REGION Network 57: ABFV 204 CLOSE FB
   RUNG wire#powerrail
      { S7_Templates := "SrcType := Int" } EQ_Contact(in1 := "MODE SELECTION DB"."UF PLC_1 MODE BUFF", in2 := 1)
      { S7_Templates := "SrcType := Int" } EQ_Contact(in1 := "MODE SELECTION DB"."UF PLC_1 PROCESS BUFF", in2 := 255)
      Contact( "INPUT MAPPING DB"."ABFV 204 FEED BACK CLOSE" )
      Move(in := 260, out1 => "MODE SELECTION DB"."UF PLC_1 PROCESS BUFF")
   END_RUNG
   // the same network as SCL:
   IF ("MODE SELECTION DB"."UF PLC_1 MODE BUFF" = 1) AND ("MODE SELECTION DB"."UF PLC_1 PROCESS BUFF" = 255) AND "INPUT MAPPING DB"."ABFV 204 FEED BACK CLOSE" THEN
       "MODE SELECTION DB"."UF PLC_1 PROCESS BUFF" := 260;
   END_IF;
END_REGION

REGION Network 58: ABFV 202 CLOSE FB
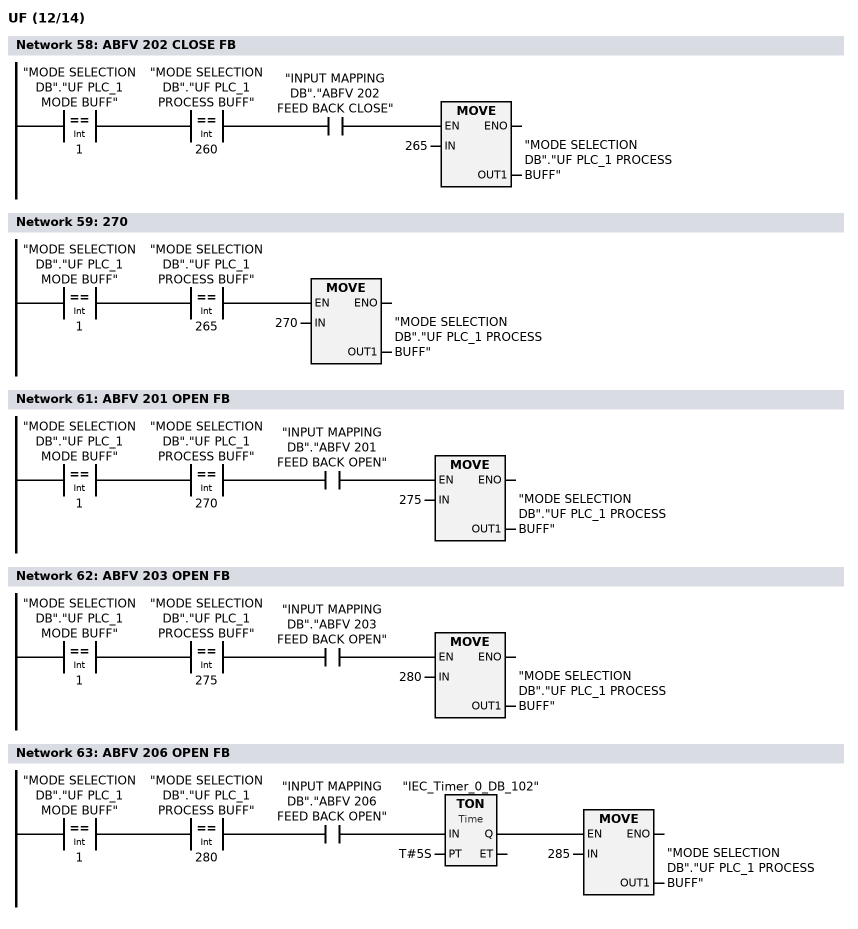
   RUNG wire#powerrail
      { S7_Templates := "SrcType := Int" } EQ_Contact(in1 := "MODE SELECTION DB"."UF PLC_1 MODE BUFF", in2 := 1)
      { S7_Templates := "SrcType := Int" } EQ_Contact(in1 := "MODE SELECTION DB"."UF PLC_1 PROCESS BUFF", in2 := 260)
      Contact( "INPUT MAPPING DB"."ABFV 202 FEED BACK CLOSE" )
      Move(in := 265, out1 => "MODE SELECTION DB"."UF PLC_1 PROCESS BUFF")
   END_RUNG
   // the same network as SCL:
   IF ("MODE SELECTION DB"."UF PLC_1 MODE BUFF" = 1) AND ("MODE SELECTION DB"."UF PLC_1 PROCESS BUFF" = 260) AND "INPUT MAPPING DB"."ABFV 202 FEED BACK CLOSE" THEN
       "MODE SELECTION DB"."UF PLC_1 PROCESS BUFF" := 265;
   END_IF;
END_REGION

REGION Network 59: 270
   RUNG wire#powerrail
      { S7_Templates := "SrcType := Int" } EQ_Contact(in1 := "MODE SELECTION DB"."UF PLC_1 MODE BUFF", in2 := 1)
      { S7_Templates := "SrcType := Int" } EQ_Contact(in1 := "MODE SELECTION DB"."UF PLC_1 PROCESS BUFF", in2 := 265)
      Move(in := 270, out1 => "MODE SELECTION DB"."UF PLC_1 PROCESS BUFF")
   END_RUNG
   // the same network as SCL:
   IF ("MODE SELECTION DB"."UF PLC_1 MODE BUFF" = 1) AND ("MODE SELECTION DB"."UF PLC_1 PROCESS BUFF" = 265) THEN
       "MODE SELECTION DB"."UF PLC_1 PROCESS BUFF" := 270;
   END_IF;
END_REGION

REGION Network 61: ABFV 201 OPEN FB
   RUNG wire#powerrail
      { S7_Templates := "SrcType := Int" } EQ_Contact(in1 := "MODE SELECTION DB"."UF PLC_1 MODE BUFF", in2 := 1)
      { S7_Templates := "SrcType := Int" } EQ_Contact(in1 := "MODE SELECTION DB"."UF PLC_1 PROCESS BUFF", in2 := 270)
      Contact( "INPUT MAPPING DB"."ABFV 201 FEED BACK OPEN" )
      Move(in := 275, out1 => "MODE SELECTION DB"."UF PLC_1 PROCESS BUFF")
   END_RUNG
   // the same network as SCL:
   IF ("MODE SELECTION DB"."UF PLC_1 MODE BUFF" = 1) AND ("MODE SELECTION DB"."UF PLC_1 PROCESS BUFF" = 270) AND "INPUT MAPPING DB"."ABFV 201 FEED BACK OPEN" THEN
       "MODE SELECTION DB"."UF PLC_1 PROCESS BUFF" := 275;
   END_IF;
END_REGION

REGION Network 62: ABFV 203 OPEN FB
   RUNG wire#powerrail
      { S7_Templates := "SrcType := Int" } EQ_Contact(in1 := "MODE SELECTION DB"."UF PLC_1 MODE BUFF", in2 := 1)
      { S7_Templates := "SrcType := Int" } EQ_Contact(in1 := "MODE SELECTION DB"."UF PLC_1 PROCESS BUFF", in2 := 275)
      Contact( "INPUT MAPPING DB"."ABFV 203 FEED BACK OPEN" )
      Move(in := 280, out1 => "MODE SELECTION DB"."UF PLC_1 PROCESS BUFF")
   END_RUNG
   // the same network as SCL:
   IF ("MODE SELECTION DB"."UF PLC_1 MODE BUFF" = 1) AND ("MODE SELECTION DB"."UF PLC_1 PROCESS BUFF" = 275) AND "INPUT MAPPING DB"."ABFV 203 FEED BACK OPEN" THEN
       "MODE SELECTION DB"."UF PLC_1 PROCESS BUFF" := 280;
   END_IF;
END_REGION

REGION Network 63: ABFV 206 OPEN FB
   RUNG wire#powerrail
      { S7_Templates := "SrcType := Int" } EQ_Contact(in1 := "MODE SELECTION DB"."UF PLC_1 MODE BUFF", in2 := 1)
      { S7_Templates := "SrcType := Int" } EQ_Contact(in1 := "MODE SELECTION DB"."UF PLC_1 PROCESS BUFF", in2 := 280)
      Contact( "INPUT MAPPING DB"."ABFV 206 FEED BACK OPEN" )
      { S7_Templates := "time_type := Time" } "IEC_Timer_0_DB_102".TON(pt := T#5S, et =>)
      Move(in := 285, out1 => "MODE SELECTION DB"."UF PLC_1 PROCESS BUFF")
   END_RUNG
   // the same network as SCL:
   "IEC_Timer_0_DB_102".TON(IN := ("MODE SELECTION DB"."UF PLC_1 MODE BUFF" = 1) AND ("MODE SELECTION DB"."UF PLC_1 PROCESS BUFF" = 280) AND "INPUT MAPPING DB"."ABFV 206 FEED BACK OPEN",
                           PT := T#5S);
   IF "IEC_Timer_0_DB_102".Q THEN "MODE SELECTION DB"."UF PLC_1 PROCESS BUFF" := 285; END_IF;
END_REGION

REGION Network 64: FORWARD FLUSH_2
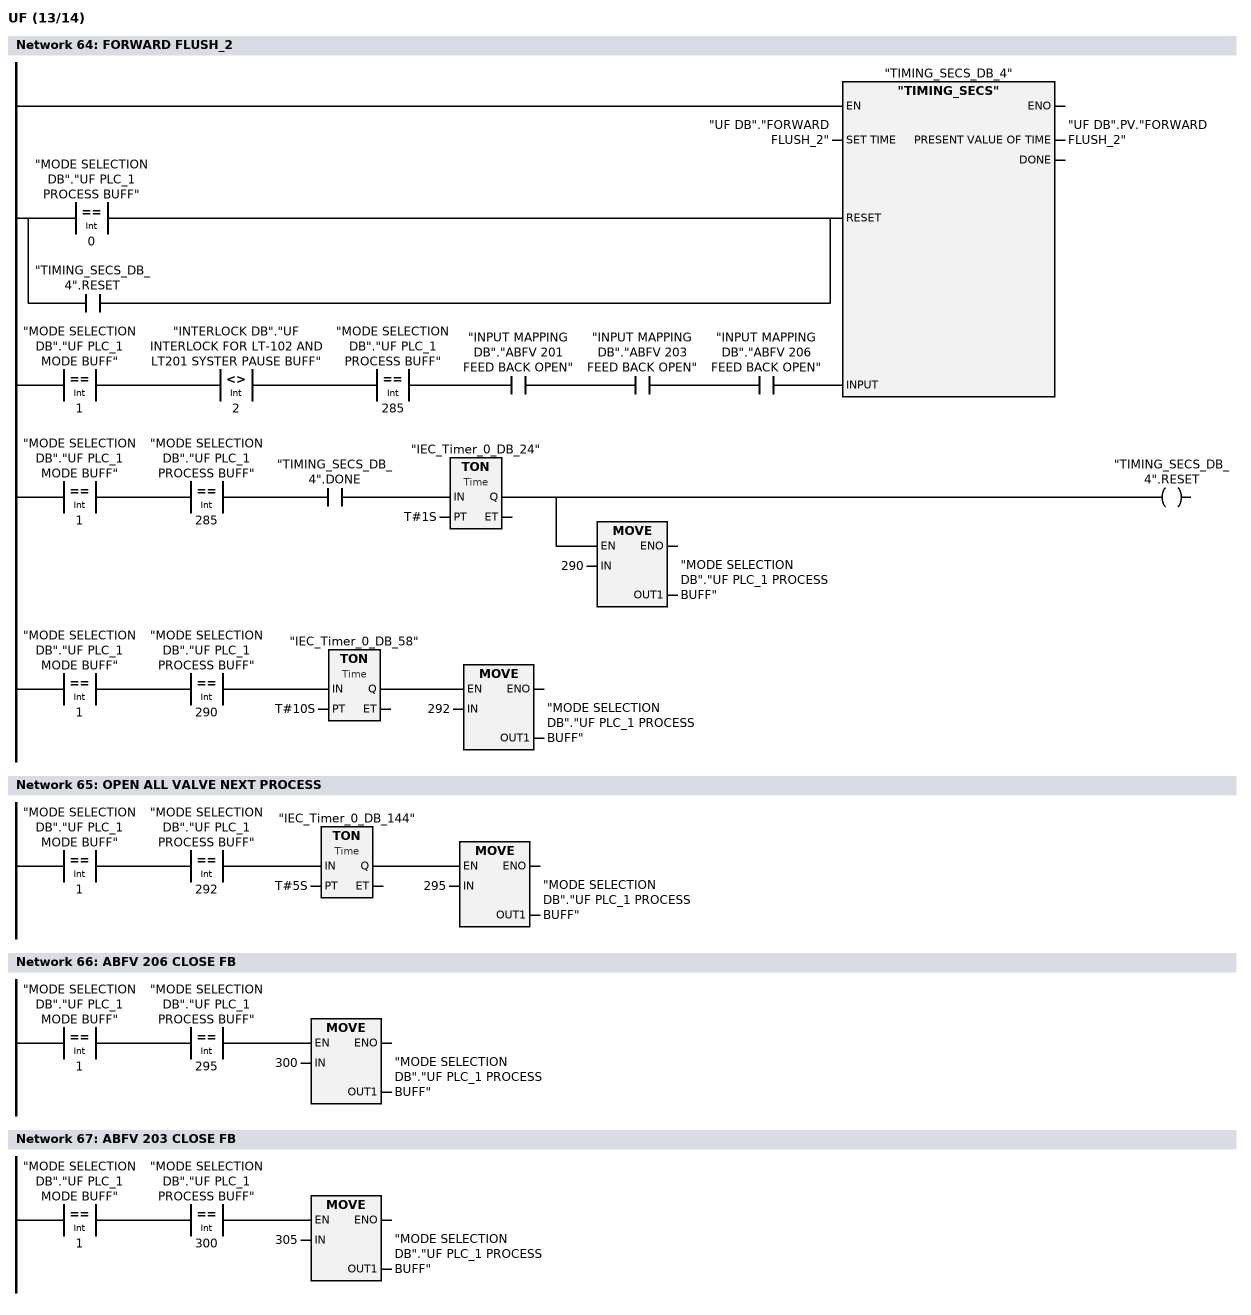
   RUNG wire#powerrail
      "TIMING_SECS_DB_4"(RESET := wire#w1, INPUT := wire#w2, "SET TIME" := "UF DB"."FORWARD FLUSH_2", "PRESENT VALUE OF TIME" => "UF DB".PV."FORWARD FLUSH_2", DONE =>)
   END_RUNG
   RUNG wire#powerrail
      { S7_Templates := "SrcType := Int" } EQ_Contact(in1 := "MODE SELECTION DB"."UF PLC_1 PROCESS BUFF", in2 := 0)
   END_RUNG wire#w1
   RUNG wire#powerrail
      Contact( "TIMING_SECS_DB_4".RESET )
   END_RUNG wire#w1
   RUNG wire#powerrail
      { S7_Templates := "SrcType := Int" } EQ_Contact(in1 := "MODE SELECTION DB"."UF PLC_1 MODE BUFF", in2 := 1)
      { S7_Templates := "SrcType := Int" } NE_Contact(in1 := "INTERLOCK DB"."UF INTERLOCK FOR LT-102 AND LT201 SYSTER PAUSE BUFF", in2 := 2)
      { S7_Templates := "SrcType := Int" } EQ_Contact(in1 := "MODE SELECTION DB"."UF PLC_1 PROCESS BUFF", in2 := 285)
      Contact( "INPUT MAPPING DB"."ABFV 201 FEED BACK OPEN" )
      Contact( "INPUT MAPPING DB"."ABFV 203 FEED BACK OPEN" )
      Contact( "INPUT MAPPING DB"."ABFV 206 FEED BACK OPEN" )
   END_RUNG wire#w2
   RUNG wire#powerrail
      { S7_Templates := "SrcType := Int" } EQ_Contact(in1 := "MODE SELECTION DB"."UF PLC_1 MODE BUFF", in2 := 1)
      { S7_Templates := "SrcType := Int" } EQ_Contact(in1 := "MODE SELECTION DB"."UF PLC_1 PROCESS BUFF", in2 := 285)
      Contact( "TIMING_SECS_DB_4".DONE )
      { S7_Templates := "time_type := Time" } "IEC_Timer_0_DB_24".TON(pt := T#1S, et =>)
      wire#w3
      Coil( "TIMING_SECS_DB_4".RESET )
   END_RUNG
   RUNG wire#w3
      Move(in := 290, out1 => "MODE SELECTION DB"."UF PLC_1 PROCESS BUFF")
   END_RUNG
   RUNG wire#powerrail
      { S7_Templates := "SrcType := Int" } EQ_Contact(in1 := "MODE SELECTION DB"."UF PLC_1 MODE BUFF", in2 := 1)
      { S7_Templates := "SrcType := Int" } EQ_Contact(in1 := "MODE SELECTION DB"."UF PLC_1 PROCESS BUFF", in2 := 290)
      { S7_Templates := "time_type := Time" } "IEC_Timer_0_DB_58".TON(pt := T#10S, et =>)
      Move(in := 292, out1 => "MODE SELECTION DB"."UF PLC_1 PROCESS BUFF")
   END_RUNG
   // the same network as SCL:
   "TIMING_SECS_DB_4"("SET TIME" := "UF DB"."FORWARD FLUSH_2",   // "TIMING_SECS"
                      RESET := ("MODE SELECTION DB"."UF PLC_1 PROCESS BUFF" = 0) OR "TIMING_SECS_DB_4".RESET,
                      INPUT := ("MODE SELECTION DB"."UF PLC_1 MODE BUFF" = 1) AND ("INTERLOCK DB"."UF INTERLOCK FOR LT-102 AND LT201 SYSTER PAUSE BUFF" <> 2) AND ("MODE SELECTION DB"."UF PLC_1 PROCESS BUFF" = 285) AND "INPUT MAPPING DB"."ABFV 201 FEED BACK OPEN" AND "INPUT MAPPING DB"."ABFV 203 FEED BACK OPEN" AND "INPUT MAPPING DB"."ABFV 206 FEED BACK OPEN",
                      "PRESENT VALUE OF TIME" => "UF DB".PV."FORWARD FLUSH_2");
   "IEC_Timer_0_DB_24".TON(IN := ("MODE SELECTION DB"."UF PLC_1 MODE BUFF" = 1) AND ("MODE SELECTION DB"."UF PLC_1 PROCESS BUFF" = 285) AND "TIMING_SECS_DB_4".DONE,
                           PT := T#1S);
   "TIMING_SECS_DB_4".RESET := "IEC_Timer_0_DB_24".Q;
   IF "IEC_Timer_0_DB_24".Q THEN "MODE SELECTION DB"."UF PLC_1 PROCESS BUFF" := 290; END_IF;
   "IEC_Timer_0_DB_58".TON(IN := ("MODE SELECTION DB"."UF PLC_1 MODE BUFF" = 1) AND ("MODE SELECTION DB"."UF PLC_1 PROCESS BUFF" = 290),
                           PT := T#10S);
   IF "IEC_Timer_0_DB_58".Q THEN "MODE SELECTION DB"."UF PLC_1 PROCESS BUFF" := 292; END_IF;
END_REGION

REGION Network 65: OPEN ALL VALVE NEXT PROCESS
   RUNG wire#powerrail
      { S7_Templates := "SrcType := Int" } EQ_Contact(in1 := "MODE SELECTION DB"."UF PLC_1 MODE BUFF", in2 := 1)
      { S7_Templates := "SrcType := Int" } EQ_Contact(in1 := "MODE SELECTION DB"."UF PLC_1 PROCESS BUFF", in2 := 292)
      { S7_Templates := "time_type := Time" } "IEC_Timer_0_DB_144".TON(pt := T#5S, et =>)
      Move(in := 295, out1 => "MODE SELECTION DB"."UF PLC_1 PROCESS BUFF")
   END_RUNG
   // the same network as SCL:
   "IEC_Timer_0_DB_144".TON(IN := ("MODE SELECTION DB"."UF PLC_1 MODE BUFF" = 1) AND ("MODE SELECTION DB"."UF PLC_1 PROCESS BUFF" = 292),
                           PT := T#5S);
   IF "IEC_Timer_0_DB_144".Q THEN "MODE SELECTION DB"."UF PLC_1 PROCESS BUFF" := 295; END_IF;
END_REGION

REGION Network 66: ABFV 206 CLOSE FB
   RUNG wire#powerrail
      { S7_Templates := "SrcType := Int" } EQ_Contact(in1 := "MODE SELECTION DB"."UF PLC_1 MODE BUFF", in2 := 1)
      { S7_Templates := "SrcType := Int" } EQ_Contact(in1 := "MODE SELECTION DB"."UF PLC_1 PROCESS BUFF", in2 := 295)
      Move(in := 300, out1 => "MODE SELECTION DB"."UF PLC_1 PROCESS BUFF")
   END_RUNG
   // the same network as SCL:
   IF ("MODE SELECTION DB"."UF PLC_1 MODE BUFF" = 1) AND ("MODE SELECTION DB"."UF PLC_1 PROCESS BUFF" = 295) THEN
       "MODE SELECTION DB"."UF PLC_1 PROCESS BUFF" := 300;
   END_IF;
END_REGION

REGION Network 67: ABFV 203 CLOSE FB
   RUNG wire#powerrail
      { S7_Templates := "SrcType := Int" } EQ_Contact(in1 := "MODE SELECTION DB"."UF PLC_1 MODE BUFF", in2 := 1)
      { S7_Templates := "SrcType := Int" } EQ_Contact(in1 := "MODE SELECTION DB"."UF PLC_1 PROCESS BUFF", in2 := 300)
      Move(in := 305, out1 => "MODE SELECTION DB"."UF PLC_1 PROCESS BUFF")
   END_RUNG
   // the same network as SCL:
   IF ("MODE SELECTION DB"."UF PLC_1 MODE BUFF" = 1) AND ("MODE SELECTION DB"."UF PLC_1 PROCESS BUFF" = 300) THEN
       "MODE SELECTION DB"."UF PLC_1 PROCESS BUFF" := 305;
   END_IF;
END_REGION

REGION Network 68: ABFV 201 CLOSE FB
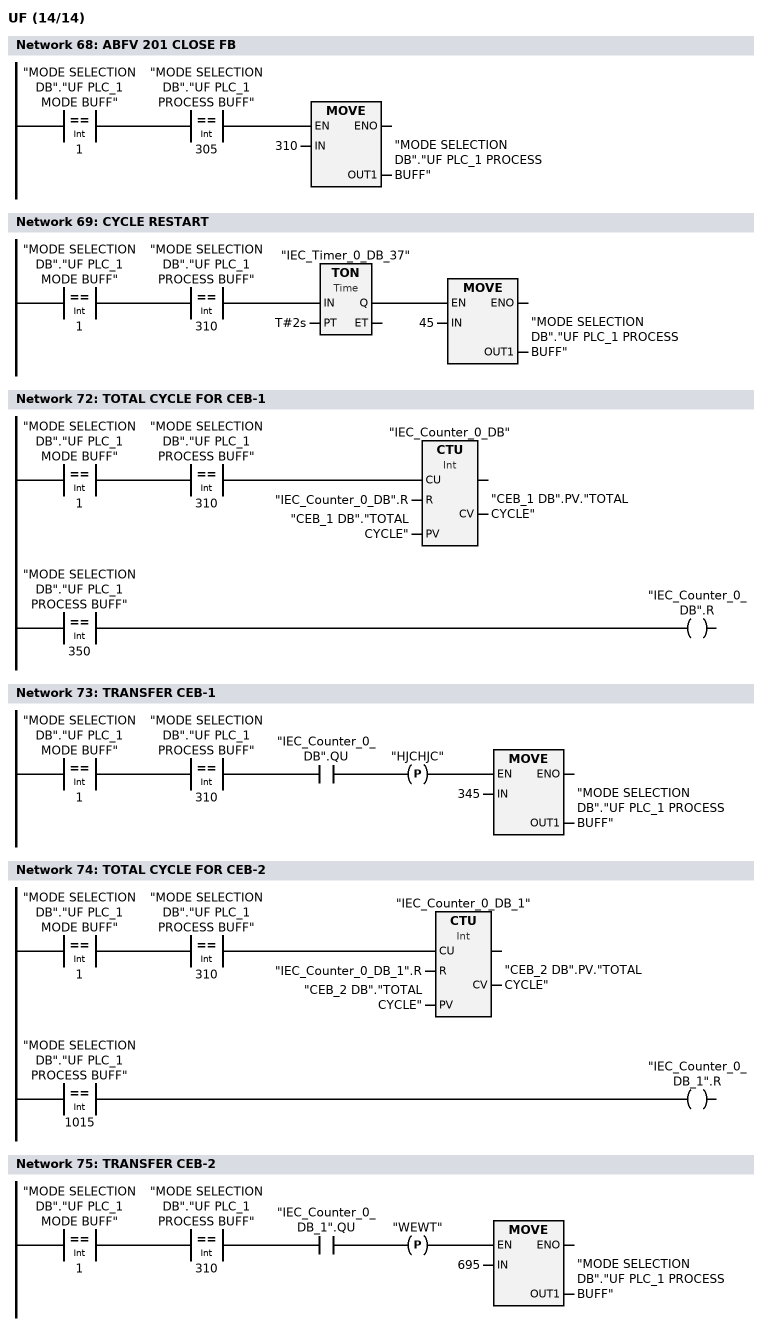
   RUNG wire#powerrail
      { S7_Templates := "SrcType := Int" } EQ_Contact(in1 := "MODE SELECTION DB"."UF PLC_1 MODE BUFF", in2 := 1)
      { S7_Templates := "SrcType := Int" } EQ_Contact(in1 := "MODE SELECTION DB"."UF PLC_1 PROCESS BUFF", in2 := 305)
      Move(in := 310, out1 => "MODE SELECTION DB"."UF PLC_1 PROCESS BUFF")
   END_RUNG
   // the same network as SCL:
   IF ("MODE SELECTION DB"."UF PLC_1 MODE BUFF" = 1) AND ("MODE SELECTION DB"."UF PLC_1 PROCESS BUFF" = 305) THEN
       "MODE SELECTION DB"."UF PLC_1 PROCESS BUFF" := 310;
   END_IF;
END_REGION

REGION Network 69: CYCLE RESTART
   RUNG wire#powerrail
      { S7_Templates := "SrcType := Int" } EQ_Contact(in1 := "MODE SELECTION DB"."UF PLC_1 MODE BUFF", in2 := 1)
      { S7_Templates := "SrcType := Int" } EQ_Contact(in1 := "MODE SELECTION DB"."UF PLC_1 PROCESS BUFF", in2 := 310)
      { S7_Templates := "time_type := Time" } "IEC_Timer_0_DB_37".TON(pt := T#2s, et =>)
      Move(in := 45, out1 => "MODE SELECTION DB"."UF PLC_1 PROCESS BUFF")
   END_RUNG
   // the same network as SCL:
   "IEC_Timer_0_DB_37".TON(IN := ("MODE SELECTION DB"."UF PLC_1 MODE BUFF" = 1) AND ("MODE SELECTION DB"."UF PLC_1 PROCESS BUFF" = 310),
                           PT := T#2s);
   IF "IEC_Timer_0_DB_37".Q THEN "MODE SELECTION DB"."UF PLC_1 PROCESS BUFF" := 45; END_IF;
END_REGION

REGION Network 72: TOTAL CYCLE FOR CEB-1
   RUNG wire#powerrail
      { S7_Templates := "SrcType := Int" } EQ_Contact(in1 := "MODE SELECTION DB"."UF PLC_1 MODE BUFF", in2 := 1)
      { S7_Templates := "SrcType := Int" } EQ_Contact(in1 := "MODE SELECTION DB"."UF PLC_1 PROCESS BUFF", in2 := 310)
      { S7_Templates := "value_type := Int" } "IEC_Counter_0_DB".CTU(r := "IEC_Counter_0_DB".R, pv := "CEB_1 DB"."TOTAL CYCLE", cv => "CEB_1 DB".PV."TOTAL CYCLE")
   END_RUNG
   RUNG wire#powerrail
      { S7_Templates := "SrcType := Int" } EQ_Contact(in1 := "MODE SELECTION DB"."UF PLC_1 PROCESS BUFF", in2 := 350)
      Coil( "IEC_Counter_0_DB".R )
   END_RUNG
   // the same network as SCL:
   "IEC_Counter_0_DB".CTU(CU := ("MODE SELECTION DB"."UF PLC_1 MODE BUFF" = 1) AND ("MODE SELECTION DB"."UF PLC_1 PROCESS BUFF" = 310),
                          R := "IEC_Counter_0_DB".R,
                          PV := "CEB_1 DB"."TOTAL CYCLE",
                          CV => "CEB_1 DB".PV."TOTAL CYCLE");
   "IEC_Counter_0_DB".R := "MODE SELECTION DB"."UF PLC_1 PROCESS BUFF" = 350;
END_REGION

REGION Network 73: TRANSFER CEB-1
   RUNG wire#powerrail
      { S7_Templates := "SrcType := Int" } EQ_Contact(in1 := "MODE SELECTION DB"."UF PLC_1 MODE BUFF", in2 := 1)
      { S7_Templates := "SrcType := Int" } EQ_Contact(in1 := "MODE SELECTION DB"."UF PLC_1 PROCESS BUFF", in2 := 310)
      Contact( "IEC_Counter_0_DB".QU )
      P_Trig( "HJCHJC" )
      Move(in := 345, out1 => "MODE SELECTION DB"."UF PLC_1 PROCESS BUFF")
   END_RUNG
   // the same network as SCL:
   #_w1 := ("MODE SELECTION DB"."UF PLC_1 MODE BUFF" = 1) AND ("MODE SELECTION DB"."UF PLC_1 PROCESS BUFF" = 310) AND "IEC_Counter_0_DB".QU;
   #_w2 := #_w1 AND NOT "HJCHJC";   // rising edge
   "HJCHJC" := #_w1;
   IF #_w2 THEN "MODE SELECTION DB"."UF PLC_1 PROCESS BUFF" := 345; END_IF;
END_REGION

REGION Network 74: TOTAL CYCLE FOR CEB-2
   RUNG wire#powerrail
      { S7_Templates := "SrcType := Int" } EQ_Contact(in1 := "MODE SELECTION DB"."UF PLC_1 MODE BUFF", in2 := 1)
      { S7_Templates := "SrcType := Int" } EQ_Contact(in1 := "MODE SELECTION DB"."UF PLC_1 PROCESS BUFF", in2 := 310)
      { S7_Templates := "value_type := Int" } "IEC_Counter_0_DB_1".CTU(r := "IEC_Counter_0_DB_1".R, pv := "CEB_2 DB"."TOTAL CYCLE", cv => "CEB_2 DB".PV."TOTAL CYCLE")
   END_RUNG
   RUNG wire#powerrail
      { S7_Templates := "SrcType := Int" } EQ_Contact(in1 := "MODE SELECTION DB"."UF PLC_1 PROCESS BUFF", in2 := 1015)
      Coil( "IEC_Counter_0_DB_1".R )
   END_RUNG
   // the same network as SCL:
   "IEC_Counter_0_DB_1".CTU(CU := ("MODE SELECTION DB"."UF PLC_1 MODE BUFF" = 1) AND ("MODE SELECTION DB"."UF PLC_1 PROCESS BUFF" = 310),
                           R := "IEC_Counter_0_DB_1".R,
                           PV := "CEB_2 DB"."TOTAL CYCLE",
                           CV => "CEB_2 DB".PV."TOTAL CYCLE");
   "IEC_Counter_0_DB_1".R := "MODE SELECTION DB"."UF PLC_1 PROCESS BUFF" = 1015;
END_REGION

REGION Network 75: TRANSFER CEB-2
   RUNG wire#powerrail
      { S7_Templates := "SrcType := Int" } EQ_Contact(in1 := "MODE SELECTION DB"."UF PLC_1 MODE BUFF", in2 := 1)
      { S7_Templates := "SrcType := Int" } EQ_Contact(in1 := "MODE SELECTION DB"."UF PLC_1 PROCESS BUFF", in2 := 310)
      Contact( "IEC_Counter_0_DB_1".QU )
      P_Trig( "WEWT" )
      Move(in := 695, out1 => "MODE SELECTION DB"."UF PLC_1 PROCESS BUFF")
   END_RUNG
   // the same network as SCL:
   #_w1 := ("MODE SELECTION DB"."UF PLC_1 MODE BUFF" = 1) AND ("MODE SELECTION DB"."UF PLC_1 PROCESS BUFF" = 310) AND "IEC_Counter_0_DB_1".QU;
   #_w2 := #_w1 AND NOT "WEWT";   // rising edge
   "WEWT" := #_w1;
   IF #_w2 THEN "MODE SELECTION DB"."UF PLC_1 PROCESS BUFF" := 695; END_IF;
END_REGION
END_FUNCTION

FUNCTION_BLOCK "TIMING_SECS"   // FB3, LAD
{ S7_Optimized_Access := 'TRUE' }
// stored: MemoryReserve 100, SetENOAutomatically false
   VAR_INPUT
      "SET TIME" : Int;
      RESET : Bool;
      INPUT : Bool;
   END_VAR
   VAR_OUTPUT
      "PRESENT VALUE OF TIME" : Int;
      DONE : Bool;
   END_VAR
   VAR
      "TIMER 1" { S7_SetPoint := 'True'} : IEC_TIMER;
   END_VAR
   VAR RETAIN
      "COUNTER1 1" { S7_SetPoint := 'True'} : IEC_COUNTER;
   END_VAR
   VAR_TEMP   // added for the SCL form of the ladder/FBD networks
      _w1 : Bool;
      _w2 : Bool;
   END_VAR
BEGIN

REGION Network 1
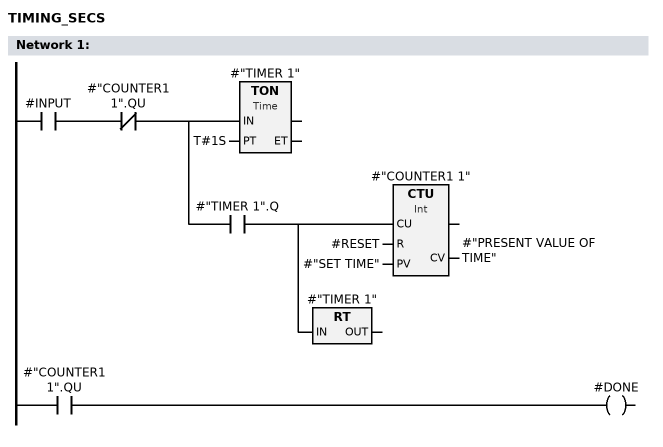
   RUNG wire#powerrail
      Contact( #INPUT )
      I_Contact( #"COUNTER1 1".QU )
      wire#w1
      { S7_Templates := "time_type := Time" } #"TIMER 1".TON(pt := T#1S, et =>)
   END_RUNG
   RUNG wire#w1
      Contact( #"TIMER 1".Q )
      wire#w2
      { S7_Templates := "value_type := Int" } #"COUNTER1 1".CTU(r := #RESET, pv := #"SET TIME", cv => #"PRESENT VALUE OF TIME")
   END_RUNG
   RUNG wire#w2
      RT_Coil( #"TIMER 1" )
   END_RUNG
   RUNG wire#powerrail
      Contact( #"COUNTER1 1".QU )
      Coil( #DONE )
   END_RUNG
   // the same network as SCL:
   #_w1 := #INPUT AND NOT #"COUNTER1 1".QU;
   #"TIMER 1".TON(IN := #_w1, PT := T#1S);
   #_w2 := #_w1 AND #"TIMER 1".Q;
   #"COUNTER1 1".CTU(CU := #_w2, R := #RESET, PV := #"SET TIME", CV => #"PRESENT VALUE OF TIME");
   IF #_w2 THEN RESET_TIMER(#"TIMER 1"); END_IF;
   #DONE := #"COUNTER1 1".QU;
END_REGION
END_FUNCTION_BLOCK

FUNCTION "CEB_1" : Void   // FC14, LAD
{ S7_Optimized_Access := 'TRUE' }
// stored: SetENOAutomatically false
BEGIN

REGION Network 1: CEB_1 START
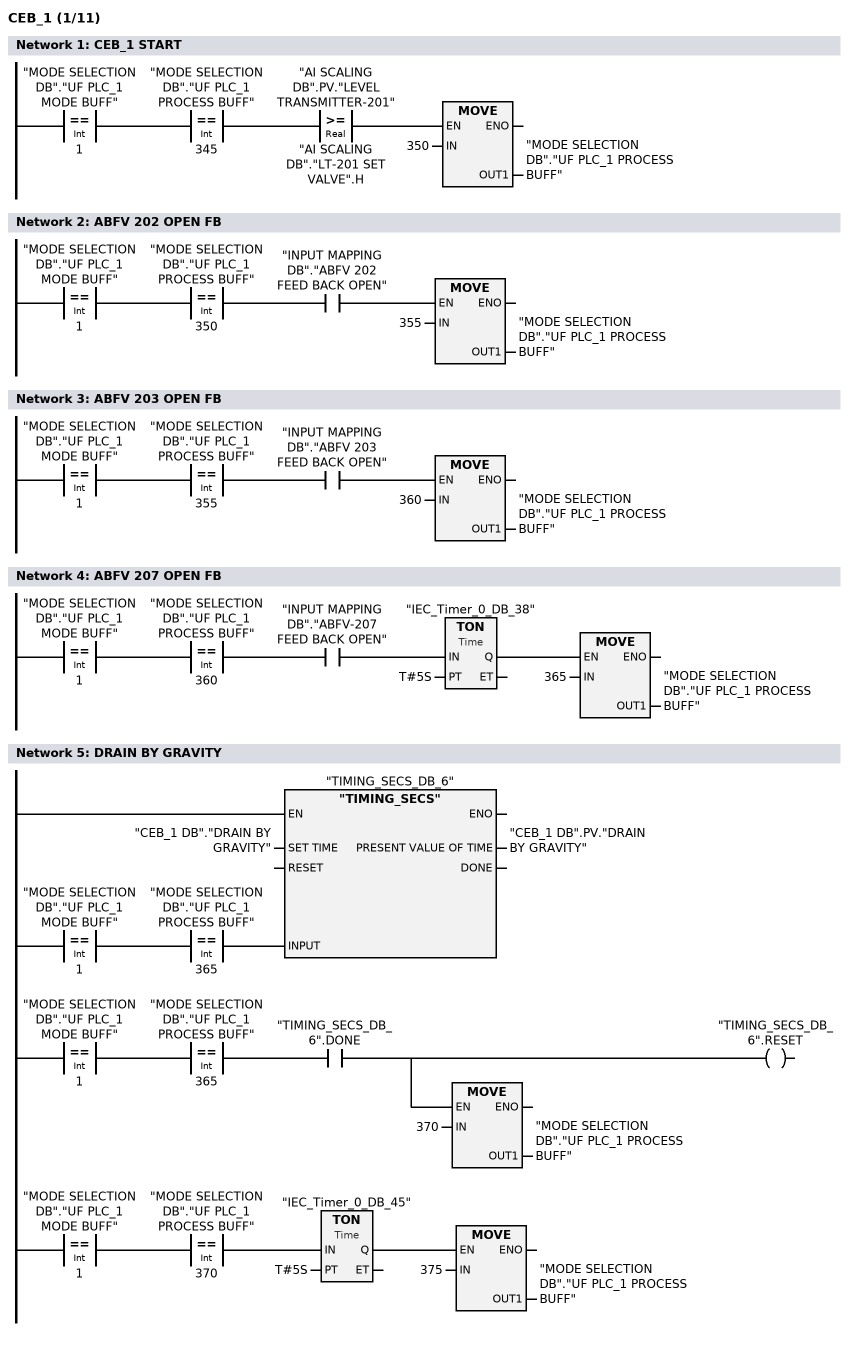
   RUNG wire#powerrail
      { S7_Templates := "SrcType := Int" } EQ_Contact(in1 := "MODE SELECTION DB"."UF PLC_1 MODE BUFF", in2 := 1)
      { S7_Templates := "SrcType := Int" } EQ_Contact(in1 := "MODE SELECTION DB"."UF PLC_1 PROCESS BUFF", in2 := 345)
      { S7_Templates := "SrcType := Real" } GE_Contact(in1 := "AI SCALING DB".PV."LEVEL TRANSMITTER-201", in2 := "AI SCALING DB"."LT-201 SET VALVE".H)
      Move(in := 350, out1 => "MODE SELECTION DB"."UF PLC_1 PROCESS BUFF")
   END_RUNG
   // the same network as SCL:
   IF ("MODE SELECTION DB"."UF PLC_1 MODE BUFF" = 1) AND ("MODE SELECTION DB"."UF PLC_1 PROCESS BUFF" = 345) AND ("AI SCALING DB".PV."LEVEL TRANSMITTER-201" >= "AI SCALING DB"."LT-201 SET VALVE".H) THEN
       "MODE SELECTION DB"."UF PLC_1 PROCESS BUFF" := 350;
   END_IF;
END_REGION

REGION Network 2: ABFV 202 OPEN FB
   RUNG wire#powerrail
      { S7_Templates := "SrcType := Int" } EQ_Contact(in1 := "MODE SELECTION DB"."UF PLC_1 MODE BUFF", in2 := 1)
      { S7_Templates := "SrcType := Int" } EQ_Contact(in1 := "MODE SELECTION DB"."UF PLC_1 PROCESS BUFF", in2 := 350)
      Contact( "INPUT MAPPING DB"."ABFV 202 FEED BACK OPEN" )
      Move(in := 355, out1 => "MODE SELECTION DB"."UF PLC_1 PROCESS BUFF")
   END_RUNG
   // the same network as SCL:
   IF ("MODE SELECTION DB"."UF PLC_1 MODE BUFF" = 1) AND ("MODE SELECTION DB"."UF PLC_1 PROCESS BUFF" = 350) AND "INPUT MAPPING DB"."ABFV 202 FEED BACK OPEN" THEN
       "MODE SELECTION DB"."UF PLC_1 PROCESS BUFF" := 355;
   END_IF;
END_REGION

REGION Network 3: ABFV 203 OPEN FB
   RUNG wire#powerrail
      { S7_Templates := "SrcType := Int" } EQ_Contact(in1 := "MODE SELECTION DB"."UF PLC_1 MODE BUFF", in2 := 1)
      { S7_Templates := "SrcType := Int" } EQ_Contact(in1 := "MODE SELECTION DB"."UF PLC_1 PROCESS BUFF", in2 := 355)
      Contact( "INPUT MAPPING DB"."ABFV 203 FEED BACK OPEN" )
      Move(in := 360, out1 => "MODE SELECTION DB"."UF PLC_1 PROCESS BUFF")
   END_RUNG
   // the same network as SCL:
   IF ("MODE SELECTION DB"."UF PLC_1 MODE BUFF" = 1) AND ("MODE SELECTION DB"."UF PLC_1 PROCESS BUFF" = 355) AND "INPUT MAPPING DB"."ABFV 203 FEED BACK OPEN" THEN
       "MODE SELECTION DB"."UF PLC_1 PROCESS BUFF" := 360;
   END_IF;
END_REGION

REGION Network 4: ABFV 207 OPEN FB
   RUNG wire#powerrail
      { S7_Templates := "SrcType := Int" } EQ_Contact(in1 := "MODE SELECTION DB"."UF PLC_1 MODE BUFF", in2 := 1)
      { S7_Templates := "SrcType := Int" } EQ_Contact(in1 := "MODE SELECTION DB"."UF PLC_1 PROCESS BUFF", in2 := 360)
      Contact( "INPUT MAPPING DB"."ABFV-207 FEED BACK OPEN" )
      { S7_Templates := "time_type := Time" } "IEC_Timer_0_DB_38".TON(pt := T#5S, et =>)
      Move(in := 365, out1 => "MODE SELECTION DB"."UF PLC_1 PROCESS BUFF")
   END_RUNG
   // the same network as SCL:
   "IEC_Timer_0_DB_38".TON(IN := ("MODE SELECTION DB"."UF PLC_1 MODE BUFF" = 1) AND ("MODE SELECTION DB"."UF PLC_1 PROCESS BUFF" = 360) AND "INPUT MAPPING DB"."ABFV-207 FEED BACK OPEN",
                           PT := T#5S);
   IF "IEC_Timer_0_DB_38".Q THEN "MODE SELECTION DB"."UF PLC_1 PROCESS BUFF" := 365; END_IF;
END_REGION

REGION Network 5: DRAIN BY GRAVITY
   RUNG wire#powerrail
      "TIMING_SECS_DB_6"(INPUT := wire#w1, "SET TIME" := "CEB_1 DB"."DRAIN BY GRAVITY", RESET :=, "PRESENT VALUE OF TIME" => "CEB_1 DB".PV."DRAIN BY GRAVITY", DONE =>)
   END_RUNG
   RUNG wire#powerrail
      { S7_Templates := "SrcType := Int" } EQ_Contact(in1 := "MODE SELECTION DB"."UF PLC_1 MODE BUFF", in2 := 1)
      { S7_Templates := "SrcType := Int" } EQ_Contact(in1 := "MODE SELECTION DB"."UF PLC_1 PROCESS BUFF", in2 := 365)
   END_RUNG wire#w1
   RUNG wire#powerrail
      { S7_Templates := "SrcType := Int" } EQ_Contact(in1 := "MODE SELECTION DB"."UF PLC_1 MODE BUFF", in2 := 1)
      { S7_Templates := "SrcType := Int" } EQ_Contact(in1 := "MODE SELECTION DB"."UF PLC_1 PROCESS BUFF", in2 := 365)
      Contact( "TIMING_SECS_DB_6".DONE )
      wire#w2
      Coil( "TIMING_SECS_DB_6".RESET )
   END_RUNG
   RUNG wire#w2
      Move(in := 370, out1 => "MODE SELECTION DB"."UF PLC_1 PROCESS BUFF")
   END_RUNG
   RUNG wire#powerrail
      { S7_Templates := "SrcType := Int" } EQ_Contact(in1 := "MODE SELECTION DB"."UF PLC_1 MODE BUFF", in2 := 1)
      { S7_Templates := "SrcType := Int" } EQ_Contact(in1 := "MODE SELECTION DB"."UF PLC_1 PROCESS BUFF", in2 := 370)
      { S7_Templates := "time_type := Time" } "IEC_Timer_0_DB_45".TON(pt := T#5S, et =>)
      Move(in := 375, out1 => "MODE SELECTION DB"."UF PLC_1 PROCESS BUFF")
   END_RUNG
   // the same network as SCL:
   "TIMING_SECS_DB_6"("SET TIME" := "CEB_1 DB"."DRAIN BY GRAVITY",   // "TIMING_SECS"
                      INPUT := ("MODE SELECTION DB"."UF PLC_1 MODE BUFF" = 1) AND ("MODE SELECTION DB"."UF PLC_1 PROCESS BUFF" = 365),
                      "PRESENT VALUE OF TIME" => "CEB_1 DB".PV."DRAIN BY GRAVITY");
   "TIMING_SECS_DB_6".RESET := ("MODE SELECTION DB"."UF PLC_1 MODE BUFF" = 1) AND ("MODE SELECTION DB"."UF PLC_1 PROCESS BUFF" = 365) AND "TIMING_SECS_DB_6".DONE;
   IF "TIMING_SECS_DB_6".RESET THEN "MODE SELECTION DB"."UF PLC_1 PROCESS BUFF" := 370; END_IF;
   "IEC_Timer_0_DB_45".TON(IN := ("MODE SELECTION DB"."UF PLC_1 MODE BUFF" = 1) AND ("MODE SELECTION DB"."UF PLC_1 PROCESS BUFF" = 370),
                           PT := T#5S);
   IF "IEC_Timer_0_DB_45".Q THEN "MODE SELECTION DB"."UF PLC_1 PROCESS BUFF" := 375; END_IF;
END_REGION

REGION Network 6: ABFV 207 CLOSE FB
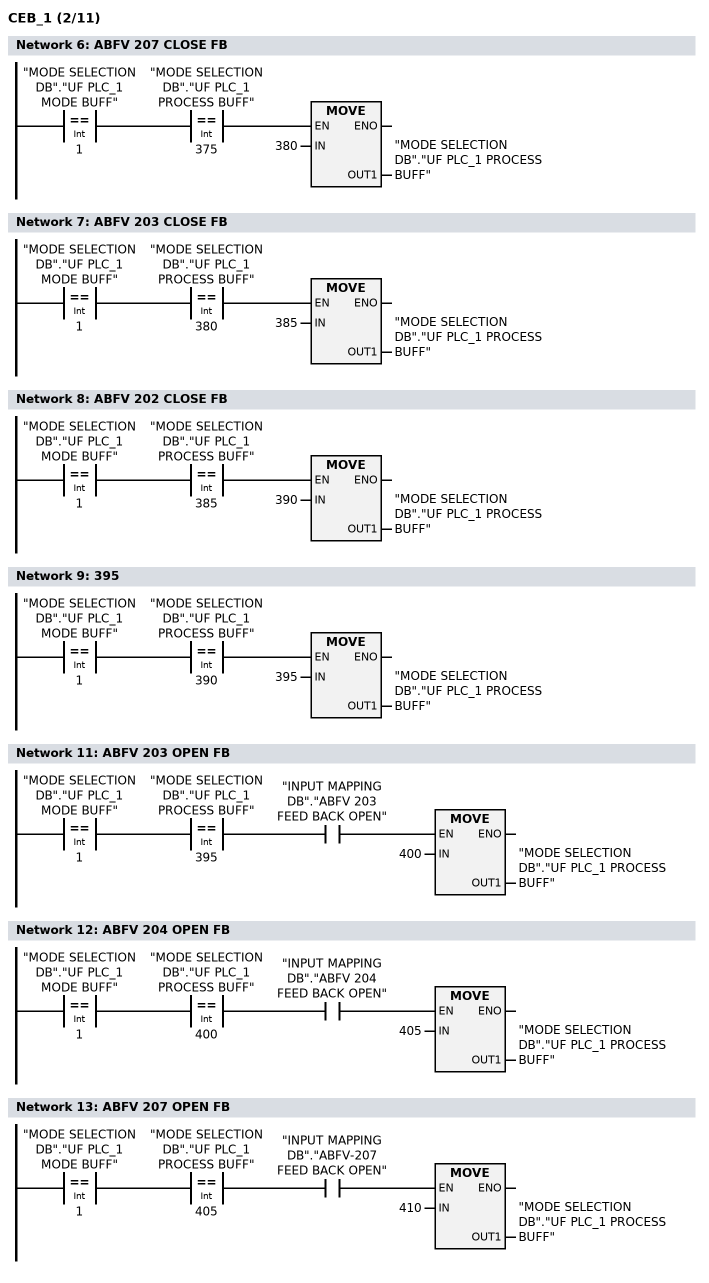
   RUNG wire#powerrail
      { S7_Templates := "SrcType := Int" } EQ_Contact(in1 := "MODE SELECTION DB"."UF PLC_1 MODE BUFF", in2 := 1)
      { S7_Templates := "SrcType := Int" } EQ_Contact(in1 := "MODE SELECTION DB"."UF PLC_1 PROCESS BUFF", in2 := 375)
      Move(in := 380, out1 => "MODE SELECTION DB"."UF PLC_1 PROCESS BUFF")
   END_RUNG
   // the same network as SCL:
   IF ("MODE SELECTION DB"."UF PLC_1 MODE BUFF" = 1) AND ("MODE SELECTION DB"."UF PLC_1 PROCESS BUFF" = 375) THEN
       "MODE SELECTION DB"."UF PLC_1 PROCESS BUFF" := 380;
   END_IF;
END_REGION

REGION Network 7: ABFV 203 CLOSE FB
   RUNG wire#powerrail
      { S7_Templates := "SrcType := Int" } EQ_Contact(in1 := "MODE SELECTION DB"."UF PLC_1 MODE BUFF", in2 := 1)
      { S7_Templates := "SrcType := Int" } EQ_Contact(in1 := "MODE SELECTION DB"."UF PLC_1 PROCESS BUFF", in2 := 380)
      Move(in := 385, out1 => "MODE SELECTION DB"."UF PLC_1 PROCESS BUFF")
   END_RUNG
   // the same network as SCL:
   IF ("MODE SELECTION DB"."UF PLC_1 MODE BUFF" = 1) AND ("MODE SELECTION DB"."UF PLC_1 PROCESS BUFF" = 380) THEN
       "MODE SELECTION DB"."UF PLC_1 PROCESS BUFF" := 385;
   END_IF;
END_REGION

REGION Network 8: ABFV 202 CLOSE FB
   RUNG wire#powerrail
      { S7_Templates := "SrcType := Int" } EQ_Contact(in1 := "MODE SELECTION DB"."UF PLC_1 MODE BUFF", in2 := 1)
      { S7_Templates := "SrcType := Int" } EQ_Contact(in1 := "MODE SELECTION DB"."UF PLC_1 PROCESS BUFF", in2 := 385)
      Move(in := 390, out1 => "MODE SELECTION DB"."UF PLC_1 PROCESS BUFF")
   END_RUNG
   // the same network as SCL:
   IF ("MODE SELECTION DB"."UF PLC_1 MODE BUFF" = 1) AND ("MODE SELECTION DB"."UF PLC_1 PROCESS BUFF" = 385) THEN
       "MODE SELECTION DB"."UF PLC_1 PROCESS BUFF" := 390;
   END_IF;
END_REGION

REGION Network 9: 395
   RUNG wire#powerrail
      { S7_Templates := "SrcType := Int" } EQ_Contact(in1 := "MODE SELECTION DB"."UF PLC_1 MODE BUFF", in2 := 1)
      { S7_Templates := "SrcType := Int" } EQ_Contact(in1 := "MODE SELECTION DB"."UF PLC_1 PROCESS BUFF", in2 := 390)
      Move(in := 395, out1 => "MODE SELECTION DB"."UF PLC_1 PROCESS BUFF")
   END_RUNG
   // the same network as SCL:
   IF ("MODE SELECTION DB"."UF PLC_1 MODE BUFF" = 1) AND ("MODE SELECTION DB"."UF PLC_1 PROCESS BUFF" = 390) THEN
       "MODE SELECTION DB"."UF PLC_1 PROCESS BUFF" := 395;
   END_IF;
END_REGION

REGION Network 11: ABFV 203 OPEN FB
   RUNG wire#powerrail
      { S7_Templates := "SrcType := Int" } EQ_Contact(in1 := "MODE SELECTION DB"."UF PLC_1 MODE BUFF", in2 := 1)
      { S7_Templates := "SrcType := Int" } EQ_Contact(in1 := "MODE SELECTION DB"."UF PLC_1 PROCESS BUFF", in2 := 395)
      Contact( "INPUT MAPPING DB"."ABFV 203 FEED BACK OPEN" )
      Move(in := 400, out1 => "MODE SELECTION DB"."UF PLC_1 PROCESS BUFF")
   END_RUNG
   // the same network as SCL:
   IF ("MODE SELECTION DB"."UF PLC_1 MODE BUFF" = 1) AND ("MODE SELECTION DB"."UF PLC_1 PROCESS BUFF" = 395) AND "INPUT MAPPING DB"."ABFV 203 FEED BACK OPEN" THEN
       "MODE SELECTION DB"."UF PLC_1 PROCESS BUFF" := 400;
   END_IF;
END_REGION

REGION Network 12: ABFV 204 OPEN FB
   RUNG wire#powerrail
      { S7_Templates := "SrcType := Int" } EQ_Contact(in1 := "MODE SELECTION DB"."UF PLC_1 MODE BUFF", in2 := 1)
      { S7_Templates := "SrcType := Int" } EQ_Contact(in1 := "MODE SELECTION DB"."UF PLC_1 PROCESS BUFF", in2 := 400)
      Contact( "INPUT MAPPING DB"."ABFV 204 FEED BACK OPEN" )
      Move(in := 405, out1 => "MODE SELECTION DB"."UF PLC_1 PROCESS BUFF")
   END_RUNG
   // the same network as SCL:
   IF ("MODE SELECTION DB"."UF PLC_1 MODE BUFF" = 1) AND ("MODE SELECTION DB"."UF PLC_1 PROCESS BUFF" = 400) AND "INPUT MAPPING DB"."ABFV 204 FEED BACK OPEN" THEN
       "MODE SELECTION DB"."UF PLC_1 PROCESS BUFF" := 405;
   END_IF;
END_REGION

REGION Network 13: ABFV 207 OPEN FB
   RUNG wire#powerrail
      { S7_Templates := "SrcType := Int" } EQ_Contact(in1 := "MODE SELECTION DB"."UF PLC_1 MODE BUFF", in2 := 1)
      { S7_Templates := "SrcType := Int" } EQ_Contact(in1 := "MODE SELECTION DB"."UF PLC_1 PROCESS BUFF", in2 := 405)
      Contact( "INPUT MAPPING DB"."ABFV-207 FEED BACK OPEN" )
      Move(in := 410, out1 => "MODE SELECTION DB"."UF PLC_1 PROCESS BUFF")
   END_RUNG
   // the same network as SCL:
   IF ("MODE SELECTION DB"."UF PLC_1 MODE BUFF" = 1) AND ("MODE SELECTION DB"."UF PLC_1 PROCESS BUFF" = 405) AND "INPUT MAPPING DB"."ABFV-207 FEED BACK OPEN" THEN
       "MODE SELECTION DB"."UF PLC_1 PROCESS BUFF" := 410;
   END_IF;
END_REGION

REGION Network 14: ABFV 208 OPEN FB
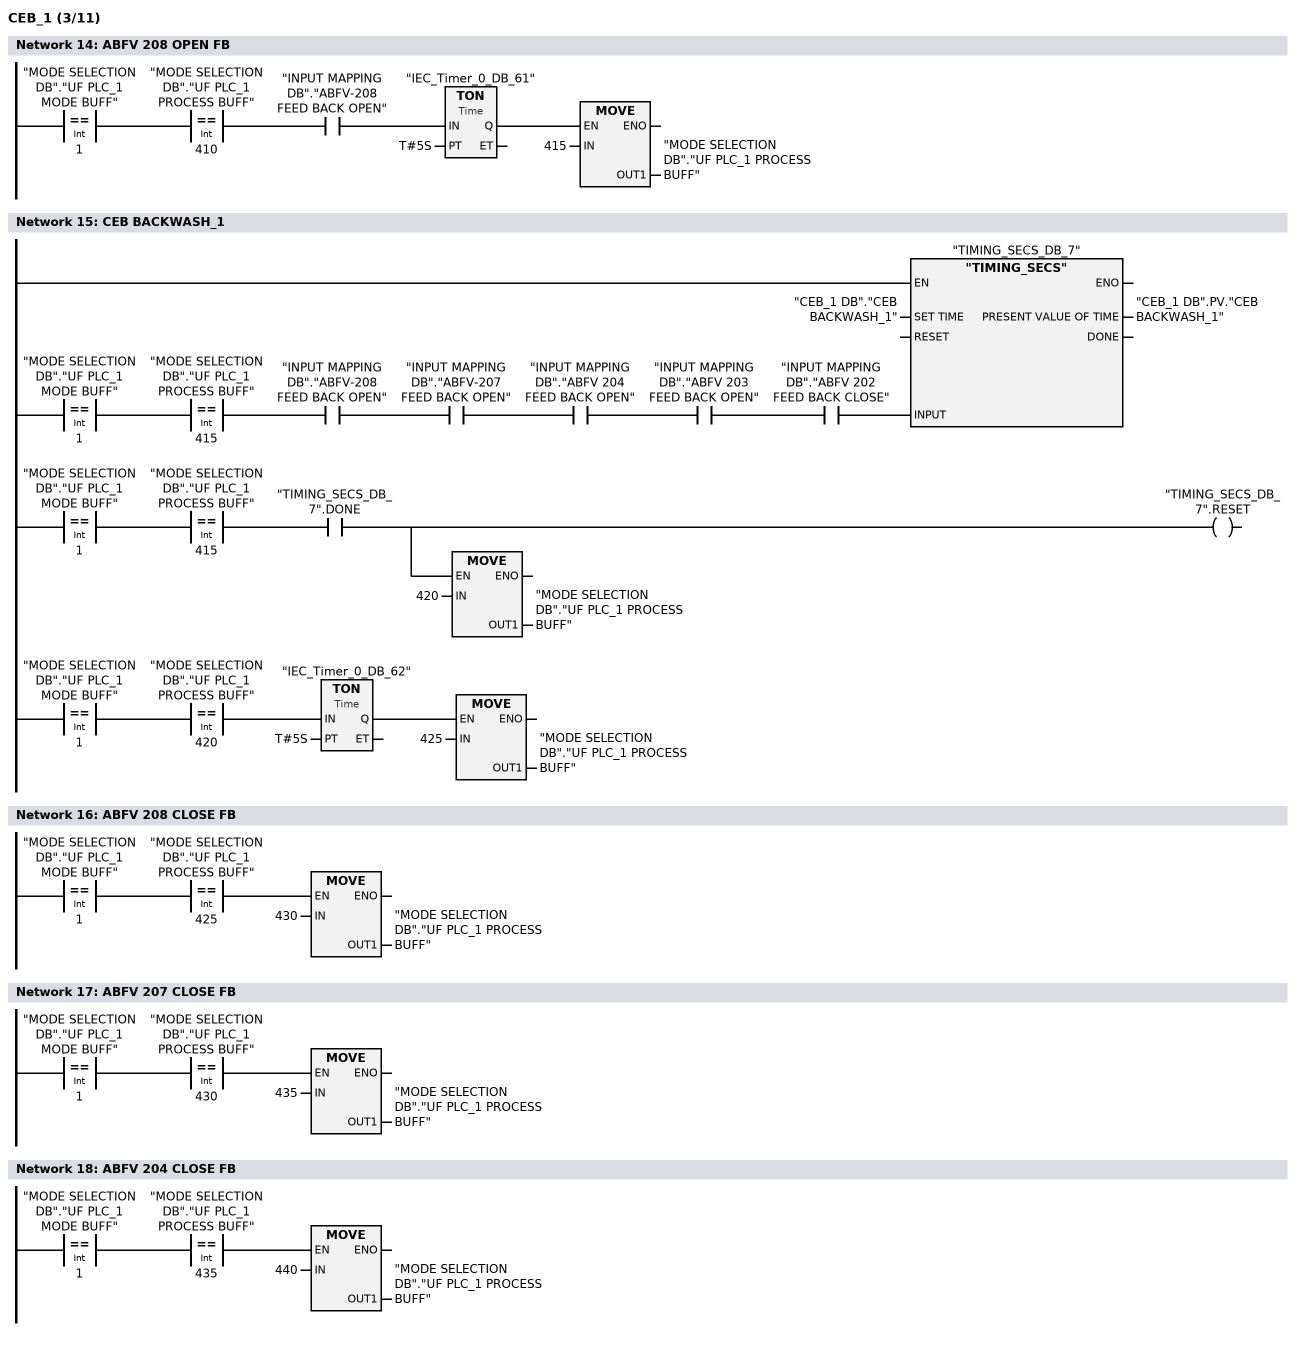
   RUNG wire#powerrail
      { S7_Templates := "SrcType := Int" } EQ_Contact(in1 := "MODE SELECTION DB"."UF PLC_1 MODE BUFF", in2 := 1)
      { S7_Templates := "SrcType := Int" } EQ_Contact(in1 := "MODE SELECTION DB"."UF PLC_1 PROCESS BUFF", in2 := 410)
      Contact( "INPUT MAPPING DB"."ABFV-208 FEED BACK OPEN" )
      { S7_Templates := "time_type := Time" } "IEC_Timer_0_DB_61".TON(pt := T#5S, et =>)
      Move(in := 415, out1 => "MODE SELECTION DB"."UF PLC_1 PROCESS BUFF")
   END_RUNG
   // the same network as SCL:
   "IEC_Timer_0_DB_61".TON(IN := ("MODE SELECTION DB"."UF PLC_1 MODE BUFF" = 1) AND ("MODE SELECTION DB"."UF PLC_1 PROCESS BUFF" = 410) AND "INPUT MAPPING DB"."ABFV-208 FEED BACK OPEN",
                           PT := T#5S);
   IF "IEC_Timer_0_DB_61".Q THEN "MODE SELECTION DB"."UF PLC_1 PROCESS BUFF" := 415; END_IF;
END_REGION

REGION Network 15: CEB BACKWASH_1
   RUNG wire#powerrail
      "TIMING_SECS_DB_7"(INPUT := wire#w1, "SET TIME" := "CEB_1 DB"."CEB BACKWASH_1", RESET :=, "PRESENT VALUE OF TIME" => "CEB_1 DB".PV."CEB BACKWASH_1", DONE =>)
   END_RUNG
   RUNG wire#powerrail
      { S7_Templates := "SrcType := Int" } EQ_Contact(in1 := "MODE SELECTION DB"."UF PLC_1 MODE BUFF", in2 := 1)
      { S7_Templates := "SrcType := Int" } EQ_Contact(in1 := "MODE SELECTION DB"."UF PLC_1 PROCESS BUFF", in2 := 415)
      Contact( "INPUT MAPPING DB"."ABFV-208 FEED BACK OPEN" )
      Contact( "INPUT MAPPING DB"."ABFV-207 FEED BACK OPEN" )
      Contact( "INPUT MAPPING DB"."ABFV 204 FEED BACK OPEN" )
      Contact( "INPUT MAPPING DB"."ABFV 203 FEED BACK OPEN" )
      Contact( "INPUT MAPPING DB"."ABFV 202 FEED BACK CLOSE" )
   END_RUNG wire#w1
   RUNG wire#powerrail
      { S7_Templates := "SrcType := Int" } EQ_Contact(in1 := "MODE SELECTION DB"."UF PLC_1 MODE BUFF", in2 := 1)
      { S7_Templates := "SrcType := Int" } EQ_Contact(in1 := "MODE SELECTION DB"."UF PLC_1 PROCESS BUFF", in2 := 415)
      Contact( "TIMING_SECS_DB_7".DONE )
      wire#w2
      Coil( "TIMING_SECS_DB_7".RESET )
   END_RUNG
   RUNG wire#w2
      Move(in := 420, out1 => "MODE SELECTION DB"."UF PLC_1 PROCESS BUFF")
   END_RUNG
   RUNG wire#powerrail
      { S7_Templates := "SrcType := Int" } EQ_Contact(in1 := "MODE SELECTION DB"."UF PLC_1 MODE BUFF", in2 := 1)
      { S7_Templates := "SrcType := Int" } EQ_Contact(in1 := "MODE SELECTION DB"."UF PLC_1 PROCESS BUFF", in2 := 420)
      { S7_Templates := "time_type := Time" } "IEC_Timer_0_DB_62".TON(pt := T#5S, et =>)
      Move(in := 425, out1 => "MODE SELECTION DB"."UF PLC_1 PROCESS BUFF")
   END_RUNG
   // the same network as SCL:
   "TIMING_SECS_DB_7"("SET TIME" := "CEB_1 DB"."CEB BACKWASH_1",   // "TIMING_SECS"
                      INPUT := ("MODE SELECTION DB"."UF PLC_1 MODE BUFF" = 1) AND ("MODE SELECTION DB"."UF PLC_1 PROCESS BUFF" = 415) AND "INPUT MAPPING DB"."ABFV-208 FEED BACK OPEN" AND "INPUT MAPPING DB"."ABFV-207 FEED BACK OPEN" AND "INPUT MAPPING DB"."ABFV 204 FEED BACK OPEN" AND "INPUT MAPPING DB"."ABFV 203 FEED BACK OPEN" AND "INPUT MAPPING DB"."ABFV 202 FEED BACK CLOSE",
                      "PRESENT VALUE OF TIME" => "CEB_1 DB".PV."CEB BACKWASH_1");
   "TIMING_SECS_DB_7".RESET := ("MODE SELECTION DB"."UF PLC_1 MODE BUFF" = 1) AND ("MODE SELECTION DB"."UF PLC_1 PROCESS BUFF" = 415) AND "TIMING_SECS_DB_7".DONE;
   IF "TIMING_SECS_DB_7".RESET THEN "MODE SELECTION DB"."UF PLC_1 PROCESS BUFF" := 420; END_IF;
   "IEC_Timer_0_DB_62".TON(IN := ("MODE SELECTION DB"."UF PLC_1 MODE BUFF" = 1) AND ("MODE SELECTION DB"."UF PLC_1 PROCESS BUFF" = 420),
                           PT := T#5S);
   IF "IEC_Timer_0_DB_62".Q THEN "MODE SELECTION DB"."UF PLC_1 PROCESS BUFF" := 425; END_IF;
END_REGION

REGION Network 16: ABFV 208 CLOSE FB
   RUNG wire#powerrail
      { S7_Templates := "SrcType := Int" } EQ_Contact(in1 := "MODE SELECTION DB"."UF PLC_1 MODE BUFF", in2 := 1)
      { S7_Templates := "SrcType := Int" } EQ_Contact(in1 := "MODE SELECTION DB"."UF PLC_1 PROCESS BUFF", in2 := 425)
      Move(in := 430, out1 => "MODE SELECTION DB"."UF PLC_1 PROCESS BUFF")
   END_RUNG
   // the same network as SCL:
   IF ("MODE SELECTION DB"."UF PLC_1 MODE BUFF" = 1) AND ("MODE SELECTION DB"."UF PLC_1 PROCESS BUFF" = 425) THEN
       "MODE SELECTION DB"."UF PLC_1 PROCESS BUFF" := 430;
   END_IF;
END_REGION

REGION Network 17: ABFV 207 CLOSE FB
   RUNG wire#powerrail
      { S7_Templates := "SrcType := Int" } EQ_Contact(in1 := "MODE SELECTION DB"."UF PLC_1 MODE BUFF", in2 := 1)
      { S7_Templates := "SrcType := Int" } EQ_Contact(in1 := "MODE SELECTION DB"."UF PLC_1 PROCESS BUFF", in2 := 430)
      Move(in := 435, out1 => "MODE SELECTION DB"."UF PLC_1 PROCESS BUFF")
   END_RUNG
   // the same network as SCL:
   IF ("MODE SELECTION DB"."UF PLC_1 MODE BUFF" = 1) AND ("MODE SELECTION DB"."UF PLC_1 PROCESS BUFF" = 430) THEN
       "MODE SELECTION DB"."UF PLC_1 PROCESS BUFF" := 435;
   END_IF;
END_REGION

REGION Network 18: ABFV 204 CLOSE FB
   RUNG wire#powerrail
      { S7_Templates := "SrcType := Int" } EQ_Contact(in1 := "MODE SELECTION DB"."UF PLC_1 MODE BUFF", in2 := 1)
      { S7_Templates := "SrcType := Int" } EQ_Contact(in1 := "MODE SELECTION DB"."UF PLC_1 PROCESS BUFF", in2 := 435)
      Move(in := 440, out1 => "MODE SELECTION DB"."UF PLC_1 PROCESS BUFF")
   END_RUNG
   // the same network as SCL:
   IF ("MODE SELECTION DB"."UF PLC_1 MODE BUFF" = 1) AND ("MODE SELECTION DB"."UF PLC_1 PROCESS BUFF" = 435) THEN
       "MODE SELECTION DB"."UF PLC_1 PROCESS BUFF" := 440;
   END_IF;
END_REGION

REGION Network 19: ABFV 203 CLOSE FB
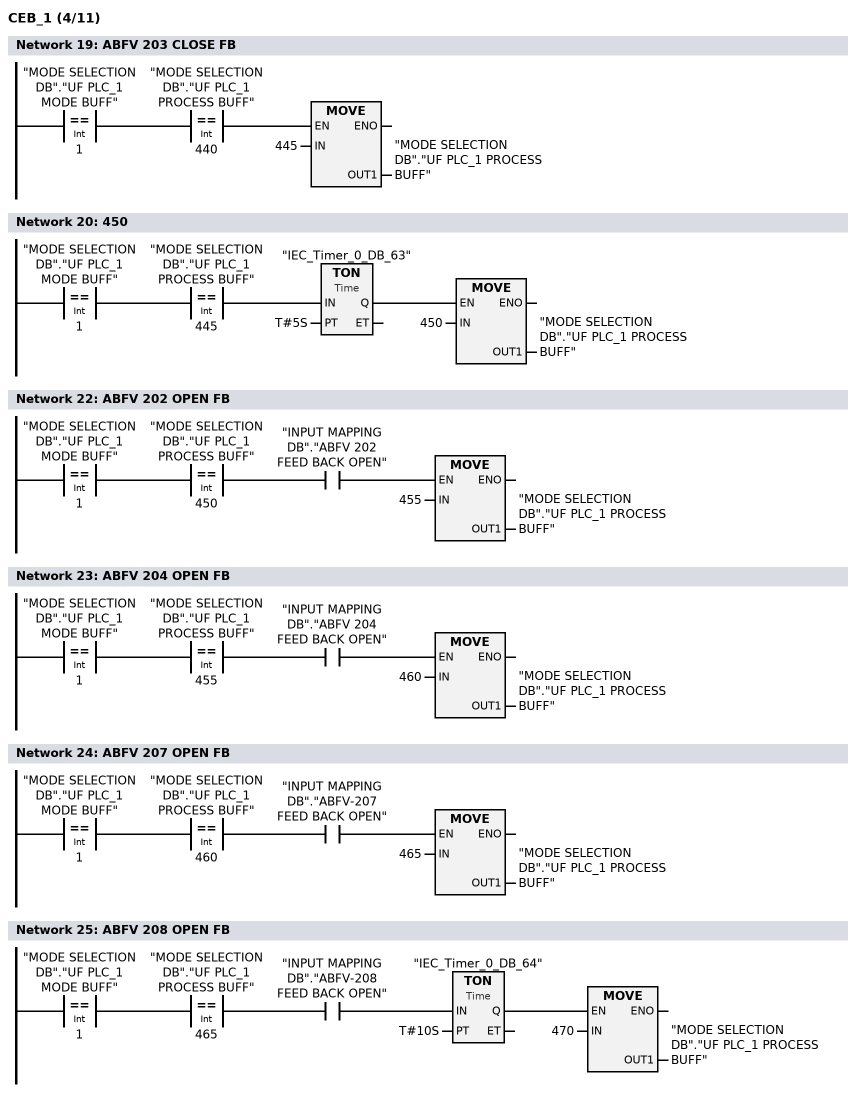
   RUNG wire#powerrail
      { S7_Templates := "SrcType := Int" } EQ_Contact(in1 := "MODE SELECTION DB"."UF PLC_1 MODE BUFF", in2 := 1)
      { S7_Templates := "SrcType := Int" } EQ_Contact(in1 := "MODE SELECTION DB"."UF PLC_1 PROCESS BUFF", in2 := 440)
      Move(in := 445, out1 => "MODE SELECTION DB"."UF PLC_1 PROCESS BUFF")
   END_RUNG
   // the same network as SCL:
   IF ("MODE SELECTION DB"."UF PLC_1 MODE BUFF" = 1) AND ("MODE SELECTION DB"."UF PLC_1 PROCESS BUFF" = 440) THEN
       "MODE SELECTION DB"."UF PLC_1 PROCESS BUFF" := 445;
   END_IF;
END_REGION

REGION Network 20: 450
   RUNG wire#powerrail
      { S7_Templates := "SrcType := Int" } EQ_Contact(in1 := "MODE SELECTION DB"."UF PLC_1 MODE BUFF", in2 := 1)
      { S7_Templates := "SrcType := Int" } EQ_Contact(in1 := "MODE SELECTION DB"."UF PLC_1 PROCESS BUFF", in2 := 445)
      { S7_Templates := "time_type := Time" } "IEC_Timer_0_DB_63".TON(pt := T#5S, et =>)
      Move(in := 450, out1 => "MODE SELECTION DB"."UF PLC_1 PROCESS BUFF")
   END_RUNG
   // the same network as SCL:
   "IEC_Timer_0_DB_63".TON(IN := ("MODE SELECTION DB"."UF PLC_1 MODE BUFF" = 1) AND ("MODE SELECTION DB"."UF PLC_1 PROCESS BUFF" = 445),
                           PT := T#5S);
   IF "IEC_Timer_0_DB_63".Q THEN "MODE SELECTION DB"."UF PLC_1 PROCESS BUFF" := 450; END_IF;
END_REGION

REGION Network 22: ABFV 202 OPEN FB
   RUNG wire#powerrail
      { S7_Templates := "SrcType := Int" } EQ_Contact(in1 := "MODE SELECTION DB"."UF PLC_1 MODE BUFF", in2 := 1)
      { S7_Templates := "SrcType := Int" } EQ_Contact(in1 := "MODE SELECTION DB"."UF PLC_1 PROCESS BUFF", in2 := 450)
      Contact( "INPUT MAPPING DB"."ABFV 202 FEED BACK OPEN" )
      Move(in := 455, out1 => "MODE SELECTION DB"."UF PLC_1 PROCESS BUFF")
   END_RUNG
   // the same network as SCL:
   IF ("MODE SELECTION DB"."UF PLC_1 MODE BUFF" = 1) AND ("MODE SELECTION DB"."UF PLC_1 PROCESS BUFF" = 450) AND "INPUT MAPPING DB"."ABFV 202 FEED BACK OPEN" THEN
       "MODE SELECTION DB"."UF PLC_1 PROCESS BUFF" := 455;
   END_IF;
END_REGION

REGION Network 23: ABFV 204 OPEN FB
   RUNG wire#powerrail
      { S7_Templates := "SrcType := Int" } EQ_Contact(in1 := "MODE SELECTION DB"."UF PLC_1 MODE BUFF", in2 := 1)
      { S7_Templates := "SrcType := Int" } EQ_Contact(in1 := "MODE SELECTION DB"."UF PLC_1 PROCESS BUFF", in2 := 455)
      Contact( "INPUT MAPPING DB"."ABFV 204 FEED BACK OPEN" )
      Move(in := 460, out1 => "MODE SELECTION DB"."UF PLC_1 PROCESS BUFF")
   END_RUNG
   // the same network as SCL:
   IF ("MODE SELECTION DB"."UF PLC_1 MODE BUFF" = 1) AND ("MODE SELECTION DB"."UF PLC_1 PROCESS BUFF" = 455) AND "INPUT MAPPING DB"."ABFV 204 FEED BACK OPEN" THEN
       "MODE SELECTION DB"."UF PLC_1 PROCESS BUFF" := 460;
   END_IF;
END_REGION

REGION Network 24: ABFV 207 OPEN FB
   RUNG wire#powerrail
      { S7_Templates := "SrcType := Int" } EQ_Contact(in1 := "MODE SELECTION DB"."UF PLC_1 MODE BUFF", in2 := 1)
      { S7_Templates := "SrcType := Int" } EQ_Contact(in1 := "MODE SELECTION DB"."UF PLC_1 PROCESS BUFF", in2 := 460)
      Contact( "INPUT MAPPING DB"."ABFV-207 FEED BACK OPEN" )
      Move(in := 465, out1 => "MODE SELECTION DB"."UF PLC_1 PROCESS BUFF")
   END_RUNG
   // the same network as SCL:
   IF ("MODE SELECTION DB"."UF PLC_1 MODE BUFF" = 1) AND ("MODE SELECTION DB"."UF PLC_1 PROCESS BUFF" = 460) AND "INPUT MAPPING DB"."ABFV-207 FEED BACK OPEN" THEN
       "MODE SELECTION DB"."UF PLC_1 PROCESS BUFF" := 465;
   END_IF;
END_REGION

REGION Network 25: ABFV 208 OPEN FB
   RUNG wire#powerrail
      { S7_Templates := "SrcType := Int" } EQ_Contact(in1 := "MODE SELECTION DB"."UF PLC_1 MODE BUFF", in2 := 1)
      { S7_Templates := "SrcType := Int" } EQ_Contact(in1 := "MODE SELECTION DB"."UF PLC_1 PROCESS BUFF", in2 := 465)
      Contact( "INPUT MAPPING DB"."ABFV-208 FEED BACK OPEN" )
      { S7_Templates := "time_type := Time" } "IEC_Timer_0_DB_64".TON(pt := T#10S, et =>)
      Move(in := 470, out1 => "MODE SELECTION DB"."UF PLC_1 PROCESS BUFF")
   END_RUNG
   // the same network as SCL:
   "IEC_Timer_0_DB_64".TON(IN := ("MODE SELECTION DB"."UF PLC_1 MODE BUFF" = 1) AND ("MODE SELECTION DB"."UF PLC_1 PROCESS BUFF" = 465) AND "INPUT MAPPING DB"."ABFV-208 FEED BACK OPEN",
                           PT := T#10S);
   IF "IEC_Timer_0_DB_64".Q THEN "MODE SELECTION DB"."UF PLC_1 PROCESS BUFF" := 470; END_IF;
END_REGION

REGION Network 26: CEB BACKWASH_2
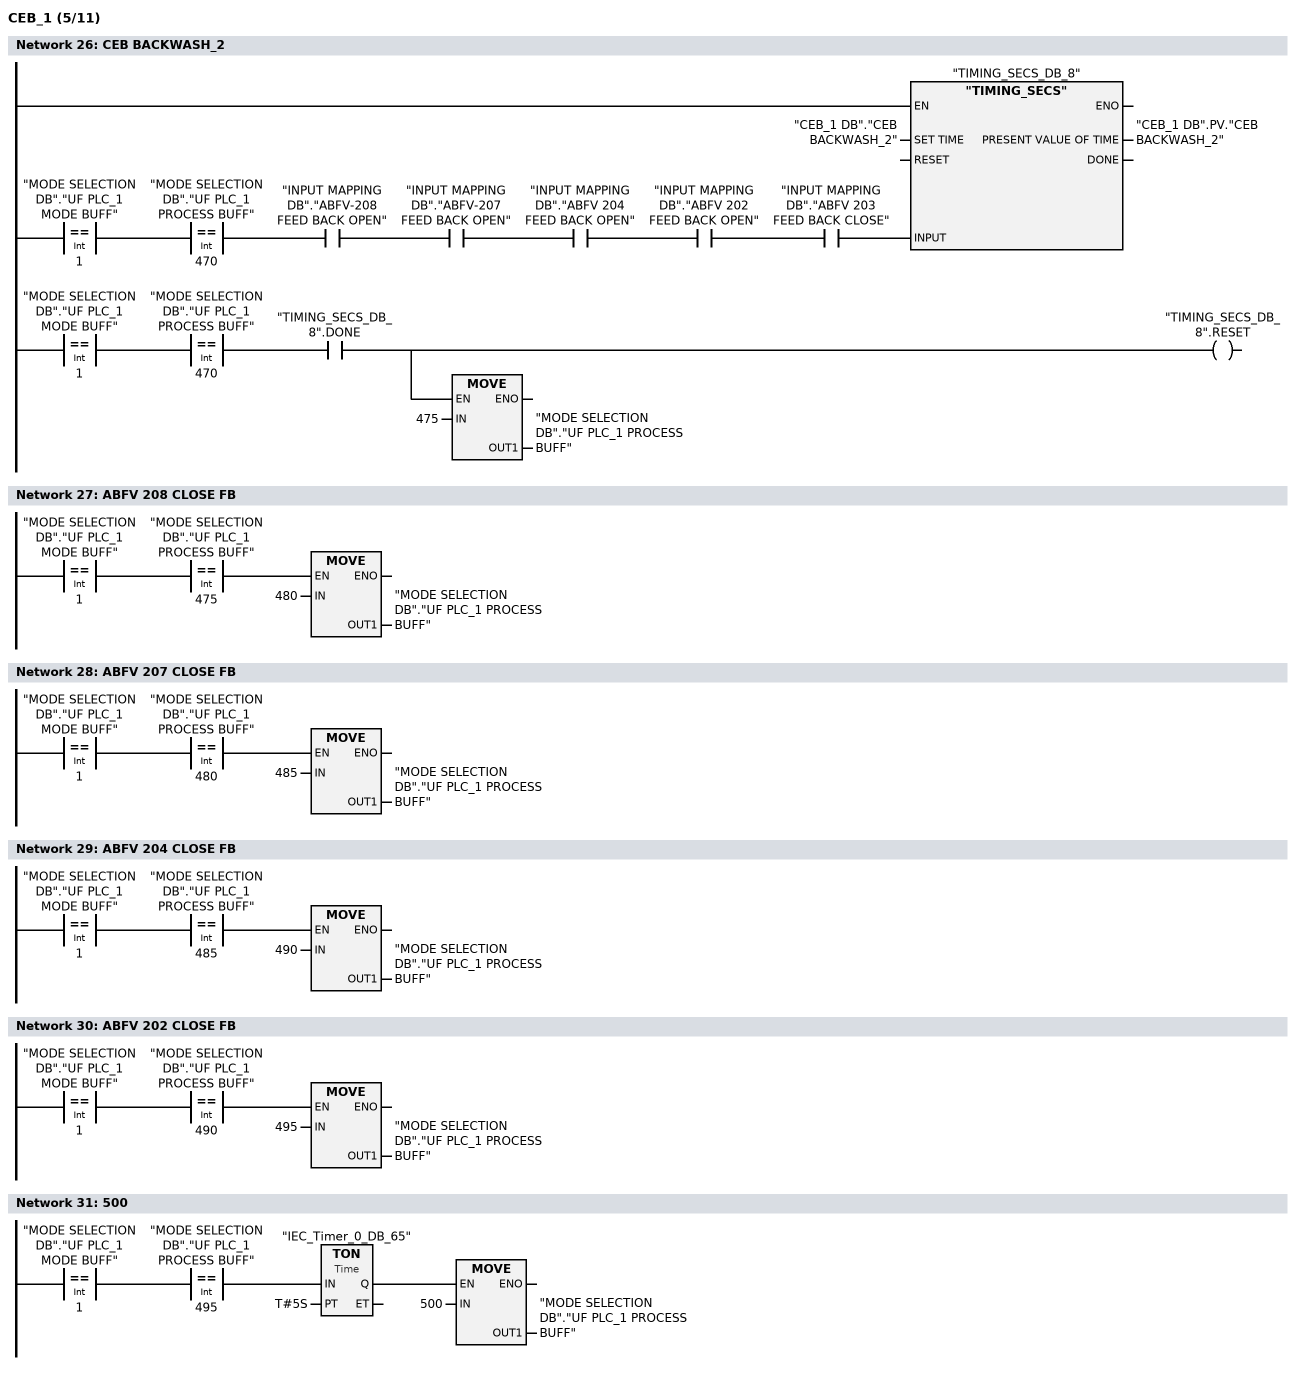
   RUNG wire#powerrail
      "TIMING_SECS_DB_8"(INPUT := wire#w1, "SET TIME" := "CEB_1 DB"."CEB BACKWASH_2", RESET :=, "PRESENT VALUE OF TIME" => "CEB_1 DB".PV."CEB BACKWASH_2", DONE =>)
   END_RUNG
   RUNG wire#powerrail
      { S7_Templates := "SrcType := Int" } EQ_Contact(in1 := "MODE SELECTION DB"."UF PLC_1 MODE BUFF", in2 := 1)
      { S7_Templates := "SrcType := Int" } EQ_Contact(in1 := "MODE SELECTION DB"."UF PLC_1 PROCESS BUFF", in2 := 470)
      Contact( "INPUT MAPPING DB"."ABFV-208 FEED BACK OPEN" )
      Contact( "INPUT MAPPING DB"."ABFV-207 FEED BACK OPEN" )
      Contact( "INPUT MAPPING DB"."ABFV 204 FEED BACK OPEN" )
      Contact( "INPUT MAPPING DB"."ABFV 202 FEED BACK OPEN" )
      Contact( "INPUT MAPPING DB"."ABFV 203 FEED BACK CLOSE" )
   END_RUNG wire#w1
   RUNG wire#powerrail
      { S7_Templates := "SrcType := Int" } EQ_Contact(in1 := "MODE SELECTION DB"."UF PLC_1 MODE BUFF", in2 := 1)
      { S7_Templates := "SrcType := Int" } EQ_Contact(in1 := "MODE SELECTION DB"."UF PLC_1 PROCESS BUFF", in2 := 470)
      Contact( "TIMING_SECS_DB_8".DONE )
      wire#w2
      Coil( "TIMING_SECS_DB_8".RESET )
   END_RUNG
   RUNG wire#w2
      Move(in := 475, out1 => "MODE SELECTION DB"."UF PLC_1 PROCESS BUFF")
   END_RUNG
   // the same network as SCL:
   "TIMING_SECS_DB_8"("SET TIME" := "CEB_1 DB"."CEB BACKWASH_2",   // "TIMING_SECS"
                      INPUT := ("MODE SELECTION DB"."UF PLC_1 MODE BUFF" = 1) AND ("MODE SELECTION DB"."UF PLC_1 PROCESS BUFF" = 470) AND "INPUT MAPPING DB"."ABFV-208 FEED BACK OPEN" AND "INPUT MAPPING DB"."ABFV-207 FEED BACK OPEN" AND "INPUT MAPPING DB"."ABFV 204 FEED BACK OPEN" AND "INPUT MAPPING DB"."ABFV 202 FEED BACK OPEN" AND "INPUT MAPPING DB"."ABFV 203 FEED BACK CLOSE",
                      "PRESENT VALUE OF TIME" => "CEB_1 DB".PV."CEB BACKWASH_2");
   "TIMING_SECS_DB_8".RESET := ("MODE SELECTION DB"."UF PLC_1 MODE BUFF" = 1) AND ("MODE SELECTION DB"."UF PLC_1 PROCESS BUFF" = 470) AND "TIMING_SECS_DB_8".DONE;
   IF "TIMING_SECS_DB_8".RESET THEN "MODE SELECTION DB"."UF PLC_1 PROCESS BUFF" := 475; END_IF;
END_REGION

REGION Network 27: ABFV 208 CLOSE FB
   RUNG wire#powerrail
      { S7_Templates := "SrcType := Int" } EQ_Contact(in1 := "MODE SELECTION DB"."UF PLC_1 MODE BUFF", in2 := 1)
      { S7_Templates := "SrcType := Int" } EQ_Contact(in1 := "MODE SELECTION DB"."UF PLC_1 PROCESS BUFF", in2 := 475)
      Move(in := 480, out1 => "MODE SELECTION DB"."UF PLC_1 PROCESS BUFF")
   END_RUNG
   // the same network as SCL:
   IF ("MODE SELECTION DB"."UF PLC_1 MODE BUFF" = 1) AND ("MODE SELECTION DB"."UF PLC_1 PROCESS BUFF" = 475) THEN
       "MODE SELECTION DB"."UF PLC_1 PROCESS BUFF" := 480;
   END_IF;
END_REGION

REGION Network 28: ABFV 207 CLOSE FB
   RUNG wire#powerrail
      { S7_Templates := "SrcType := Int" } EQ_Contact(in1 := "MODE SELECTION DB"."UF PLC_1 MODE BUFF", in2 := 1)
      { S7_Templates := "SrcType := Int" } EQ_Contact(in1 := "MODE SELECTION DB"."UF PLC_1 PROCESS BUFF", in2 := 480)
      Move(in := 485, out1 => "MODE SELECTION DB"."UF PLC_1 PROCESS BUFF")
   END_RUNG
   // the same network as SCL:
   IF ("MODE SELECTION DB"."UF PLC_1 MODE BUFF" = 1) AND ("MODE SELECTION DB"."UF PLC_1 PROCESS BUFF" = 480) THEN
       "MODE SELECTION DB"."UF PLC_1 PROCESS BUFF" := 485;
   END_IF;
END_REGION

REGION Network 29: ABFV 204 CLOSE FB
   RUNG wire#powerrail
      { S7_Templates := "SrcType := Int" } EQ_Contact(in1 := "MODE SELECTION DB"."UF PLC_1 MODE BUFF", in2 := 1)
      { S7_Templates := "SrcType := Int" } EQ_Contact(in1 := "MODE SELECTION DB"."UF PLC_1 PROCESS BUFF", in2 := 485)
      Move(in := 490, out1 => "MODE SELECTION DB"."UF PLC_1 PROCESS BUFF")
   END_RUNG
   // the same network as SCL:
   IF ("MODE SELECTION DB"."UF PLC_1 MODE BUFF" = 1) AND ("MODE SELECTION DB"."UF PLC_1 PROCESS BUFF" = 485) THEN
       "MODE SELECTION DB"."UF PLC_1 PROCESS BUFF" := 490;
   END_IF;
END_REGION

REGION Network 30: ABFV 202 CLOSE FB
   RUNG wire#powerrail
      { S7_Templates := "SrcType := Int" } EQ_Contact(in1 := "MODE SELECTION DB"."UF PLC_1 MODE BUFF", in2 := 1)
      { S7_Templates := "SrcType := Int" } EQ_Contact(in1 := "MODE SELECTION DB"."UF PLC_1 PROCESS BUFF", in2 := 490)
      Move(in := 495, out1 => "MODE SELECTION DB"."UF PLC_1 PROCESS BUFF")
   END_RUNG
   // the same network as SCL:
   IF ("MODE SELECTION DB"."UF PLC_1 MODE BUFF" = 1) AND ("MODE SELECTION DB"."UF PLC_1 PROCESS BUFF" = 490) THEN
       "MODE SELECTION DB"."UF PLC_1 PROCESS BUFF" := 495;
   END_IF;
END_REGION

REGION Network 31: 500
   RUNG wire#powerrail
      { S7_Templates := "SrcType := Int" } EQ_Contact(in1 := "MODE SELECTION DB"."UF PLC_1 MODE BUFF", in2 := 1)
      { S7_Templates := "SrcType := Int" } EQ_Contact(in1 := "MODE SELECTION DB"."UF PLC_1 PROCESS BUFF", in2 := 495)
      { S7_Templates := "time_type := Time" } "IEC_Timer_0_DB_65".TON(pt := T#5S, et =>)
      Move(in := 500, out1 => "MODE SELECTION DB"."UF PLC_1 PROCESS BUFF")
   END_RUNG
   // the same network as SCL:
   "IEC_Timer_0_DB_65".TON(IN := ("MODE SELECTION DB"."UF PLC_1 MODE BUFF" = 1) AND ("MODE SELECTION DB"."UF PLC_1 PROCESS BUFF" = 495),
                           PT := T#5S);
   IF "IEC_Timer_0_DB_65".Q THEN "MODE SELECTION DB"."UF PLC_1 PROCESS BUFF" := 500; END_IF;
END_REGION

REGION Network 33: SOAK
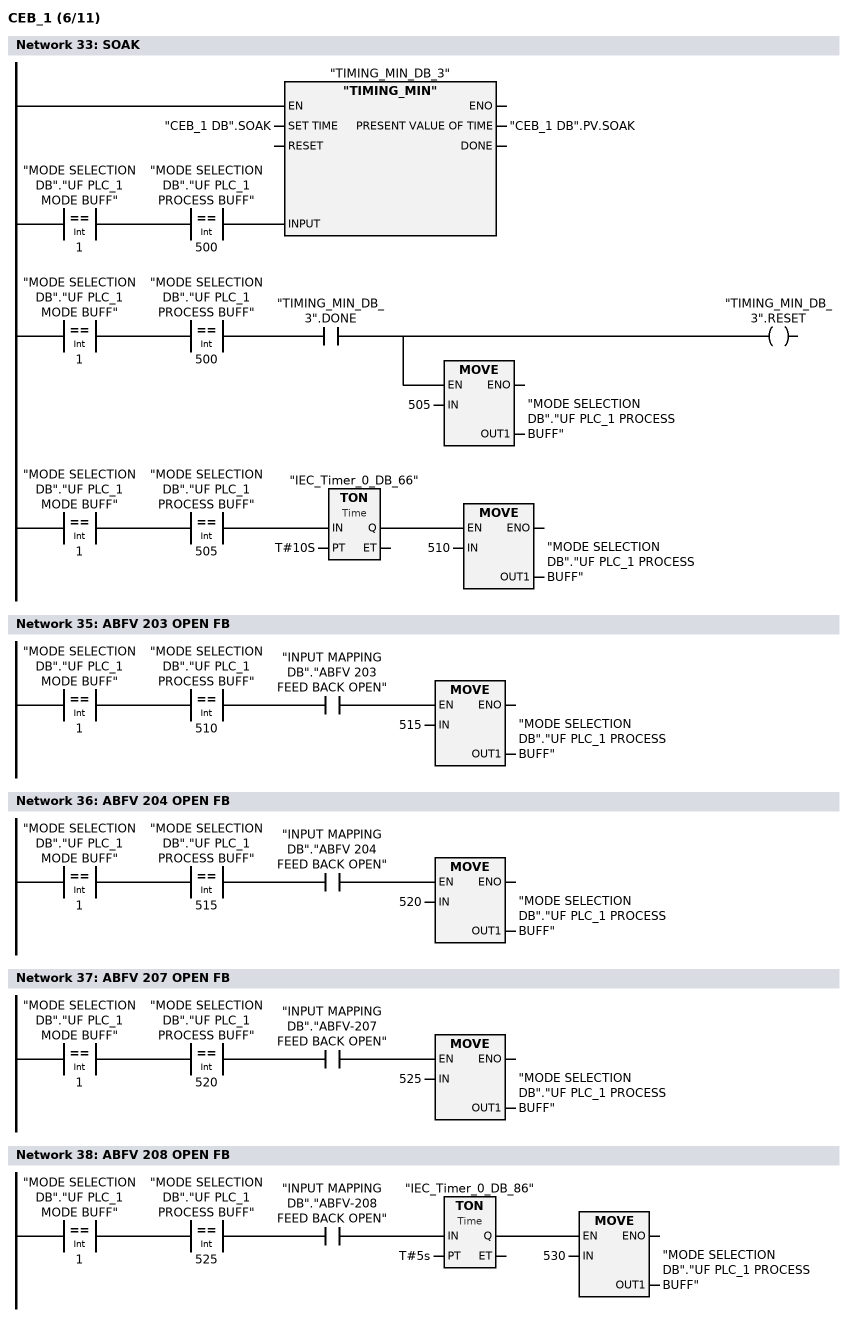
   RUNG wire#powerrail
      "TIMING_MIN_DB_3"(INPUT := wire#w1, "SET TIME" := "CEB_1 DB".SOAK, RESET :=, "PRESENT VALUE OF TIME" => "CEB_1 DB".PV.SOAK, DONE =>)
   END_RUNG
   RUNG wire#powerrail
      { S7_Templates := "SrcType := Int" } EQ_Contact(in1 := "MODE SELECTION DB"."UF PLC_1 MODE BUFF", in2 := 1)
      { S7_Templates := "SrcType := Int" } EQ_Contact(in1 := "MODE SELECTION DB"."UF PLC_1 PROCESS BUFF", in2 := 500)
   END_RUNG wire#w1
   RUNG wire#powerrail
      { S7_Templates := "SrcType := Int" } EQ_Contact(in1 := "MODE SELECTION DB"."UF PLC_1 MODE BUFF", in2 := 1)
      { S7_Templates := "SrcType := Int" } EQ_Contact(in1 := "MODE SELECTION DB"."UF PLC_1 PROCESS BUFF", in2 := 500)
      Contact( "TIMING_MIN_DB_3".DONE )
      wire#w2
      Coil( "TIMING_MIN_DB_3".RESET )
   END_RUNG
   RUNG wire#w2
      Move(in := 505, out1 => "MODE SELECTION DB"."UF PLC_1 PROCESS BUFF")
   END_RUNG
   RUNG wire#powerrail
      { S7_Templates := "SrcType := Int" } EQ_Contact(in1 := "MODE SELECTION DB"."UF PLC_1 MODE BUFF", in2 := 1)
      { S7_Templates := "SrcType := Int" } EQ_Contact(in1 := "MODE SELECTION DB"."UF PLC_1 PROCESS BUFF", in2 := 505)
      { S7_Templates := "time_type := Time" } "IEC_Timer_0_DB_66".TON(pt := T#10S, et =>)
      Move(in := 510, out1 => "MODE SELECTION DB"."UF PLC_1 PROCESS BUFF")
   END_RUNG
   // the same network as SCL:
   "TIMING_MIN_DB_3"("SET TIME" := "CEB_1 DB".SOAK,   // "TIMING_MIN"
                     INPUT := ("MODE SELECTION DB"."UF PLC_1 MODE BUFF" = 1) AND ("MODE SELECTION DB"."UF PLC_1 PROCESS BUFF" = 500),
                     "PRESENT VALUE OF TIME" => "CEB_1 DB".PV.SOAK);
   "TIMING_MIN_DB_3".RESET := ("MODE SELECTION DB"."UF PLC_1 MODE BUFF" = 1) AND ("MODE SELECTION DB"."UF PLC_1 PROCESS BUFF" = 500) AND "TIMING_MIN_DB_3".DONE;
   IF "TIMING_MIN_DB_3".RESET THEN "MODE SELECTION DB"."UF PLC_1 PROCESS BUFF" := 505; END_IF;
   "IEC_Timer_0_DB_66".TON(IN := ("MODE SELECTION DB"."UF PLC_1 MODE BUFF" = 1) AND ("MODE SELECTION DB"."UF PLC_1 PROCESS BUFF" = 505),
                           PT := T#10S);
   IF "IEC_Timer_0_DB_66".Q THEN "MODE SELECTION DB"."UF PLC_1 PROCESS BUFF" := 510; END_IF;
END_REGION

REGION Network 35: ABFV 203 OPEN FB
   RUNG wire#powerrail
      { S7_Templates := "SrcType := Int" } EQ_Contact(in1 := "MODE SELECTION DB"."UF PLC_1 MODE BUFF", in2 := 1)
      { S7_Templates := "SrcType := Int" } EQ_Contact(in1 := "MODE SELECTION DB"."UF PLC_1 PROCESS BUFF", in2 := 510)
      Contact( "INPUT MAPPING DB"."ABFV 203 FEED BACK OPEN" )
      Move(in := 515, out1 => "MODE SELECTION DB"."UF PLC_1 PROCESS BUFF")
   END_RUNG
   // the same network as SCL:
   IF ("MODE SELECTION DB"."UF PLC_1 MODE BUFF" = 1) AND ("MODE SELECTION DB"."UF PLC_1 PROCESS BUFF" = 510) AND "INPUT MAPPING DB"."ABFV 203 FEED BACK OPEN" THEN
       "MODE SELECTION DB"."UF PLC_1 PROCESS BUFF" := 515;
   END_IF;
END_REGION

REGION Network 36: ABFV 204 OPEN FB
   RUNG wire#powerrail
      { S7_Templates := "SrcType := Int" } EQ_Contact(in1 := "MODE SELECTION DB"."UF PLC_1 MODE BUFF", in2 := 1)
      { S7_Templates := "SrcType := Int" } EQ_Contact(in1 := "MODE SELECTION DB"."UF PLC_1 PROCESS BUFF", in2 := 515)
      Contact( "INPUT MAPPING DB"."ABFV 204 FEED BACK OPEN" )
      Move(in := 520, out1 => "MODE SELECTION DB"."UF PLC_1 PROCESS BUFF")
   END_RUNG
   // the same network as SCL:
   IF ("MODE SELECTION DB"."UF PLC_1 MODE BUFF" = 1) AND ("MODE SELECTION DB"."UF PLC_1 PROCESS BUFF" = 515) AND "INPUT MAPPING DB"."ABFV 204 FEED BACK OPEN" THEN
       "MODE SELECTION DB"."UF PLC_1 PROCESS BUFF" := 520;
   END_IF;
END_REGION

REGION Network 37: ABFV 207 OPEN FB
   RUNG wire#powerrail
      { S7_Templates := "SrcType := Int" } EQ_Contact(in1 := "MODE SELECTION DB"."UF PLC_1 MODE BUFF", in2 := 1)
      { S7_Templates := "SrcType := Int" } EQ_Contact(in1 := "MODE SELECTION DB"."UF PLC_1 PROCESS BUFF", in2 := 520)
      Contact( "INPUT MAPPING DB"."ABFV-207 FEED BACK OPEN" )
      Move(in := 525, out1 => "MODE SELECTION DB"."UF PLC_1 PROCESS BUFF")
   END_RUNG
   // the same network as SCL:
   IF ("MODE SELECTION DB"."UF PLC_1 MODE BUFF" = 1) AND ("MODE SELECTION DB"."UF PLC_1 PROCESS BUFF" = 520) AND "INPUT MAPPING DB"."ABFV-207 FEED BACK OPEN" THEN
       "MODE SELECTION DB"."UF PLC_1 PROCESS BUFF" := 525;
   END_IF;
END_REGION

REGION Network 38: ABFV 208 OPEN FB
   RUNG wire#powerrail
      { S7_Templates := "SrcType := Int" } EQ_Contact(in1 := "MODE SELECTION DB"."UF PLC_1 MODE BUFF", in2 := 1)
      { S7_Templates := "SrcType := Int" } EQ_Contact(in1 := "MODE SELECTION DB"."UF PLC_1 PROCESS BUFF", in2 := 525)
      Contact( "INPUT MAPPING DB"."ABFV-208 FEED BACK OPEN" )
      { S7_Templates := "time_type := Time" } "IEC_Timer_0_DB_86".TON(pt := T#5s, et =>)
      Move(in := 530, out1 => "MODE SELECTION DB"."UF PLC_1 PROCESS BUFF")
   END_RUNG
   // the same network as SCL:
   "IEC_Timer_0_DB_86".TON(IN := ("MODE SELECTION DB"."UF PLC_1 MODE BUFF" = 1) AND ("MODE SELECTION DB"."UF PLC_1 PROCESS BUFF" = 525) AND "INPUT MAPPING DB"."ABFV-208 FEED BACK OPEN",
                           PT := T#5s);
   IF "IEC_Timer_0_DB_86".Q THEN "MODE SELECTION DB"."UF PLC_1 PROCESS BUFF" := 530; END_IF;
END_REGION

REGION Network 39: BACKWASH_1
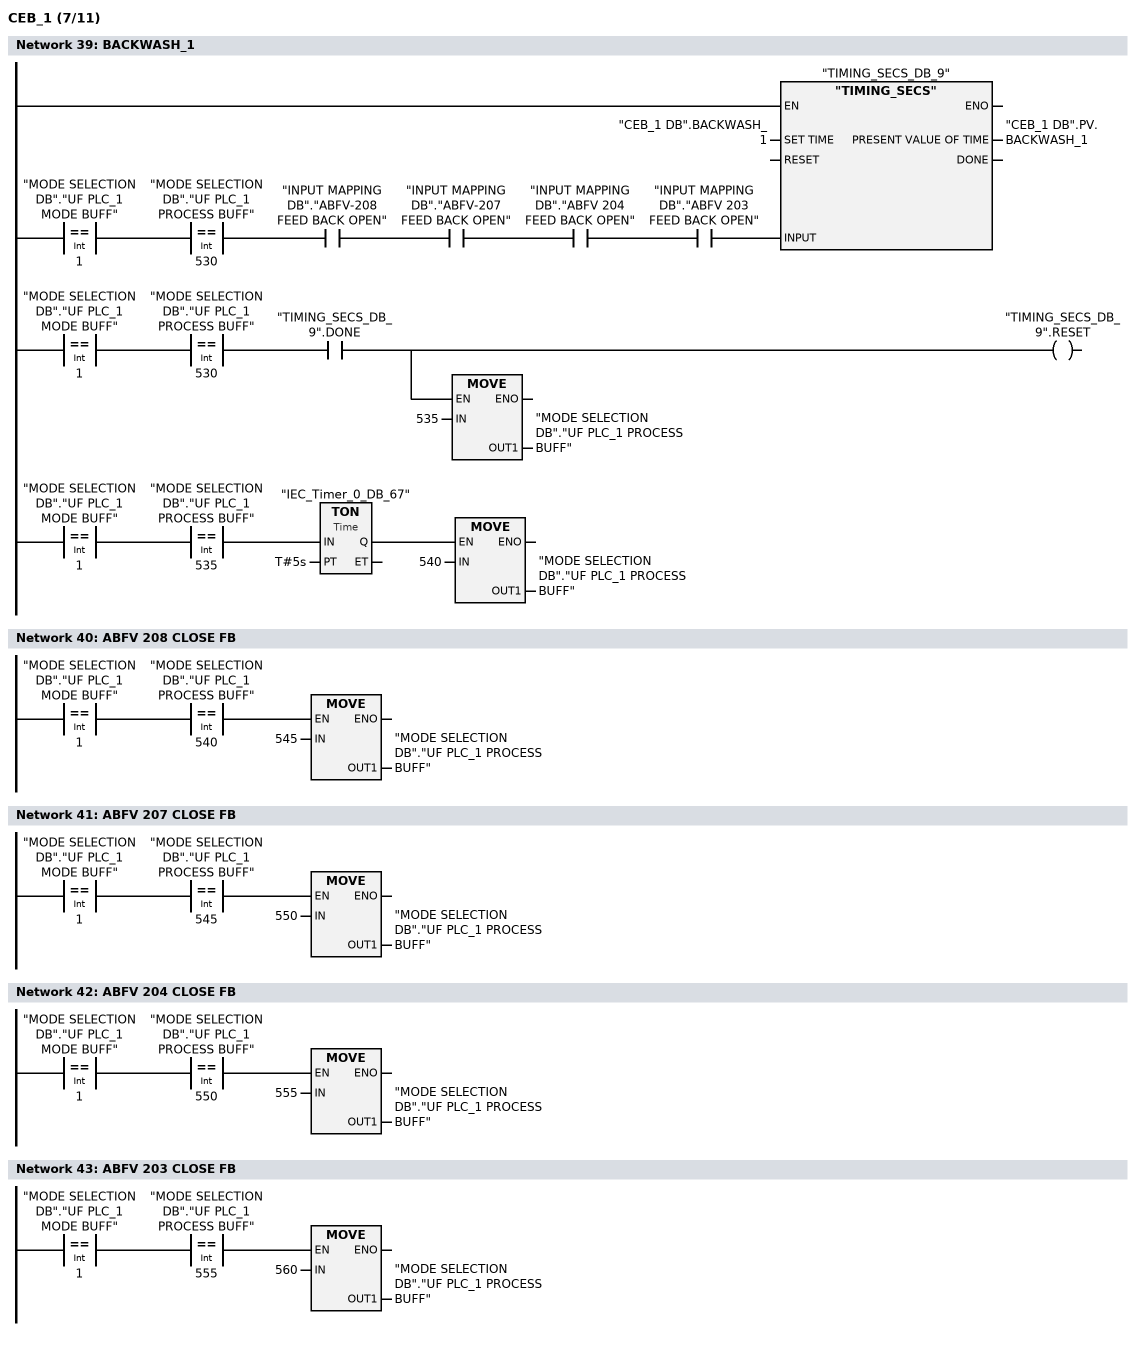
   RUNG wire#powerrail
      "TIMING_SECS_DB_9"(INPUT := wire#w1, "SET TIME" := "CEB_1 DB".BACKWASH_1, RESET :=, "PRESENT VALUE OF TIME" => "CEB_1 DB".PV.BACKWASH_1, DONE =>)
   END_RUNG
   RUNG wire#powerrail
      { S7_Templates := "SrcType := Int" } EQ_Contact(in1 := "MODE SELECTION DB"."UF PLC_1 MODE BUFF", in2 := 1)
      { S7_Templates := "SrcType := Int" } EQ_Contact(in1 := "MODE SELECTION DB"."UF PLC_1 PROCESS BUFF", in2 := 530)
      Contact( "INPUT MAPPING DB"."ABFV-208 FEED BACK OPEN" )
      Contact( "INPUT MAPPING DB"."ABFV-207 FEED BACK OPEN" )
      Contact( "INPUT MAPPING DB"."ABFV 204 FEED BACK OPEN" )
      Contact( "INPUT MAPPING DB"."ABFV 203 FEED BACK OPEN" )
   END_RUNG wire#w1
   RUNG wire#powerrail
      { S7_Templates := "SrcType := Int" } EQ_Contact(in1 := "MODE SELECTION DB"."UF PLC_1 MODE BUFF", in2 := 1)
      { S7_Templates := "SrcType := Int" } EQ_Contact(in1 := "MODE SELECTION DB"."UF PLC_1 PROCESS BUFF", in2 := 530)
      Contact( "TIMING_SECS_DB_9".DONE )
      wire#w2
      Coil( "TIMING_SECS_DB_9".RESET )
   END_RUNG
   RUNG wire#w2
      Move(in := 535, out1 => "MODE SELECTION DB"."UF PLC_1 PROCESS BUFF")
   END_RUNG
   RUNG wire#powerrail
      { S7_Templates := "SrcType := Int" } EQ_Contact(in1 := "MODE SELECTION DB"."UF PLC_1 MODE BUFF", in2 := 1)
      { S7_Templates := "SrcType := Int" } EQ_Contact(in1 := "MODE SELECTION DB"."UF PLC_1 PROCESS BUFF", in2 := 535)
      { S7_Templates := "time_type := Time" } "IEC_Timer_0_DB_67".TON(pt := T#5s, et =>)
      Move(in := 540, out1 => "MODE SELECTION DB"."UF PLC_1 PROCESS BUFF")
   END_RUNG
   // the same network as SCL:
   "TIMING_SECS_DB_9"("SET TIME" := "CEB_1 DB".BACKWASH_1,   // "TIMING_SECS"
                      INPUT := ("MODE SELECTION DB"."UF PLC_1 MODE BUFF" = 1) AND ("MODE SELECTION DB"."UF PLC_1 PROCESS BUFF" = 530) AND "INPUT MAPPING DB"."ABFV-208 FEED BACK OPEN" AND "INPUT MAPPING DB"."ABFV-207 FEED BACK OPEN" AND "INPUT MAPPING DB"."ABFV 204 FEED BACK OPEN" AND "INPUT MAPPING DB"."ABFV 203 FEED BACK OPEN",
                      "PRESENT VALUE OF TIME" => "CEB_1 DB".PV.BACKWASH_1);
   "TIMING_SECS_DB_9".RESET := ("MODE SELECTION DB"."UF PLC_1 MODE BUFF" = 1) AND ("MODE SELECTION DB"."UF PLC_1 PROCESS BUFF" = 530) AND "TIMING_SECS_DB_9".DONE;
   IF "TIMING_SECS_DB_9".RESET THEN "MODE SELECTION DB"."UF PLC_1 PROCESS BUFF" := 535; END_IF;
   "IEC_Timer_0_DB_67".TON(IN := ("MODE SELECTION DB"."UF PLC_1 MODE BUFF" = 1) AND ("MODE SELECTION DB"."UF PLC_1 PROCESS BUFF" = 535),
                           PT := T#5s);
   IF "IEC_Timer_0_DB_67".Q THEN "MODE SELECTION DB"."UF PLC_1 PROCESS BUFF" := 540; END_IF;
END_REGION

REGION Network 40: ABFV 208 CLOSE FB
   RUNG wire#powerrail
      { S7_Templates := "SrcType := Int" } EQ_Contact(in1 := "MODE SELECTION DB"."UF PLC_1 MODE BUFF", in2 := 1)
      { S7_Templates := "SrcType := Int" } EQ_Contact(in1 := "MODE SELECTION DB"."UF PLC_1 PROCESS BUFF", in2 := 540)
      Move(in := 545, out1 => "MODE SELECTION DB"."UF PLC_1 PROCESS BUFF")
   END_RUNG
   // the same network as SCL:
   IF ("MODE SELECTION DB"."UF PLC_1 MODE BUFF" = 1) AND ("MODE SELECTION DB"."UF PLC_1 PROCESS BUFF" = 540) THEN
       "MODE SELECTION DB"."UF PLC_1 PROCESS BUFF" := 545;
   END_IF;
END_REGION

REGION Network 41: ABFV 207 CLOSE FB
   RUNG wire#powerrail
      { S7_Templates := "SrcType := Int" } EQ_Contact(in1 := "MODE SELECTION DB"."UF PLC_1 MODE BUFF", in2 := 1)
      { S7_Templates := "SrcType := Int" } EQ_Contact(in1 := "MODE SELECTION DB"."UF PLC_1 PROCESS BUFF", in2 := 545)
      Move(in := 550, out1 => "MODE SELECTION DB"."UF PLC_1 PROCESS BUFF")
   END_RUNG
   // the same network as SCL:
   IF ("MODE SELECTION DB"."UF PLC_1 MODE BUFF" = 1) AND ("MODE SELECTION DB"."UF PLC_1 PROCESS BUFF" = 545) THEN
       "MODE SELECTION DB"."UF PLC_1 PROCESS BUFF" := 550;
   END_IF;
END_REGION

REGION Network 42: ABFV 204 CLOSE FB
   RUNG wire#powerrail
      { S7_Templates := "SrcType := Int" } EQ_Contact(in1 := "MODE SELECTION DB"."UF PLC_1 MODE BUFF", in2 := 1)
      { S7_Templates := "SrcType := Int" } EQ_Contact(in1 := "MODE SELECTION DB"."UF PLC_1 PROCESS BUFF", in2 := 550)
      Move(in := 555, out1 => "MODE SELECTION DB"."UF PLC_1 PROCESS BUFF")
   END_RUNG
   // the same network as SCL:
   IF ("MODE SELECTION DB"."UF PLC_1 MODE BUFF" = 1) AND ("MODE SELECTION DB"."UF PLC_1 PROCESS BUFF" = 550) THEN
       "MODE SELECTION DB"."UF PLC_1 PROCESS BUFF" := 555;
   END_IF;
END_REGION

REGION Network 43: ABFV 203 CLOSE FB
   RUNG wire#powerrail
      { S7_Templates := "SrcType := Int" } EQ_Contact(in1 := "MODE SELECTION DB"."UF PLC_1 MODE BUFF", in2 := 1)
      { S7_Templates := "SrcType := Int" } EQ_Contact(in1 := "MODE SELECTION DB"."UF PLC_1 PROCESS BUFF", in2 := 555)
      Move(in := 560, out1 => "MODE SELECTION DB"."UF PLC_1 PROCESS BUFF")
   END_RUNG
   // the same network as SCL:
   IF ("MODE SELECTION DB"."UF PLC_1 MODE BUFF" = 1) AND ("MODE SELECTION DB"."UF PLC_1 PROCESS BUFF" = 555) THEN
       "MODE SELECTION DB"."UF PLC_1 PROCESS BUFF" := 560;
   END_IF;
END_REGION

REGION Network 44: 565
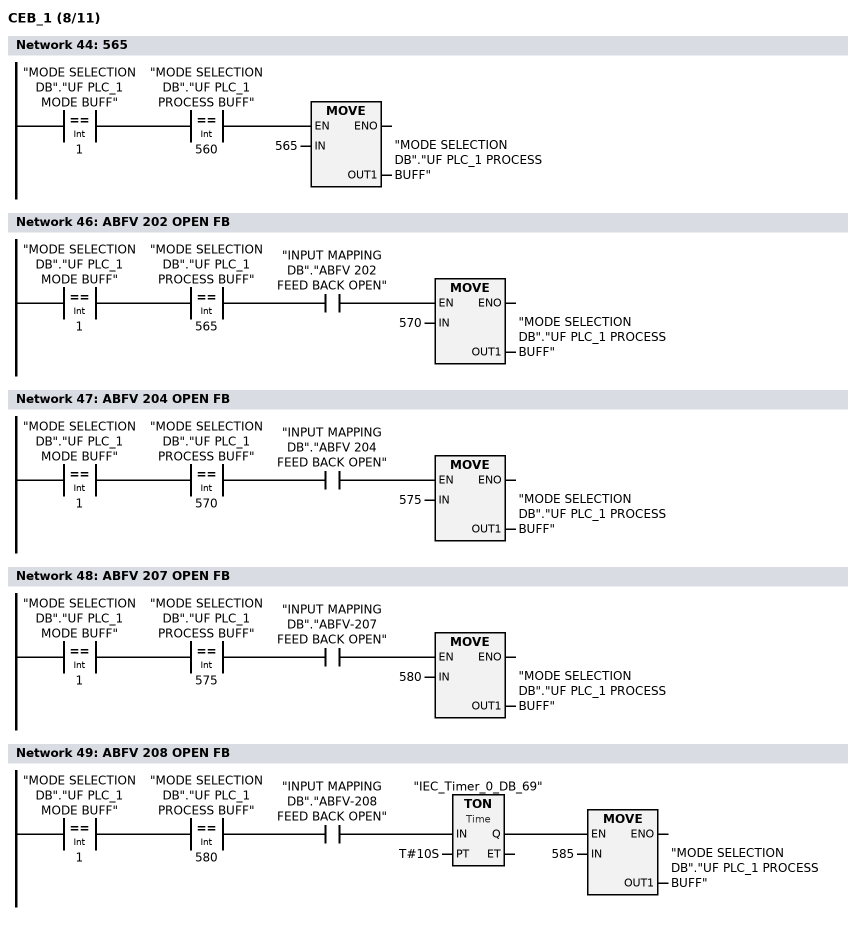
   RUNG wire#powerrail
      { S7_Templates := "SrcType := Int" } EQ_Contact(in1 := "MODE SELECTION DB"."UF PLC_1 MODE BUFF", in2 := 1)
      { S7_Templates := "SrcType := Int" } EQ_Contact(in1 := "MODE SELECTION DB"."UF PLC_1 PROCESS BUFF", in2 := 560)
      Move(in := 565, out1 => "MODE SELECTION DB"."UF PLC_1 PROCESS BUFF")
   END_RUNG
   // the same network as SCL:
   IF ("MODE SELECTION DB"."UF PLC_1 MODE BUFF" = 1) AND ("MODE SELECTION DB"."UF PLC_1 PROCESS BUFF" = 560) THEN
       "MODE SELECTION DB"."UF PLC_1 PROCESS BUFF" := 565;
   END_IF;
END_REGION

REGION Network 46: ABFV 202 OPEN FB
   RUNG wire#powerrail
      { S7_Templates := "SrcType := Int" } EQ_Contact(in1 := "MODE SELECTION DB"."UF PLC_1 MODE BUFF", in2 := 1)
      { S7_Templates := "SrcType := Int" } EQ_Contact(in1 := "MODE SELECTION DB"."UF PLC_1 PROCESS BUFF", in2 := 565)
      Contact( "INPUT MAPPING DB"."ABFV 202 FEED BACK OPEN" )
      Move(in := 570, out1 => "MODE SELECTION DB"."UF PLC_1 PROCESS BUFF")
   END_RUNG
   // the same network as SCL:
   IF ("MODE SELECTION DB"."UF PLC_1 MODE BUFF" = 1) AND ("MODE SELECTION DB"."UF PLC_1 PROCESS BUFF" = 565) AND "INPUT MAPPING DB"."ABFV 202 FEED BACK OPEN" THEN
       "MODE SELECTION DB"."UF PLC_1 PROCESS BUFF" := 570;
   END_IF;
END_REGION

REGION Network 47: ABFV 204 OPEN FB
   RUNG wire#powerrail
      { S7_Templates := "SrcType := Int" } EQ_Contact(in1 := "MODE SELECTION DB"."UF PLC_1 MODE BUFF", in2 := 1)
      { S7_Templates := "SrcType := Int" } EQ_Contact(in1 := "MODE SELECTION DB"."UF PLC_1 PROCESS BUFF", in2 := 570)
      Contact( "INPUT MAPPING DB"."ABFV 204 FEED BACK OPEN" )
      Move(in := 575, out1 => "MODE SELECTION DB"."UF PLC_1 PROCESS BUFF")
   END_RUNG
   // the same network as SCL:
   IF ("MODE SELECTION DB"."UF PLC_1 MODE BUFF" = 1) AND ("MODE SELECTION DB"."UF PLC_1 PROCESS BUFF" = 570) AND "INPUT MAPPING DB"."ABFV 204 FEED BACK OPEN" THEN
       "MODE SELECTION DB"."UF PLC_1 PROCESS BUFF" := 575;
   END_IF;
END_REGION

REGION Network 48: ABFV 207 OPEN FB
   RUNG wire#powerrail
      { S7_Templates := "SrcType := Int" } EQ_Contact(in1 := "MODE SELECTION DB"."UF PLC_1 MODE BUFF", in2 := 1)
      { S7_Templates := "SrcType := Int" } EQ_Contact(in1 := "MODE SELECTION DB"."UF PLC_1 PROCESS BUFF", in2 := 575)
      Contact( "INPUT MAPPING DB"."ABFV-207 FEED BACK OPEN" )
      Move(in := 580, out1 => "MODE SELECTION DB"."UF PLC_1 PROCESS BUFF")
   END_RUNG
   // the same network as SCL:
   IF ("MODE SELECTION DB"."UF PLC_1 MODE BUFF" = 1) AND ("MODE SELECTION DB"."UF PLC_1 PROCESS BUFF" = 575) AND "INPUT MAPPING DB"."ABFV-207 FEED BACK OPEN" THEN
       "MODE SELECTION DB"."UF PLC_1 PROCESS BUFF" := 580;
   END_IF;
END_REGION

REGION Network 49: ABFV 208 OPEN FB
   RUNG wire#powerrail
      { S7_Templates := "SrcType := Int" } EQ_Contact(in1 := "MODE SELECTION DB"."UF PLC_1 MODE BUFF", in2 := 1)
      { S7_Templates := "SrcType := Int" } EQ_Contact(in1 := "MODE SELECTION DB"."UF PLC_1 PROCESS BUFF", in2 := 580)
      Contact( "INPUT MAPPING DB"."ABFV-208 FEED BACK OPEN" )
      { S7_Templates := "time_type := Time" } "IEC_Timer_0_DB_69".TON(pt := T#10S, et =>)
      Move(in := 585, out1 => "MODE SELECTION DB"."UF PLC_1 PROCESS BUFF")
   END_RUNG
   // the same network as SCL:
   "IEC_Timer_0_DB_69".TON(IN := ("MODE SELECTION DB"."UF PLC_1 MODE BUFF" = 1) AND ("MODE SELECTION DB"."UF PLC_1 PROCESS BUFF" = 580) AND "INPUT MAPPING DB"."ABFV-208 FEED BACK OPEN",
                           PT := T#10S);
   IF "IEC_Timer_0_DB_69".Q THEN "MODE SELECTION DB"."UF PLC_1 PROCESS BUFF" := 585; END_IF;
END_REGION

REGION Network 50: BACKWASH_2
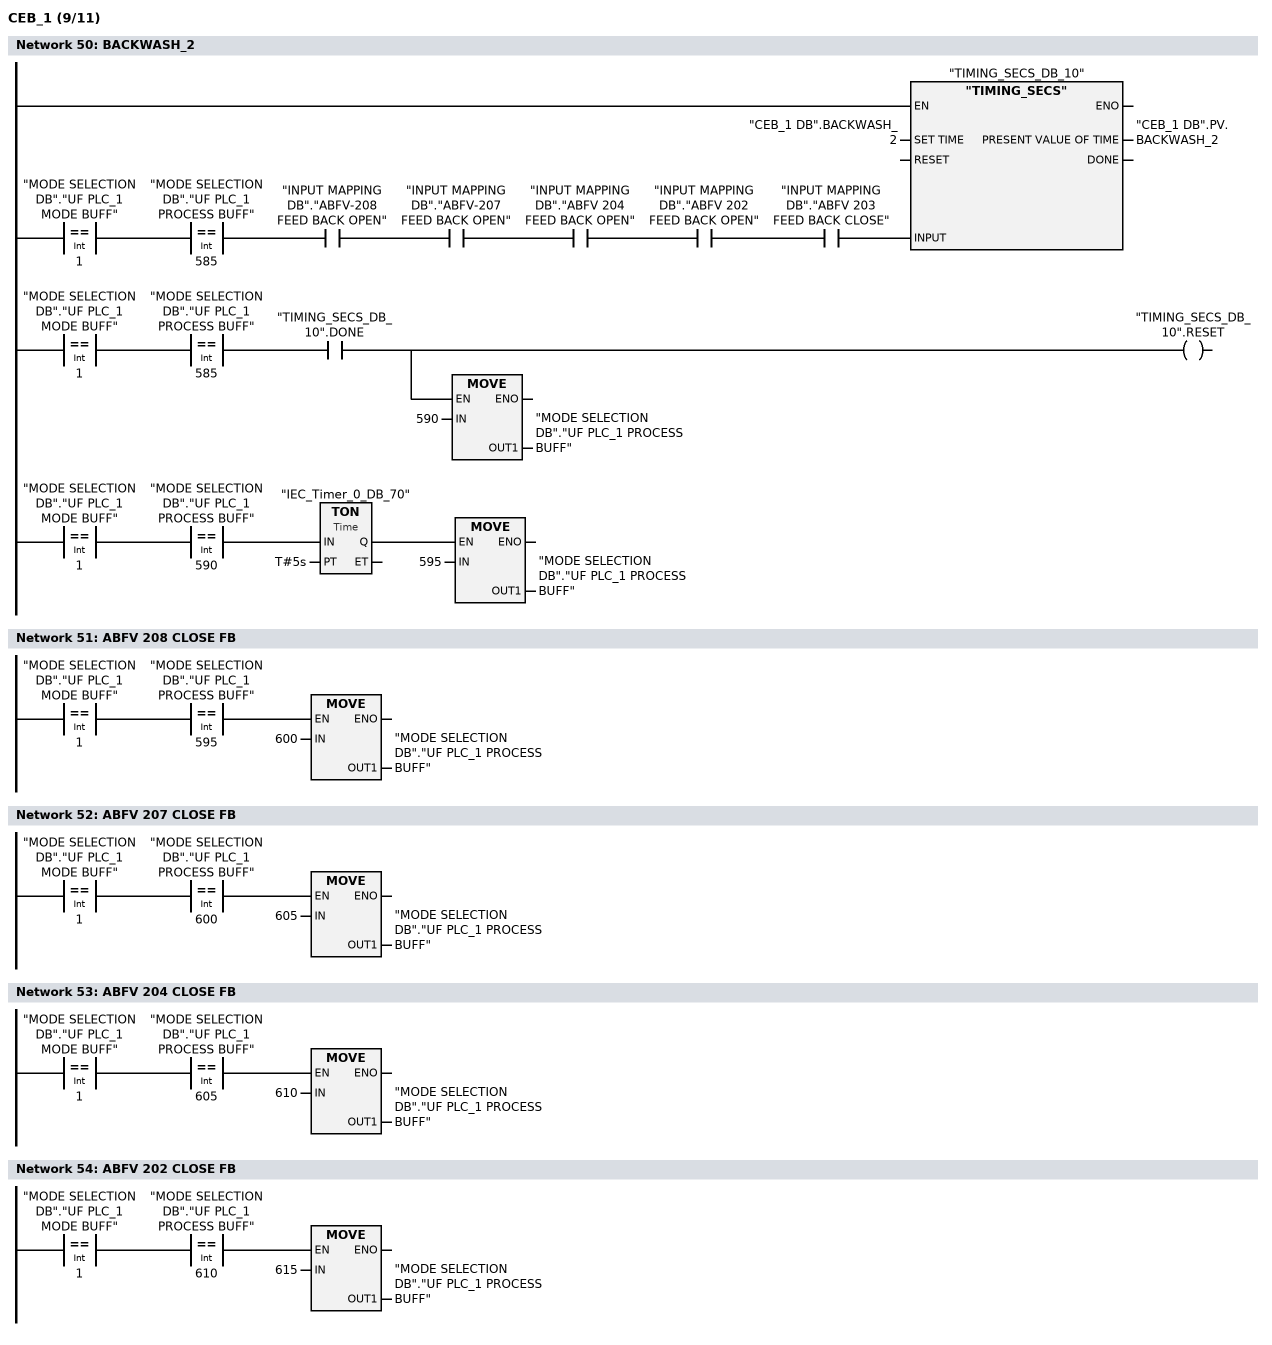
   RUNG wire#powerrail
      "TIMING_SECS_DB_10"(INPUT := wire#w1, "SET TIME" := "CEB_1 DB".BACKWASH_2, RESET :=, "PRESENT VALUE OF TIME" => "CEB_1 DB".PV.BACKWASH_2, DONE =>)
   END_RUNG
   RUNG wire#powerrail
      { S7_Templates := "SrcType := Int" } EQ_Contact(in1 := "MODE SELECTION DB"."UF PLC_1 MODE BUFF", in2 := 1)
      { S7_Templates := "SrcType := Int" } EQ_Contact(in1 := "MODE SELECTION DB"."UF PLC_1 PROCESS BUFF", in2 := 585)
      Contact( "INPUT MAPPING DB"."ABFV-208 FEED BACK OPEN" )
      Contact( "INPUT MAPPING DB"."ABFV-207 FEED BACK OPEN" )
      Contact( "INPUT MAPPING DB"."ABFV 204 FEED BACK OPEN" )
      Contact( "INPUT MAPPING DB"."ABFV 202 FEED BACK OPEN" )
      Contact( "INPUT MAPPING DB"."ABFV 203 FEED BACK CLOSE" )
   END_RUNG wire#w1
   RUNG wire#powerrail
      { S7_Templates := "SrcType := Int" } EQ_Contact(in1 := "MODE SELECTION DB"."UF PLC_1 MODE BUFF", in2 := 1)
      { S7_Templates := "SrcType := Int" } EQ_Contact(in1 := "MODE SELECTION DB"."UF PLC_1 PROCESS BUFF", in2 := 585)
      Contact( "TIMING_SECS_DB_10".DONE )
      wire#w2
      Coil( "TIMING_SECS_DB_10".RESET )
   END_RUNG
   RUNG wire#w2
      Move(in := 590, out1 => "MODE SELECTION DB"."UF PLC_1 PROCESS BUFF")
   END_RUNG
   RUNG wire#powerrail
      { S7_Templates := "SrcType := Int" } EQ_Contact(in1 := "MODE SELECTION DB"."UF PLC_1 MODE BUFF", in2 := 1)
      { S7_Templates := "SrcType := Int" } EQ_Contact(in1 := "MODE SELECTION DB"."UF PLC_1 PROCESS BUFF", in2 := 590)
      { S7_Templates := "time_type := Time" } "IEC_Timer_0_DB_70".TON(pt := T#5s, et =>)
      Move(in := 595, out1 => "MODE SELECTION DB"."UF PLC_1 PROCESS BUFF")
   END_RUNG
   // the same network as SCL:
   "TIMING_SECS_DB_10"("SET TIME" := "CEB_1 DB".BACKWASH_2,   // "TIMING_SECS"
                       INPUT := ("MODE SELECTION DB"."UF PLC_1 MODE BUFF" = 1) AND ("MODE SELECTION DB"."UF PLC_1 PROCESS BUFF" = 585) AND "INPUT MAPPING DB"."ABFV-208 FEED BACK OPEN" AND "INPUT MAPPING DB"."ABFV-207 FEED BACK OPEN" AND "INPUT MAPPING DB"."ABFV 204 FEED BACK OPEN" AND "INPUT MAPPING DB"."ABFV 202 FEED BACK OPEN" AND "INPUT MAPPING DB"."ABFV 203 FEED BACK CLOSE",
                       "PRESENT VALUE OF TIME" => "CEB_1 DB".PV.BACKWASH_2);
   "TIMING_SECS_DB_10".RESET := ("MODE SELECTION DB"."UF PLC_1 MODE BUFF" = 1) AND ("MODE SELECTION DB"."UF PLC_1 PROCESS BUFF" = 585) AND "TIMING_SECS_DB_10".DONE;
   IF "TIMING_SECS_DB_10".RESET THEN "MODE SELECTION DB"."UF PLC_1 PROCESS BUFF" := 590; END_IF;
   "IEC_Timer_0_DB_70".TON(IN := ("MODE SELECTION DB"."UF PLC_1 MODE BUFF" = 1) AND ("MODE SELECTION DB"."UF PLC_1 PROCESS BUFF" = 590),
                           PT := T#5s);
   IF "IEC_Timer_0_DB_70".Q THEN "MODE SELECTION DB"."UF PLC_1 PROCESS BUFF" := 595; END_IF;
END_REGION

REGION Network 51: ABFV 208 CLOSE FB
   RUNG wire#powerrail
      { S7_Templates := "SrcType := Int" } EQ_Contact(in1 := "MODE SELECTION DB"."UF PLC_1 MODE BUFF", in2 := 1)
      { S7_Templates := "SrcType := Int" } EQ_Contact(in1 := "MODE SELECTION DB"."UF PLC_1 PROCESS BUFF", in2 := 595)
      Move(in := 600, out1 => "MODE SELECTION DB"."UF PLC_1 PROCESS BUFF")
   END_RUNG
   // the same network as SCL:
   IF ("MODE SELECTION DB"."UF PLC_1 MODE BUFF" = 1) AND ("MODE SELECTION DB"."UF PLC_1 PROCESS BUFF" = 595) THEN
       "MODE SELECTION DB"."UF PLC_1 PROCESS BUFF" := 600;
   END_IF;
END_REGION

REGION Network 52: ABFV 207 CLOSE FB
   RUNG wire#powerrail
      { S7_Templates := "SrcType := Int" } EQ_Contact(in1 := "MODE SELECTION DB"."UF PLC_1 MODE BUFF", in2 := 1)
      { S7_Templates := "SrcType := Int" } EQ_Contact(in1 := "MODE SELECTION DB"."UF PLC_1 PROCESS BUFF", in2 := 600)
      Move(in := 605, out1 => "MODE SELECTION DB"."UF PLC_1 PROCESS BUFF")
   END_RUNG
   // the same network as SCL:
   IF ("MODE SELECTION DB"."UF PLC_1 MODE BUFF" = 1) AND ("MODE SELECTION DB"."UF PLC_1 PROCESS BUFF" = 600) THEN
       "MODE SELECTION DB"."UF PLC_1 PROCESS BUFF" := 605;
   END_IF;
END_REGION

REGION Network 53: ABFV 204 CLOSE FB
   RUNG wire#powerrail
      { S7_Templates := "SrcType := Int" } EQ_Contact(in1 := "MODE SELECTION DB"."UF PLC_1 MODE BUFF", in2 := 1)
      { S7_Templates := "SrcType := Int" } EQ_Contact(in1 := "MODE SELECTION DB"."UF PLC_1 PROCESS BUFF", in2 := 605)
      Move(in := 610, out1 => "MODE SELECTION DB"."UF PLC_1 PROCESS BUFF")
   END_RUNG
   // the same network as SCL:
   IF ("MODE SELECTION DB"."UF PLC_1 MODE BUFF" = 1) AND ("MODE SELECTION DB"."UF PLC_1 PROCESS BUFF" = 605) THEN
       "MODE SELECTION DB"."UF PLC_1 PROCESS BUFF" := 610;
   END_IF;
END_REGION

REGION Network 54: ABFV 202 CLOSE FB
   RUNG wire#powerrail
      { S7_Templates := "SrcType := Int" } EQ_Contact(in1 := "MODE SELECTION DB"."UF PLC_1 MODE BUFF", in2 := 1)
      { S7_Templates := "SrcType := Int" } EQ_Contact(in1 := "MODE SELECTION DB"."UF PLC_1 PROCESS BUFF", in2 := 610)
      Move(in := 615, out1 => "MODE SELECTION DB"."UF PLC_1 PROCESS BUFF")
   END_RUNG
   // the same network as SCL:
   IF ("MODE SELECTION DB"."UF PLC_1 MODE BUFF" = 1) AND ("MODE SELECTION DB"."UF PLC_1 PROCESS BUFF" = 610) THEN
       "MODE SELECTION DB"."UF PLC_1 PROCESS BUFF" := 615;
   END_IF;
END_REGION

REGION Network 55: 620
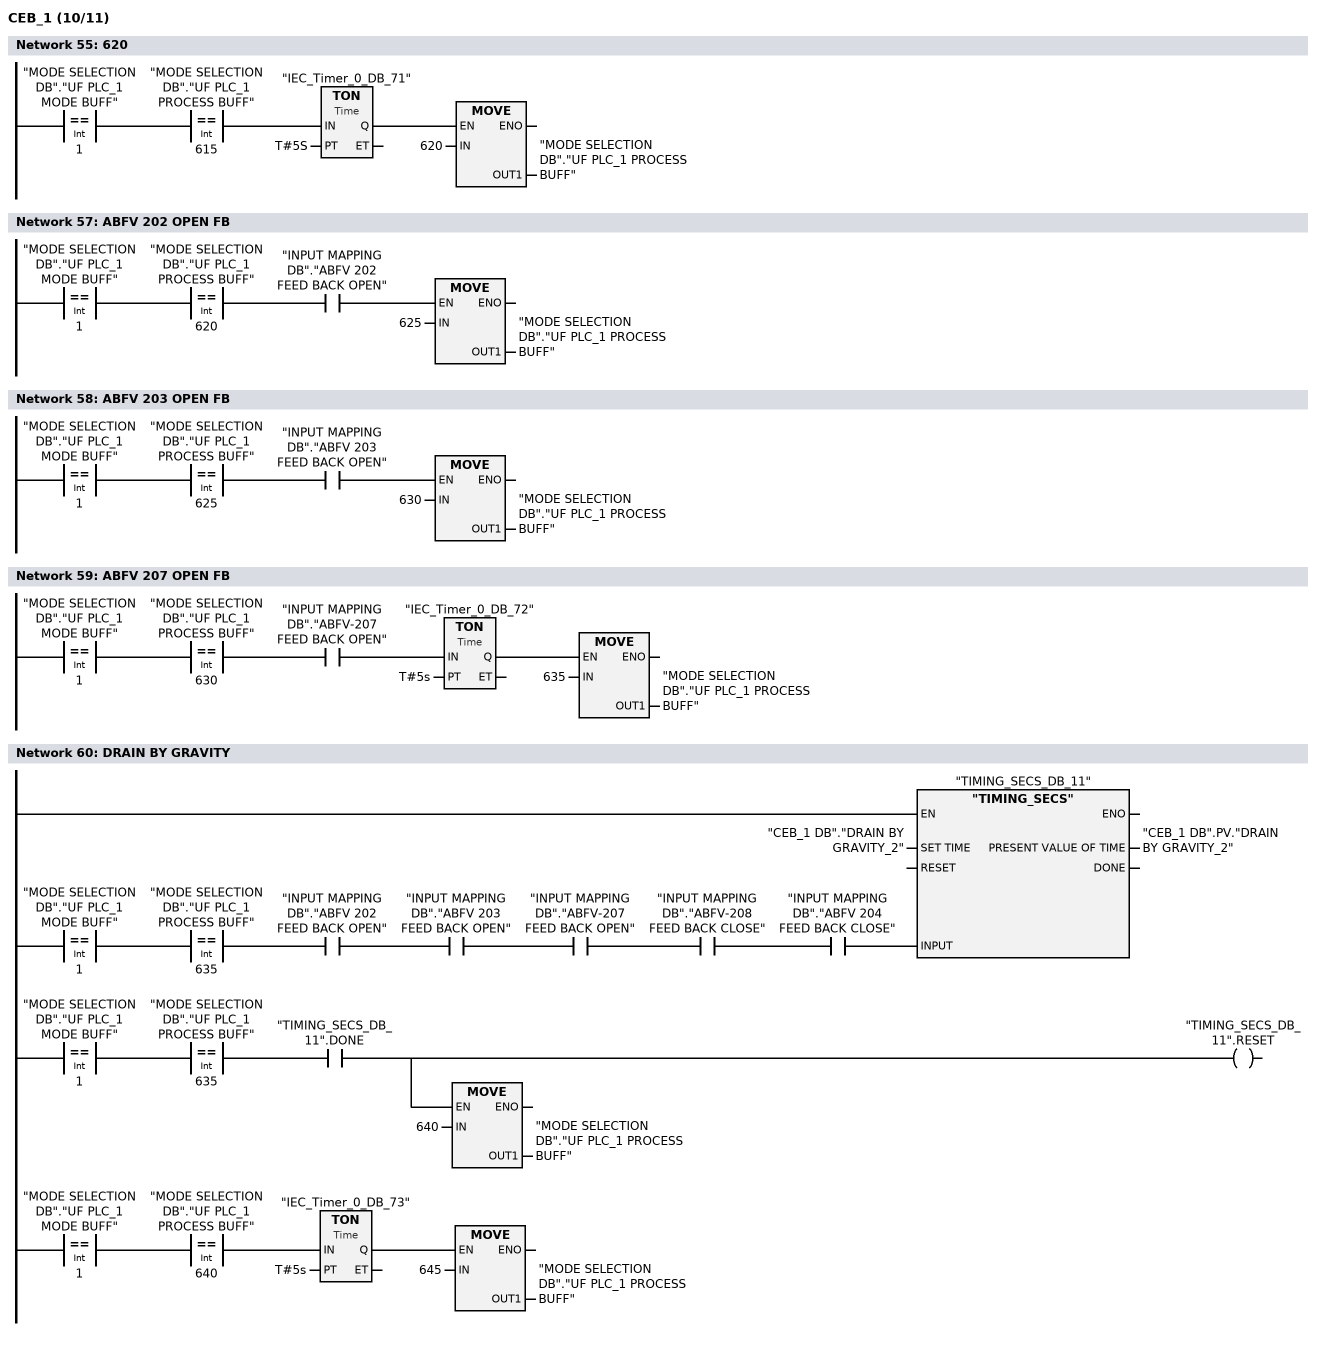
   RUNG wire#powerrail
      { S7_Templates := "SrcType := Int" } EQ_Contact(in1 := "MODE SELECTION DB"."UF PLC_1 MODE BUFF", in2 := 1)
      { S7_Templates := "SrcType := Int" } EQ_Contact(in1 := "MODE SELECTION DB"."UF PLC_1 PROCESS BUFF", in2 := 615)
      { S7_Templates := "time_type := Time" } "IEC_Timer_0_DB_71".TON(pt := T#5S, et =>)
      Move(in := 620, out1 => "MODE SELECTION DB"."UF PLC_1 PROCESS BUFF")
   END_RUNG
   // the same network as SCL:
   "IEC_Timer_0_DB_71".TON(IN := ("MODE SELECTION DB"."UF PLC_1 MODE BUFF" = 1) AND ("MODE SELECTION DB"."UF PLC_1 PROCESS BUFF" = 615),
                           PT := T#5S);
   IF "IEC_Timer_0_DB_71".Q THEN "MODE SELECTION DB"."UF PLC_1 PROCESS BUFF" := 620; END_IF;
END_REGION

REGION Network 57: ABFV 202 OPEN FB
   RUNG wire#powerrail
      { S7_Templates := "SrcType := Int" } EQ_Contact(in1 := "MODE SELECTION DB"."UF PLC_1 MODE BUFF", in2 := 1)
      { S7_Templates := "SrcType := Int" } EQ_Contact(in1 := "MODE SELECTION DB"."UF PLC_1 PROCESS BUFF", in2 := 620)
      Contact( "INPUT MAPPING DB"."ABFV 202 FEED BACK OPEN" )
      Move(in := 625, out1 => "MODE SELECTION DB"."UF PLC_1 PROCESS BUFF")
   END_RUNG
   // the same network as SCL:
   IF ("MODE SELECTION DB"."UF PLC_1 MODE BUFF" = 1) AND ("MODE SELECTION DB"."UF PLC_1 PROCESS BUFF" = 620) AND "INPUT MAPPING DB"."ABFV 202 FEED BACK OPEN" THEN
       "MODE SELECTION DB"."UF PLC_1 PROCESS BUFF" := 625;
   END_IF;
END_REGION

REGION Network 58: ABFV 203 OPEN FB
   RUNG wire#powerrail
      { S7_Templates := "SrcType := Int" } EQ_Contact(in1 := "MODE SELECTION DB"."UF PLC_1 MODE BUFF", in2 := 1)
      { S7_Templates := "SrcType := Int" } EQ_Contact(in1 := "MODE SELECTION DB"."UF PLC_1 PROCESS BUFF", in2 := 625)
      Contact( "INPUT MAPPING DB"."ABFV 203 FEED BACK OPEN" )
      Move(in := 630, out1 => "MODE SELECTION DB"."UF PLC_1 PROCESS BUFF")
   END_RUNG
   // the same network as SCL:
   IF ("MODE SELECTION DB"."UF PLC_1 MODE BUFF" = 1) AND ("MODE SELECTION DB"."UF PLC_1 PROCESS BUFF" = 625) AND "INPUT MAPPING DB"."ABFV 203 FEED BACK OPEN" THEN
       "MODE SELECTION DB"."UF PLC_1 PROCESS BUFF" := 630;
   END_IF;
END_REGION

REGION Network 59: ABFV 207 OPEN FB
   RUNG wire#powerrail
      { S7_Templates := "SrcType := Int" } EQ_Contact(in1 := "MODE SELECTION DB"."UF PLC_1 MODE BUFF", in2 := 1)
      { S7_Templates := "SrcType := Int" } EQ_Contact(in1 := "MODE SELECTION DB"."UF PLC_1 PROCESS BUFF", in2 := 630)
      Contact( "INPUT MAPPING DB"."ABFV-207 FEED BACK OPEN" )
      { S7_Templates := "time_type := Time" } "IEC_Timer_0_DB_72".TON(pt := T#5s, et =>)
      Move(in := 635, out1 => "MODE SELECTION DB"."UF PLC_1 PROCESS BUFF")
   END_RUNG
   // the same network as SCL:
   "IEC_Timer_0_DB_72".TON(IN := ("MODE SELECTION DB"."UF PLC_1 MODE BUFF" = 1) AND ("MODE SELECTION DB"."UF PLC_1 PROCESS BUFF" = 630) AND "INPUT MAPPING DB"."ABFV-207 FEED BACK OPEN",
                           PT := T#5s);
   IF "IEC_Timer_0_DB_72".Q THEN "MODE SELECTION DB"."UF PLC_1 PROCESS BUFF" := 635; END_IF;
END_REGION

REGION Network 60: DRAIN BY GRAVITY
   RUNG wire#powerrail
      "TIMING_SECS_DB_11"(INPUT := wire#w1, "SET TIME" := "CEB_1 DB"."DRAIN BY GRAVITY_2", RESET :=, "PRESENT VALUE OF TIME" => "CEB_1 DB".PV."DRAIN BY GRAVITY_2", DONE =>)
   END_RUNG
   RUNG wire#powerrail
      { S7_Templates := "SrcType := Int" } EQ_Contact(in1 := "MODE SELECTION DB"."UF PLC_1 MODE BUFF", in2 := 1)
      { S7_Templates := "SrcType := Int" } EQ_Contact(in1 := "MODE SELECTION DB"."UF PLC_1 PROCESS BUFF", in2 := 635)
      Contact( "INPUT MAPPING DB"."ABFV 202 FEED BACK OPEN" )
      Contact( "INPUT MAPPING DB"."ABFV 203 FEED BACK OPEN" )
      Contact( "INPUT MAPPING DB"."ABFV-207 FEED BACK OPEN" )
      Contact( "INPUT MAPPING DB"."ABFV-208 FEED BACK CLOSE" )
      Contact( "INPUT MAPPING DB"."ABFV 204 FEED BACK CLOSE" )
   END_RUNG wire#w1
   RUNG wire#powerrail
      { S7_Templates := "SrcType := Int" } EQ_Contact(in1 := "MODE SELECTION DB"."UF PLC_1 MODE BUFF", in2 := 1)
      { S7_Templates := "SrcType := Int" } EQ_Contact(in1 := "MODE SELECTION DB"."UF PLC_1 PROCESS BUFF", in2 := 635)
      Contact( "TIMING_SECS_DB_11".DONE )
      wire#w2
      Coil( "TIMING_SECS_DB_11".RESET )
   END_RUNG
   RUNG wire#w2
      Move(in := 640, out1 => "MODE SELECTION DB"."UF PLC_1 PROCESS BUFF")
   END_RUNG
   RUNG wire#powerrail
      { S7_Templates := "SrcType := Int" } EQ_Contact(in1 := "MODE SELECTION DB"."UF PLC_1 MODE BUFF", in2 := 1)
      { S7_Templates := "SrcType := Int" } EQ_Contact(in1 := "MODE SELECTION DB"."UF PLC_1 PROCESS BUFF", in2 := 640)
      { S7_Templates := "time_type := Time" } "IEC_Timer_0_DB_73".TON(pt := T#5s, et =>)
      Move(in := 645, out1 => "MODE SELECTION DB"."UF PLC_1 PROCESS BUFF")
   END_RUNG
   // the same network as SCL:
   "TIMING_SECS_DB_11"("SET TIME" := "CEB_1 DB"."DRAIN BY GRAVITY_2",   // "TIMING_SECS"
                       INPUT := ("MODE SELECTION DB"."UF PLC_1 MODE BUFF" = 1) AND ("MODE SELECTION DB"."UF PLC_1 PROCESS BUFF" = 635) AND "INPUT MAPPING DB"."ABFV 202 FEED BACK OPEN" AND "INPUT MAPPING DB"."ABFV 203 FEED BACK OPEN" AND "INPUT MAPPING DB"."ABFV-207 FEED BACK OPEN" AND "INPUT MAPPING DB"."ABFV-208 FEED BACK CLOSE" AND "INPUT MAPPING DB"."ABFV 204 FEED BACK CLOSE",
                       "PRESENT VALUE OF TIME" => "CEB_1 DB".PV."DRAIN BY GRAVITY_2");
   "TIMING_SECS_DB_11".RESET := ("MODE SELECTION DB"."UF PLC_1 MODE BUFF" = 1) AND ("MODE SELECTION DB"."UF PLC_1 PROCESS BUFF" = 635) AND "TIMING_SECS_DB_11".DONE;
   IF "TIMING_SECS_DB_11".RESET THEN "MODE SELECTION DB"."UF PLC_1 PROCESS BUFF" := 640; END_IF;
   "IEC_Timer_0_DB_73".TON(IN := ("MODE SELECTION DB"."UF PLC_1 MODE BUFF" = 1) AND ("MODE SELECTION DB"."UF PLC_1 PROCESS BUFF" = 640),
                           PT := T#5s);
   IF "IEC_Timer_0_DB_73".Q THEN "MODE SELECTION DB"."UF PLC_1 PROCESS BUFF" := 645; END_IF;
END_REGION

REGION Network 61: ABFV 207 CLOSE FB
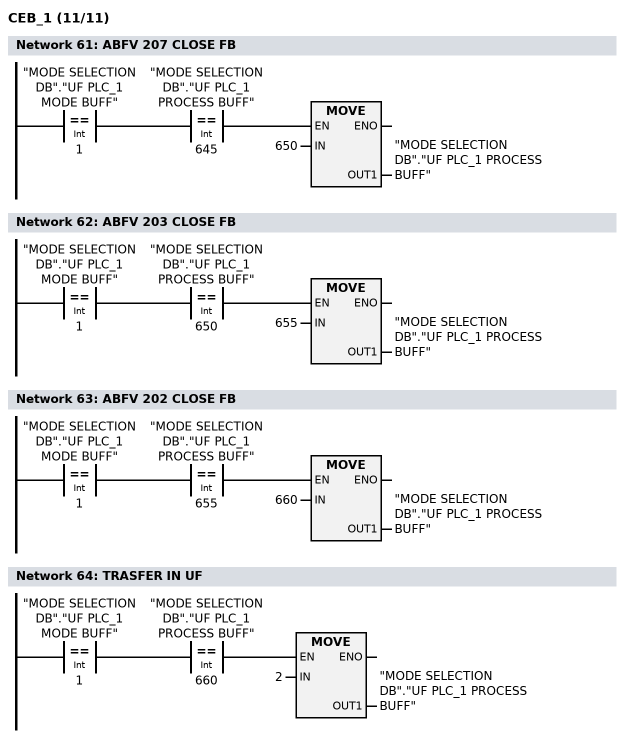
   RUNG wire#powerrail
      { S7_Templates := "SrcType := Int" } EQ_Contact(in1 := "MODE SELECTION DB"."UF PLC_1 MODE BUFF", in2 := 1)
      { S7_Templates := "SrcType := Int" } EQ_Contact(in1 := "MODE SELECTION DB"."UF PLC_1 PROCESS BUFF", in2 := 645)
      Move(in := 650, out1 => "MODE SELECTION DB"."UF PLC_1 PROCESS BUFF")
   END_RUNG
   // the same network as SCL:
   IF ("MODE SELECTION DB"."UF PLC_1 MODE BUFF" = 1) AND ("MODE SELECTION DB"."UF PLC_1 PROCESS BUFF" = 645) THEN
       "MODE SELECTION DB"."UF PLC_1 PROCESS BUFF" := 650;
   END_IF;
END_REGION

REGION Network 62: ABFV 203 CLOSE FB
   RUNG wire#powerrail
      { S7_Templates := "SrcType := Int" } EQ_Contact(in1 := "MODE SELECTION DB"."UF PLC_1 MODE BUFF", in2 := 1)
      { S7_Templates := "SrcType := Int" } EQ_Contact(in1 := "MODE SELECTION DB"."UF PLC_1 PROCESS BUFF", in2 := 650)
      Move(in := 655, out1 => "MODE SELECTION DB"."UF PLC_1 PROCESS BUFF")
   END_RUNG
   // the same network as SCL:
   IF ("MODE SELECTION DB"."UF PLC_1 MODE BUFF" = 1) AND ("MODE SELECTION DB"."UF PLC_1 PROCESS BUFF" = 650) THEN
       "MODE SELECTION DB"."UF PLC_1 PROCESS BUFF" := 655;
   END_IF;
END_REGION

REGION Network 63: ABFV 202 CLOSE FB
   RUNG wire#powerrail
      { S7_Templates := "SrcType := Int" } EQ_Contact(in1 := "MODE SELECTION DB"."UF PLC_1 MODE BUFF", in2 := 1)
      { S7_Templates := "SrcType := Int" } EQ_Contact(in1 := "MODE SELECTION DB"."UF PLC_1 PROCESS BUFF", in2 := 655)
      Move(in := 660, out1 => "MODE SELECTION DB"."UF PLC_1 PROCESS BUFF")
   END_RUNG
   // the same network as SCL:
   IF ("MODE SELECTION DB"."UF PLC_1 MODE BUFF" = 1) AND ("MODE SELECTION DB"."UF PLC_1 PROCESS BUFF" = 655) THEN
       "MODE SELECTION DB"."UF PLC_1 PROCESS BUFF" := 660;
   END_IF;
END_REGION

REGION Network 64: TRASFER IN UF
   RUNG wire#powerrail
      { S7_Templates := "SrcType := Int" } EQ_Contact(in1 := "MODE SELECTION DB"."UF PLC_1 MODE BUFF", in2 := 1)
      { S7_Templates := "SrcType := Int" } EQ_Contact(in1 := "MODE SELECTION DB"."UF PLC_1 PROCESS BUFF", in2 := 660)
      Move(in := 2, out1 => "MODE SELECTION DB"."UF PLC_1 PROCESS BUFF")
   END_RUNG
   // the same network as SCL:
   IF ("MODE SELECTION DB"."UF PLC_1 MODE BUFF" = 1) AND ("MODE SELECTION DB"."UF PLC_1 PROCESS BUFF" = 660) THEN
       "MODE SELECTION DB"."UF PLC_1 PROCESS BUFF" := 2;
   END_IF;
END_REGION
END_FUNCTION

FUNCTION "CEB_2" : Void   // FC15, LAD
{ S7_Optimized_Access := 'TRUE' }
// stored: SetENOAutomatically false
BEGIN

REGION Network 2: CEB_2 START
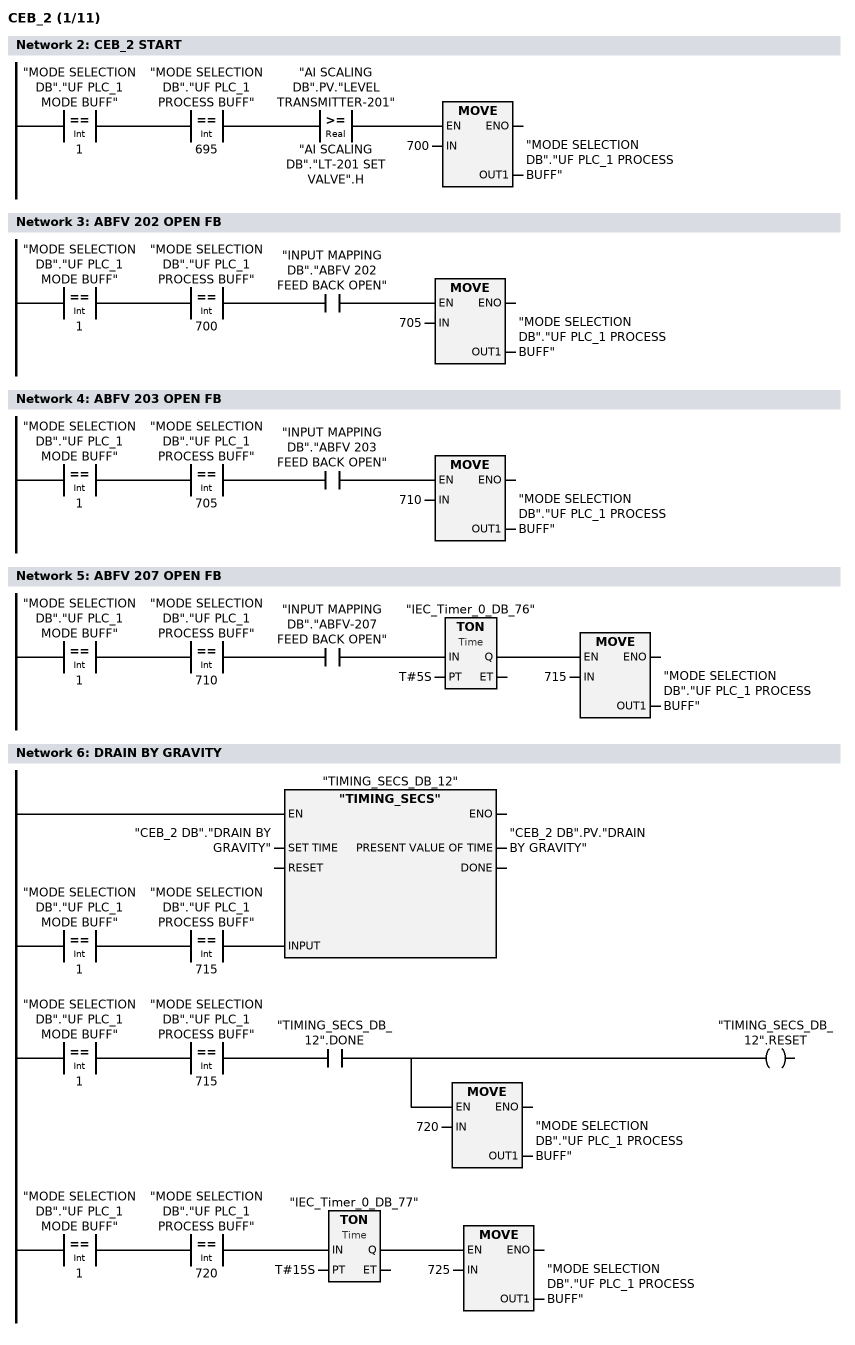
   RUNG wire#powerrail
      { S7_Templates := "SrcType := Int" } EQ_Contact(in1 := "MODE SELECTION DB"."UF PLC_1 MODE BUFF", in2 := 1)
      { S7_Templates := "SrcType := Int" } EQ_Contact(in1 := "MODE SELECTION DB"."UF PLC_1 PROCESS BUFF", in2 := 695)
      { S7_Templates := "SrcType := Real" } GE_Contact(in1 := "AI SCALING DB".PV."LEVEL TRANSMITTER-201", in2 := "AI SCALING DB"."LT-201 SET VALVE".H)
      Move(in := 700, out1 => "MODE SELECTION DB"."UF PLC_1 PROCESS BUFF")
   END_RUNG
   // the same network as SCL:
   IF ("MODE SELECTION DB"."UF PLC_1 MODE BUFF" = 1) AND ("MODE SELECTION DB"."UF PLC_1 PROCESS BUFF" = 695) AND ("AI SCALING DB".PV."LEVEL TRANSMITTER-201" >= "AI SCALING DB"."LT-201 SET VALVE".H) THEN
       "MODE SELECTION DB"."UF PLC_1 PROCESS BUFF" := 700;
   END_IF;
END_REGION

REGION Network 3: ABFV 202 OPEN FB
   RUNG wire#powerrail
      { S7_Templates := "SrcType := Int" } EQ_Contact(in1 := "MODE SELECTION DB"."UF PLC_1 MODE BUFF", in2 := 1)
      { S7_Templates := "SrcType := Int" } EQ_Contact(in1 := "MODE SELECTION DB"."UF PLC_1 PROCESS BUFF", in2 := 700)
      Contact( "INPUT MAPPING DB"."ABFV 202 FEED BACK OPEN" )
      Move(in := 705, out1 => "MODE SELECTION DB"."UF PLC_1 PROCESS BUFF")
   END_RUNG
   // the same network as SCL:
   IF ("MODE SELECTION DB"."UF PLC_1 MODE BUFF" = 1) AND ("MODE SELECTION DB"."UF PLC_1 PROCESS BUFF" = 700) AND "INPUT MAPPING DB"."ABFV 202 FEED BACK OPEN" THEN
       "MODE SELECTION DB"."UF PLC_1 PROCESS BUFF" := 705;
   END_IF;
END_REGION

REGION Network 4: ABFV 203 OPEN FB
   RUNG wire#powerrail
      { S7_Templates := "SrcType := Int" } EQ_Contact(in1 := "MODE SELECTION DB"."UF PLC_1 MODE BUFF", in2 := 1)
      { S7_Templates := "SrcType := Int" } EQ_Contact(in1 := "MODE SELECTION DB"."UF PLC_1 PROCESS BUFF", in2 := 705)
      Contact( "INPUT MAPPING DB"."ABFV 203 FEED BACK OPEN" )
      Move(in := 710, out1 => "MODE SELECTION DB"."UF PLC_1 PROCESS BUFF")
   END_RUNG
   // the same network as SCL:
   IF ("MODE SELECTION DB"."UF PLC_1 MODE BUFF" = 1) AND ("MODE SELECTION DB"."UF PLC_1 PROCESS BUFF" = 705) AND "INPUT MAPPING DB"."ABFV 203 FEED BACK OPEN" THEN
       "MODE SELECTION DB"."UF PLC_1 PROCESS BUFF" := 710;
   END_IF;
END_REGION

REGION Network 5: ABFV 207 OPEN FB
   RUNG wire#powerrail
      { S7_Templates := "SrcType := Int" } EQ_Contact(in1 := "MODE SELECTION DB"."UF PLC_1 MODE BUFF", in2 := 1)
      { S7_Templates := "SrcType := Int" } EQ_Contact(in1 := "MODE SELECTION DB"."UF PLC_1 PROCESS BUFF", in2 := 710)
      Contact( "INPUT MAPPING DB"."ABFV-207 FEED BACK OPEN" )
      { S7_Templates := "time_type := Time" } "IEC_Timer_0_DB_76".TON(pt := T#5S, et =>)
      Move(in := 715, out1 => "MODE SELECTION DB"."UF PLC_1 PROCESS BUFF")
   END_RUNG
   // the same network as SCL:
   "IEC_Timer_0_DB_76".TON(IN := ("MODE SELECTION DB"."UF PLC_1 MODE BUFF" = 1) AND ("MODE SELECTION DB"."UF PLC_1 PROCESS BUFF" = 710) AND "INPUT MAPPING DB"."ABFV-207 FEED BACK OPEN",
                           PT := T#5S);
   IF "IEC_Timer_0_DB_76".Q THEN "MODE SELECTION DB"."UF PLC_1 PROCESS BUFF" := 715; END_IF;
END_REGION

REGION Network 6: DRAIN BY GRAVITY
   RUNG wire#powerrail
      "TIMING_SECS_DB_12"(INPUT := wire#w1, "SET TIME" := "CEB_2 DB"."DRAIN BY GRAVITY", RESET :=, "PRESENT VALUE OF TIME" => "CEB_2 DB".PV."DRAIN BY GRAVITY", DONE =>)
   END_RUNG
   RUNG wire#powerrail
      { S7_Templates := "SrcType := Int" } EQ_Contact(in1 := "MODE SELECTION DB"."UF PLC_1 MODE BUFF", in2 := 1)
      { S7_Templates := "SrcType := Int" } EQ_Contact(in1 := "MODE SELECTION DB"."UF PLC_1 PROCESS BUFF", in2 := 715)
   END_RUNG wire#w1
   RUNG wire#powerrail
      { S7_Templates := "SrcType := Int" } EQ_Contact(in1 := "MODE SELECTION DB"."UF PLC_1 MODE BUFF", in2 := 1)
      { S7_Templates := "SrcType := Int" } EQ_Contact(in1 := "MODE SELECTION DB"."UF PLC_1 PROCESS BUFF", in2 := 715)
      Contact( "TIMING_SECS_DB_12".DONE )
      wire#w2
      Coil( "TIMING_SECS_DB_12".RESET )
   END_RUNG
   RUNG wire#w2
      Move(in := 720, out1 => "MODE SELECTION DB"."UF PLC_1 PROCESS BUFF")
   END_RUNG
   RUNG wire#powerrail
      { S7_Templates := "SrcType := Int" } EQ_Contact(in1 := "MODE SELECTION DB"."UF PLC_1 MODE BUFF", in2 := 1)
      { S7_Templates := "SrcType := Int" } EQ_Contact(in1 := "MODE SELECTION DB"."UF PLC_1 PROCESS BUFF", in2 := 720)
      { S7_Templates := "time_type := Time" } "IEC_Timer_0_DB_77".TON(pt := T#15S, et =>)
      Move(in := 725, out1 => "MODE SELECTION DB"."UF PLC_1 PROCESS BUFF")
   END_RUNG
   // the same network as SCL:
   "TIMING_SECS_DB_12"("SET TIME" := "CEB_2 DB"."DRAIN BY GRAVITY",   // "TIMING_SECS"
                       INPUT := ("MODE SELECTION DB"."UF PLC_1 MODE BUFF" = 1) AND ("MODE SELECTION DB"."UF PLC_1 PROCESS BUFF" = 715),
                       "PRESENT VALUE OF TIME" => "CEB_2 DB".PV."DRAIN BY GRAVITY");
   "TIMING_SECS_DB_12".RESET := ("MODE SELECTION DB"."UF PLC_1 MODE BUFF" = 1) AND ("MODE SELECTION DB"."UF PLC_1 PROCESS BUFF" = 715) AND "TIMING_SECS_DB_12".DONE;
   IF "TIMING_SECS_DB_12".RESET THEN "MODE SELECTION DB"."UF PLC_1 PROCESS BUFF" := 720; END_IF;
   "IEC_Timer_0_DB_77".TON(IN := ("MODE SELECTION DB"."UF PLC_1 MODE BUFF" = 1) AND ("MODE SELECTION DB"."UF PLC_1 PROCESS BUFF" = 720),
                           PT := T#15S);
   IF "IEC_Timer_0_DB_77".Q THEN "MODE SELECTION DB"."UF PLC_1 PROCESS BUFF" := 725; END_IF;
END_REGION

REGION Network 7: ABFV 207 CLOSE FB
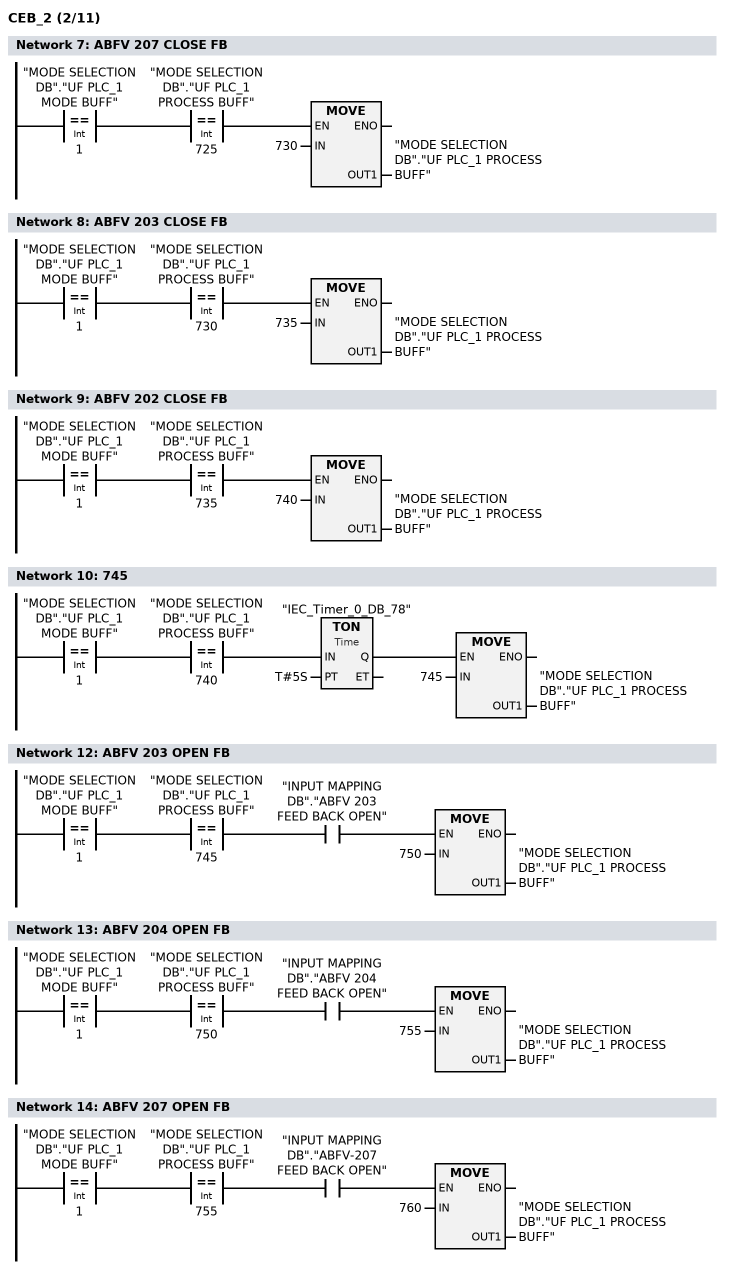
   RUNG wire#powerrail
      { S7_Templates := "SrcType := Int" } EQ_Contact(in1 := "MODE SELECTION DB"."UF PLC_1 MODE BUFF", in2 := 1)
      { S7_Templates := "SrcType := Int" } EQ_Contact(in1 := "MODE SELECTION DB"."UF PLC_1 PROCESS BUFF", in2 := 725)
      Move(in := 730, out1 => "MODE SELECTION DB"."UF PLC_1 PROCESS BUFF")
   END_RUNG
   // the same network as SCL:
   IF ("MODE SELECTION DB"."UF PLC_1 MODE BUFF" = 1) AND ("MODE SELECTION DB"."UF PLC_1 PROCESS BUFF" = 725) THEN
       "MODE SELECTION DB"."UF PLC_1 PROCESS BUFF" := 730;
   END_IF;
END_REGION

REGION Network 8: ABFV 203 CLOSE FB
   RUNG wire#powerrail
      { S7_Templates := "SrcType := Int" } EQ_Contact(in1 := "MODE SELECTION DB"."UF PLC_1 MODE BUFF", in2 := 1)
      { S7_Templates := "SrcType := Int" } EQ_Contact(in1 := "MODE SELECTION DB"."UF PLC_1 PROCESS BUFF", in2 := 730)
      Move(in := 735, out1 => "MODE SELECTION DB"."UF PLC_1 PROCESS BUFF")
   END_RUNG
   // the same network as SCL:
   IF ("MODE SELECTION DB"."UF PLC_1 MODE BUFF" = 1) AND ("MODE SELECTION DB"."UF PLC_1 PROCESS BUFF" = 730) THEN
       "MODE SELECTION DB"."UF PLC_1 PROCESS BUFF" := 735;
   END_IF;
END_REGION

REGION Network 9: ABFV 202 CLOSE FB
   RUNG wire#powerrail
      { S7_Templates := "SrcType := Int" } EQ_Contact(in1 := "MODE SELECTION DB"."UF PLC_1 MODE BUFF", in2 := 1)
      { S7_Templates := "SrcType := Int" } EQ_Contact(in1 := "MODE SELECTION DB"."UF PLC_1 PROCESS BUFF", in2 := 735)
      Move(in := 740, out1 => "MODE SELECTION DB"."UF PLC_1 PROCESS BUFF")
   END_RUNG
   // the same network as SCL:
   IF ("MODE SELECTION DB"."UF PLC_1 MODE BUFF" = 1) AND ("MODE SELECTION DB"."UF PLC_1 PROCESS BUFF" = 735) THEN
       "MODE SELECTION DB"."UF PLC_1 PROCESS BUFF" := 740;
   END_IF;
END_REGION

REGION Network 10: 745
   RUNG wire#powerrail
      { S7_Templates := "SrcType := Int" } EQ_Contact(in1 := "MODE SELECTION DB"."UF PLC_1 MODE BUFF", in2 := 1)
      { S7_Templates := "SrcType := Int" } EQ_Contact(in1 := "MODE SELECTION DB"."UF PLC_1 PROCESS BUFF", in2 := 740)
      { S7_Templates := "time_type := Time" } "IEC_Timer_0_DB_78".TON(pt := T#5S, et =>)
      Move(in := 745, out1 => "MODE SELECTION DB"."UF PLC_1 PROCESS BUFF")
   END_RUNG
   // the same network as SCL:
   "IEC_Timer_0_DB_78".TON(IN := ("MODE SELECTION DB"."UF PLC_1 MODE BUFF" = 1) AND ("MODE SELECTION DB"."UF PLC_1 PROCESS BUFF" = 740),
                           PT := T#5S);
   IF "IEC_Timer_0_DB_78".Q THEN "MODE SELECTION DB"."UF PLC_1 PROCESS BUFF" := 745; END_IF;
END_REGION

REGION Network 12: ABFV 203 OPEN FB
   RUNG wire#powerrail
      { S7_Templates := "SrcType := Int" } EQ_Contact(in1 := "MODE SELECTION DB"."UF PLC_1 MODE BUFF", in2 := 1)
      { S7_Templates := "SrcType := Int" } EQ_Contact(in1 := "MODE SELECTION DB"."UF PLC_1 PROCESS BUFF", in2 := 745)
      Contact( "INPUT MAPPING DB"."ABFV 203 FEED BACK OPEN" )
      Move(in := 750, out1 => "MODE SELECTION DB"."UF PLC_1 PROCESS BUFF")
   END_RUNG
   // the same network as SCL:
   IF ("MODE SELECTION DB"."UF PLC_1 MODE BUFF" = 1) AND ("MODE SELECTION DB"."UF PLC_1 PROCESS BUFF" = 745) AND "INPUT MAPPING DB"."ABFV 203 FEED BACK OPEN" THEN
       "MODE SELECTION DB"."UF PLC_1 PROCESS BUFF" := 750;
   END_IF;
END_REGION

REGION Network 13: ABFV 204 OPEN FB
   RUNG wire#powerrail
      { S7_Templates := "SrcType := Int" } EQ_Contact(in1 := "MODE SELECTION DB"."UF PLC_1 MODE BUFF", in2 := 1)
      { S7_Templates := "SrcType := Int" } EQ_Contact(in1 := "MODE SELECTION DB"."UF PLC_1 PROCESS BUFF", in2 := 750)
      Contact( "INPUT MAPPING DB"."ABFV 204 FEED BACK OPEN" )
      Move(in := 755, out1 => "MODE SELECTION DB"."UF PLC_1 PROCESS BUFF")
   END_RUNG
   // the same network as SCL:
   IF ("MODE SELECTION DB"."UF PLC_1 MODE BUFF" = 1) AND ("MODE SELECTION DB"."UF PLC_1 PROCESS BUFF" = 750) AND "INPUT MAPPING DB"."ABFV 204 FEED BACK OPEN" THEN
       "MODE SELECTION DB"."UF PLC_1 PROCESS BUFF" := 755;
   END_IF;
END_REGION

REGION Network 14: ABFV 207 OPEN FB
   RUNG wire#powerrail
      { S7_Templates := "SrcType := Int" } EQ_Contact(in1 := "MODE SELECTION DB"."UF PLC_1 MODE BUFF", in2 := 1)
      { S7_Templates := "SrcType := Int" } EQ_Contact(in1 := "MODE SELECTION DB"."UF PLC_1 PROCESS BUFF", in2 := 755)
      Contact( "INPUT MAPPING DB"."ABFV-207 FEED BACK OPEN" )
      Move(in := 760, out1 => "MODE SELECTION DB"."UF PLC_1 PROCESS BUFF")
   END_RUNG
   // the same network as SCL:
   IF ("MODE SELECTION DB"."UF PLC_1 MODE BUFF" = 1) AND ("MODE SELECTION DB"."UF PLC_1 PROCESS BUFF" = 755) AND "INPUT MAPPING DB"."ABFV-207 FEED BACK OPEN" THEN
       "MODE SELECTION DB"."UF PLC_1 PROCESS BUFF" := 760;
   END_IF;
END_REGION

REGION Network 15: ABFV 208 OPEN FB
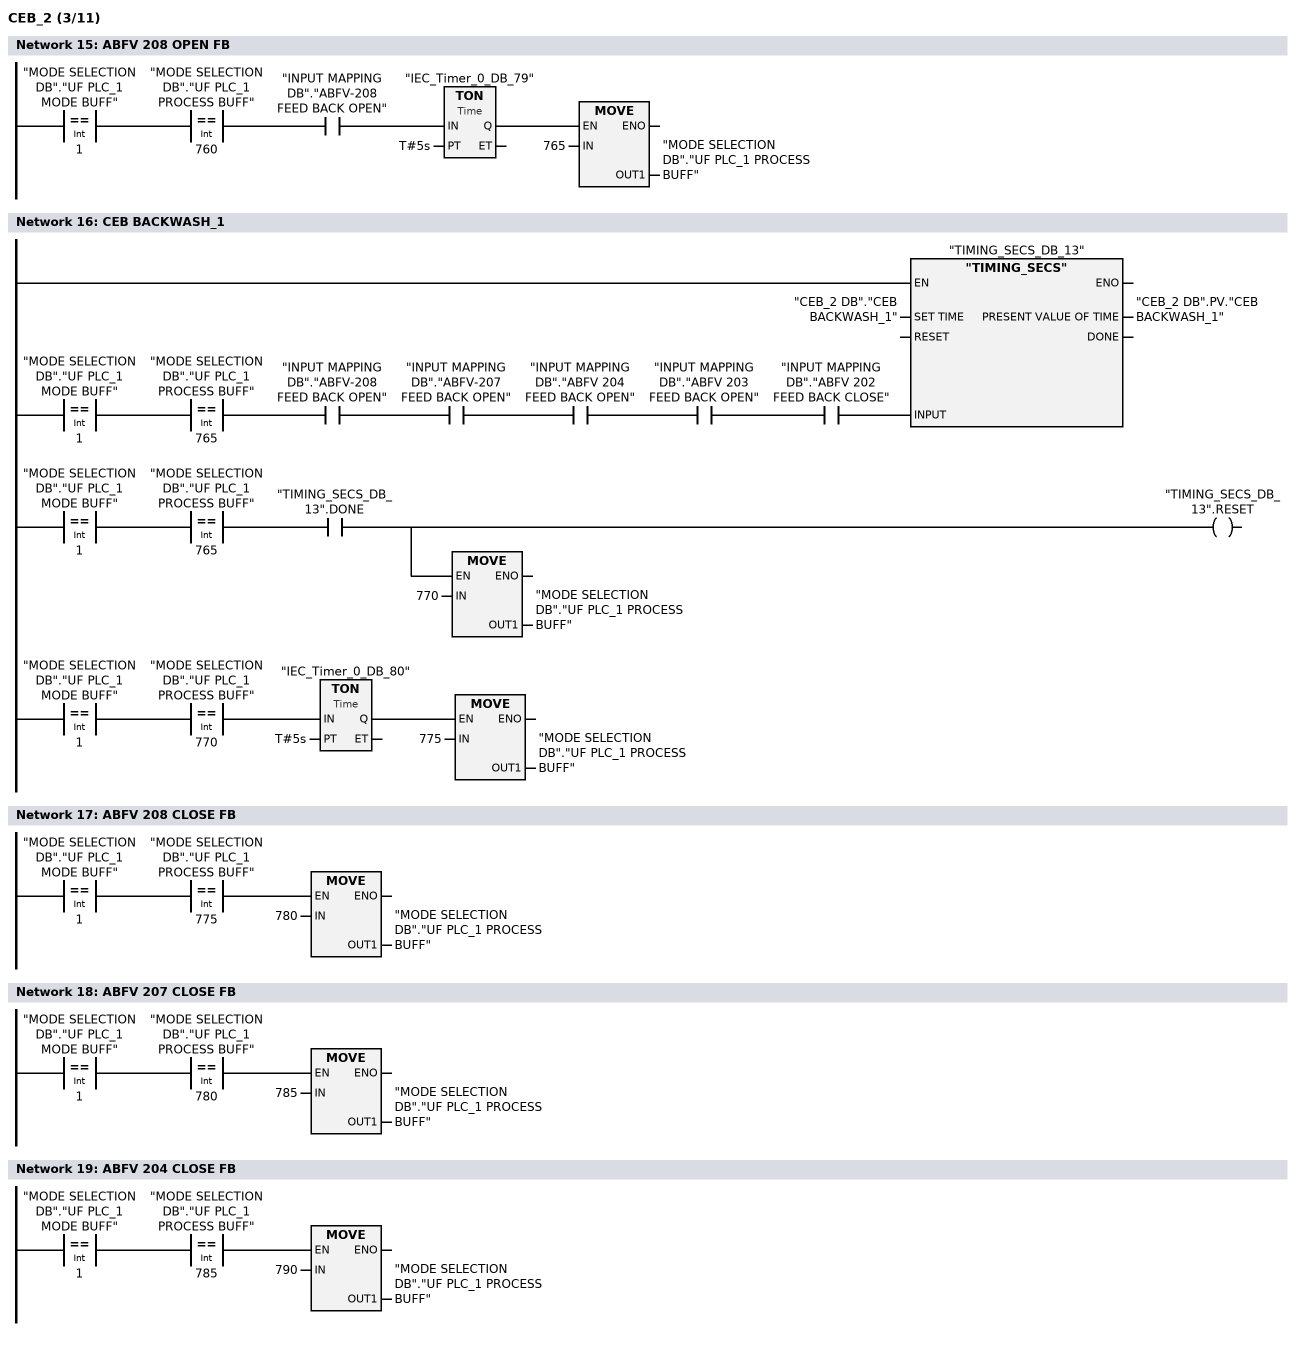
   RUNG wire#powerrail
      { S7_Templates := "SrcType := Int" } EQ_Contact(in1 := "MODE SELECTION DB"."UF PLC_1 MODE BUFF", in2 := 1)
      { S7_Templates := "SrcType := Int" } EQ_Contact(in1 := "MODE SELECTION DB"."UF PLC_1 PROCESS BUFF", in2 := 760)
      Contact( "INPUT MAPPING DB"."ABFV-208 FEED BACK OPEN" )
      { S7_Templates := "time_type := Time" } "IEC_Timer_0_DB_79".TON(pt := T#5s, et =>)
      Move(in := 765, out1 => "MODE SELECTION DB"."UF PLC_1 PROCESS BUFF")
   END_RUNG
   // the same network as SCL:
   "IEC_Timer_0_DB_79".TON(IN := ("MODE SELECTION DB"."UF PLC_1 MODE BUFF" = 1) AND ("MODE SELECTION DB"."UF PLC_1 PROCESS BUFF" = 760) AND "INPUT MAPPING DB"."ABFV-208 FEED BACK OPEN",
                           PT := T#5s);
   IF "IEC_Timer_0_DB_79".Q THEN "MODE SELECTION DB"."UF PLC_1 PROCESS BUFF" := 765; END_IF;
END_REGION

REGION Network 16: CEB BACKWASH_1
   RUNG wire#powerrail
      "TIMING_SECS_DB_13"(INPUT := wire#w1, "SET TIME" := "CEB_2 DB"."CEB BACKWASH_1", RESET :=, "PRESENT VALUE OF TIME" => "CEB_2 DB".PV."CEB BACKWASH_1", DONE =>)
   END_RUNG
   RUNG wire#powerrail
      { S7_Templates := "SrcType := Int" } EQ_Contact(in1 := "MODE SELECTION DB"."UF PLC_1 MODE BUFF", in2 := 1)
      { S7_Templates := "SrcType := Int" } EQ_Contact(in1 := "MODE SELECTION DB"."UF PLC_1 PROCESS BUFF", in2 := 765)
      Contact( "INPUT MAPPING DB"."ABFV-208 FEED BACK OPEN" )
      Contact( "INPUT MAPPING DB"."ABFV-207 FEED BACK OPEN" )
      Contact( "INPUT MAPPING DB"."ABFV 204 FEED BACK OPEN" )
      Contact( "INPUT MAPPING DB"."ABFV 203 FEED BACK OPEN" )
      Contact( "INPUT MAPPING DB"."ABFV 202 FEED BACK CLOSE" )
   END_RUNG wire#w1
   RUNG wire#powerrail
      { S7_Templates := "SrcType := Int" } EQ_Contact(in1 := "MODE SELECTION DB"."UF PLC_1 MODE BUFF", in2 := 1)
      { S7_Templates := "SrcType := Int" } EQ_Contact(in1 := "MODE SELECTION DB"."UF PLC_1 PROCESS BUFF", in2 := 765)
      Contact( "TIMING_SECS_DB_13".DONE )
      wire#w2
      Coil( "TIMING_SECS_DB_13".RESET )
   END_RUNG
   RUNG wire#w2
      Move(in := 770, out1 => "MODE SELECTION DB"."UF PLC_1 PROCESS BUFF")
   END_RUNG
   RUNG wire#powerrail
      { S7_Templates := "SrcType := Int" } EQ_Contact(in1 := "MODE SELECTION DB"."UF PLC_1 MODE BUFF", in2 := 1)
      { S7_Templates := "SrcType := Int" } EQ_Contact(in1 := "MODE SELECTION DB"."UF PLC_1 PROCESS BUFF", in2 := 770)
      { S7_Templates := "time_type := Time" } "IEC_Timer_0_DB_80".TON(pt := T#5s, et =>)
      Move(in := 775, out1 => "MODE SELECTION DB"."UF PLC_1 PROCESS BUFF")
   END_RUNG
   // the same network as SCL:
   "TIMING_SECS_DB_13"("SET TIME" := "CEB_2 DB"."CEB BACKWASH_1",   // "TIMING_SECS"
                       INPUT := ("MODE SELECTION DB"."UF PLC_1 MODE BUFF" = 1) AND ("MODE SELECTION DB"."UF PLC_1 PROCESS BUFF" = 765) AND "INPUT MAPPING DB"."ABFV-208 FEED BACK OPEN" AND "INPUT MAPPING DB"."ABFV-207 FEED BACK OPEN" AND "INPUT MAPPING DB"."ABFV 204 FEED BACK OPEN" AND "INPUT MAPPING DB"."ABFV 203 FEED BACK OPEN" AND "INPUT MAPPING DB"."ABFV 202 FEED BACK CLOSE",
                       "PRESENT VALUE OF TIME" => "CEB_2 DB".PV."CEB BACKWASH_1");
   "TIMING_SECS_DB_13".RESET := ("MODE SELECTION DB"."UF PLC_1 MODE BUFF" = 1) AND ("MODE SELECTION DB"."UF PLC_1 PROCESS BUFF" = 765) AND "TIMING_SECS_DB_13".DONE;
   IF "TIMING_SECS_DB_13".RESET THEN "MODE SELECTION DB"."UF PLC_1 PROCESS BUFF" := 770; END_IF;
   "IEC_Timer_0_DB_80".TON(IN := ("MODE SELECTION DB"."UF PLC_1 MODE BUFF" = 1) AND ("MODE SELECTION DB"."UF PLC_1 PROCESS BUFF" = 770),
                           PT := T#5s);
   IF "IEC_Timer_0_DB_80".Q THEN "MODE SELECTION DB"."UF PLC_1 PROCESS BUFF" := 775; END_IF;
END_REGION

REGION Network 17: ABFV 208 CLOSE FB
   RUNG wire#powerrail
      { S7_Templates := "SrcType := Int" } EQ_Contact(in1 := "MODE SELECTION DB"."UF PLC_1 MODE BUFF", in2 := 1)
      { S7_Templates := "SrcType := Int" } EQ_Contact(in1 := "MODE SELECTION DB"."UF PLC_1 PROCESS BUFF", in2 := 775)
      Move(in := 780, out1 => "MODE SELECTION DB"."UF PLC_1 PROCESS BUFF")
   END_RUNG
   // the same network as SCL:
   IF ("MODE SELECTION DB"."UF PLC_1 MODE BUFF" = 1) AND ("MODE SELECTION DB"."UF PLC_1 PROCESS BUFF" = 775) THEN
       "MODE SELECTION DB"."UF PLC_1 PROCESS BUFF" := 780;
   END_IF;
END_REGION

REGION Network 18: ABFV 207 CLOSE FB
   RUNG wire#powerrail
      { S7_Templates := "SrcType := Int" } EQ_Contact(in1 := "MODE SELECTION DB"."UF PLC_1 MODE BUFF", in2 := 1)
      { S7_Templates := "SrcType := Int" } EQ_Contact(in1 := "MODE SELECTION DB"."UF PLC_1 PROCESS BUFF", in2 := 780)
      Move(in := 785, out1 => "MODE SELECTION DB"."UF PLC_1 PROCESS BUFF")
   END_RUNG
   // the same network as SCL:
   IF ("MODE SELECTION DB"."UF PLC_1 MODE BUFF" = 1) AND ("MODE SELECTION DB"."UF PLC_1 PROCESS BUFF" = 780) THEN
       "MODE SELECTION DB"."UF PLC_1 PROCESS BUFF" := 785;
   END_IF;
END_REGION

REGION Network 19: ABFV 204 CLOSE FB
   RUNG wire#powerrail
      { S7_Templates := "SrcType := Int" } EQ_Contact(in1 := "MODE SELECTION DB"."UF PLC_1 MODE BUFF", in2 := 1)
      { S7_Templates := "SrcType := Int" } EQ_Contact(in1 := "MODE SELECTION DB"."UF PLC_1 PROCESS BUFF", in2 := 785)
      Move(in := 790, out1 => "MODE SELECTION DB"."UF PLC_1 PROCESS BUFF")
   END_RUNG
   // the same network as SCL:
   IF ("MODE SELECTION DB"."UF PLC_1 MODE BUFF" = 1) AND ("MODE SELECTION DB"."UF PLC_1 PROCESS BUFF" = 785) THEN
       "MODE SELECTION DB"."UF PLC_1 PROCESS BUFF" := 790;
   END_IF;
END_REGION

REGION Network 20: ABFV 203 CLOSE FB
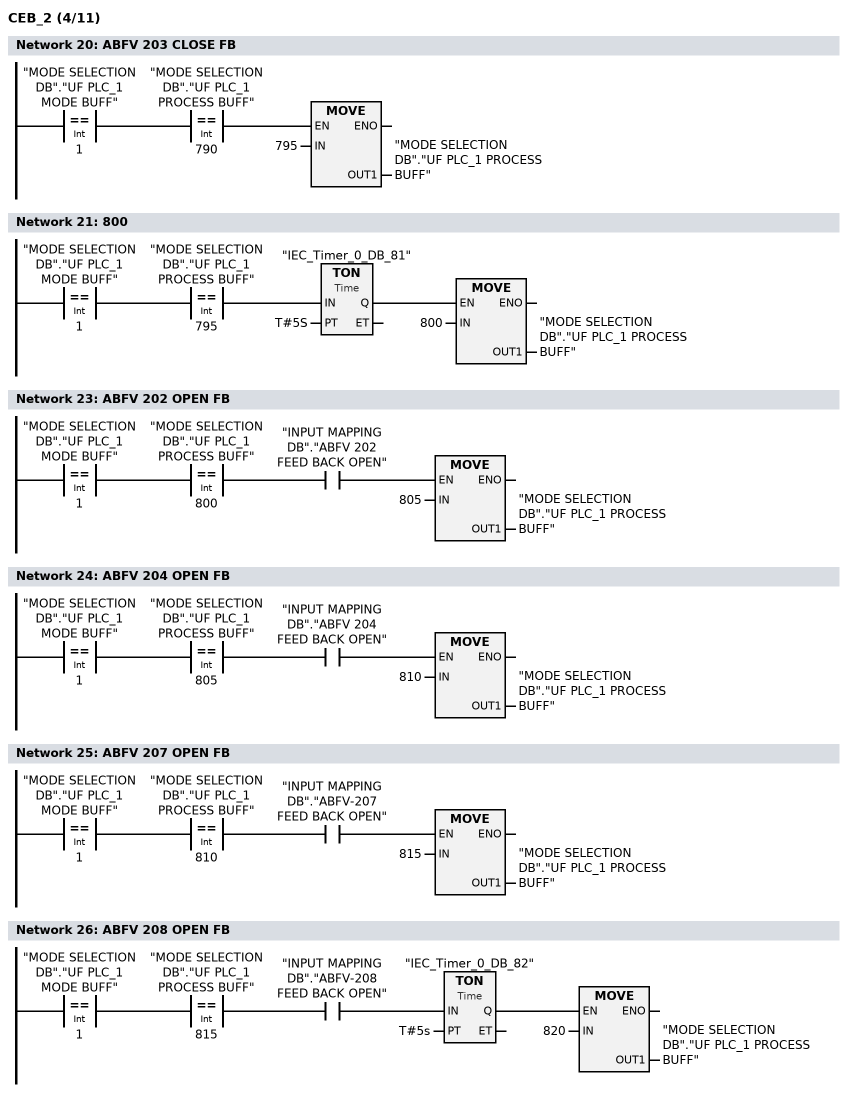
   RUNG wire#powerrail
      { S7_Templates := "SrcType := Int" } EQ_Contact(in1 := "MODE SELECTION DB"."UF PLC_1 MODE BUFF", in2 := 1)
      { S7_Templates := "SrcType := Int" } EQ_Contact(in1 := "MODE SELECTION DB"."UF PLC_1 PROCESS BUFF", in2 := 790)
      Move(in := 795, out1 => "MODE SELECTION DB"."UF PLC_1 PROCESS BUFF")
   END_RUNG
   // the same network as SCL:
   IF ("MODE SELECTION DB"."UF PLC_1 MODE BUFF" = 1) AND ("MODE SELECTION DB"."UF PLC_1 PROCESS BUFF" = 790) THEN
       "MODE SELECTION DB"."UF PLC_1 PROCESS BUFF" := 795;
   END_IF;
END_REGION

REGION Network 21: 800
   RUNG wire#powerrail
      { S7_Templates := "SrcType := Int" } EQ_Contact(in1 := "MODE SELECTION DB"."UF PLC_1 MODE BUFF", in2 := 1)
      { S7_Templates := "SrcType := Int" } EQ_Contact(in1 := "MODE SELECTION DB"."UF PLC_1 PROCESS BUFF", in2 := 795)
      { S7_Templates := "time_type := Time" } "IEC_Timer_0_DB_81".TON(pt := T#5S, et =>)
      Move(in := 800, out1 => "MODE SELECTION DB"."UF PLC_1 PROCESS BUFF")
   END_RUNG
   // the same network as SCL:
   "IEC_Timer_0_DB_81".TON(IN := ("MODE SELECTION DB"."UF PLC_1 MODE BUFF" = 1) AND ("MODE SELECTION DB"."UF PLC_1 PROCESS BUFF" = 795),
                           PT := T#5S);
   IF "IEC_Timer_0_DB_81".Q THEN "MODE SELECTION DB"."UF PLC_1 PROCESS BUFF" := 800; END_IF;
END_REGION

REGION Network 23: ABFV 202 OPEN FB
   RUNG wire#powerrail
      { S7_Templates := "SrcType := Int" } EQ_Contact(in1 := "MODE SELECTION DB"."UF PLC_1 MODE BUFF", in2 := 1)
      { S7_Templates := "SrcType := Int" } EQ_Contact(in1 := "MODE SELECTION DB"."UF PLC_1 PROCESS BUFF", in2 := 800)
      Contact( "INPUT MAPPING DB"."ABFV 202 FEED BACK OPEN" )
      Move(in := 805, out1 => "MODE SELECTION DB"."UF PLC_1 PROCESS BUFF")
   END_RUNG
   // the same network as SCL:
   IF ("MODE SELECTION DB"."UF PLC_1 MODE BUFF" = 1) AND ("MODE SELECTION DB"."UF PLC_1 PROCESS BUFF" = 800) AND "INPUT MAPPING DB"."ABFV 202 FEED BACK OPEN" THEN
       "MODE SELECTION DB"."UF PLC_1 PROCESS BUFF" := 805;
   END_IF;
END_REGION

REGION Network 24: ABFV 204 OPEN FB
   RUNG wire#powerrail
      { S7_Templates := "SrcType := Int" } EQ_Contact(in1 := "MODE SELECTION DB"."UF PLC_1 MODE BUFF", in2 := 1)
      { S7_Templates := "SrcType := Int" } EQ_Contact(in1 := "MODE SELECTION DB"."UF PLC_1 PROCESS BUFF", in2 := 805)
      Contact( "INPUT MAPPING DB"."ABFV 204 FEED BACK OPEN" )
      Move(in := 810, out1 => "MODE SELECTION DB"."UF PLC_1 PROCESS BUFF")
   END_RUNG
   // the same network as SCL:
   IF ("MODE SELECTION DB"."UF PLC_1 MODE BUFF" = 1) AND ("MODE SELECTION DB"."UF PLC_1 PROCESS BUFF" = 805) AND "INPUT MAPPING DB"."ABFV 204 FEED BACK OPEN" THEN
       "MODE SELECTION DB"."UF PLC_1 PROCESS BUFF" := 810;
   END_IF;
END_REGION

REGION Network 25: ABFV 207 OPEN FB
   RUNG wire#powerrail
      { S7_Templates := "SrcType := Int" } EQ_Contact(in1 := "MODE SELECTION DB"."UF PLC_1 MODE BUFF", in2 := 1)
      { S7_Templates := "SrcType := Int" } EQ_Contact(in1 := "MODE SELECTION DB"."UF PLC_1 PROCESS BUFF", in2 := 810)
      Contact( "INPUT MAPPING DB"."ABFV-207 FEED BACK OPEN" )
      Move(in := 815, out1 => "MODE SELECTION DB"."UF PLC_1 PROCESS BUFF")
   END_RUNG
   // the same network as SCL:
   IF ("MODE SELECTION DB"."UF PLC_1 MODE BUFF" = 1) AND ("MODE SELECTION DB"."UF PLC_1 PROCESS BUFF" = 810) AND "INPUT MAPPING DB"."ABFV-207 FEED BACK OPEN" THEN
       "MODE SELECTION DB"."UF PLC_1 PROCESS BUFF" := 815;
   END_IF;
END_REGION

REGION Network 26: ABFV 208 OPEN FB
   RUNG wire#powerrail
      { S7_Templates := "SrcType := Int" } EQ_Contact(in1 := "MODE SELECTION DB"."UF PLC_1 MODE BUFF", in2 := 1)
      { S7_Templates := "SrcType := Int" } EQ_Contact(in1 := "MODE SELECTION DB"."UF PLC_1 PROCESS BUFF", in2 := 815)
      Contact( "INPUT MAPPING DB"."ABFV-208 FEED BACK OPEN" )
      { S7_Templates := "time_type := Time" } "IEC_Timer_0_DB_82".TON(pt := T#5s, et =>)
      Move(in := 820, out1 => "MODE SELECTION DB"."UF PLC_1 PROCESS BUFF")
   END_RUNG
   // the same network as SCL:
   "IEC_Timer_0_DB_82".TON(IN := ("MODE SELECTION DB"."UF PLC_1 MODE BUFF" = 1) AND ("MODE SELECTION DB"."UF PLC_1 PROCESS BUFF" = 815) AND "INPUT MAPPING DB"."ABFV-208 FEED BACK OPEN",
                           PT := T#5s);
   IF "IEC_Timer_0_DB_82".Q THEN "MODE SELECTION DB"."UF PLC_1 PROCESS BUFF" := 820; END_IF;
END_REGION

REGION Network 27: CEB BACKWASH_2
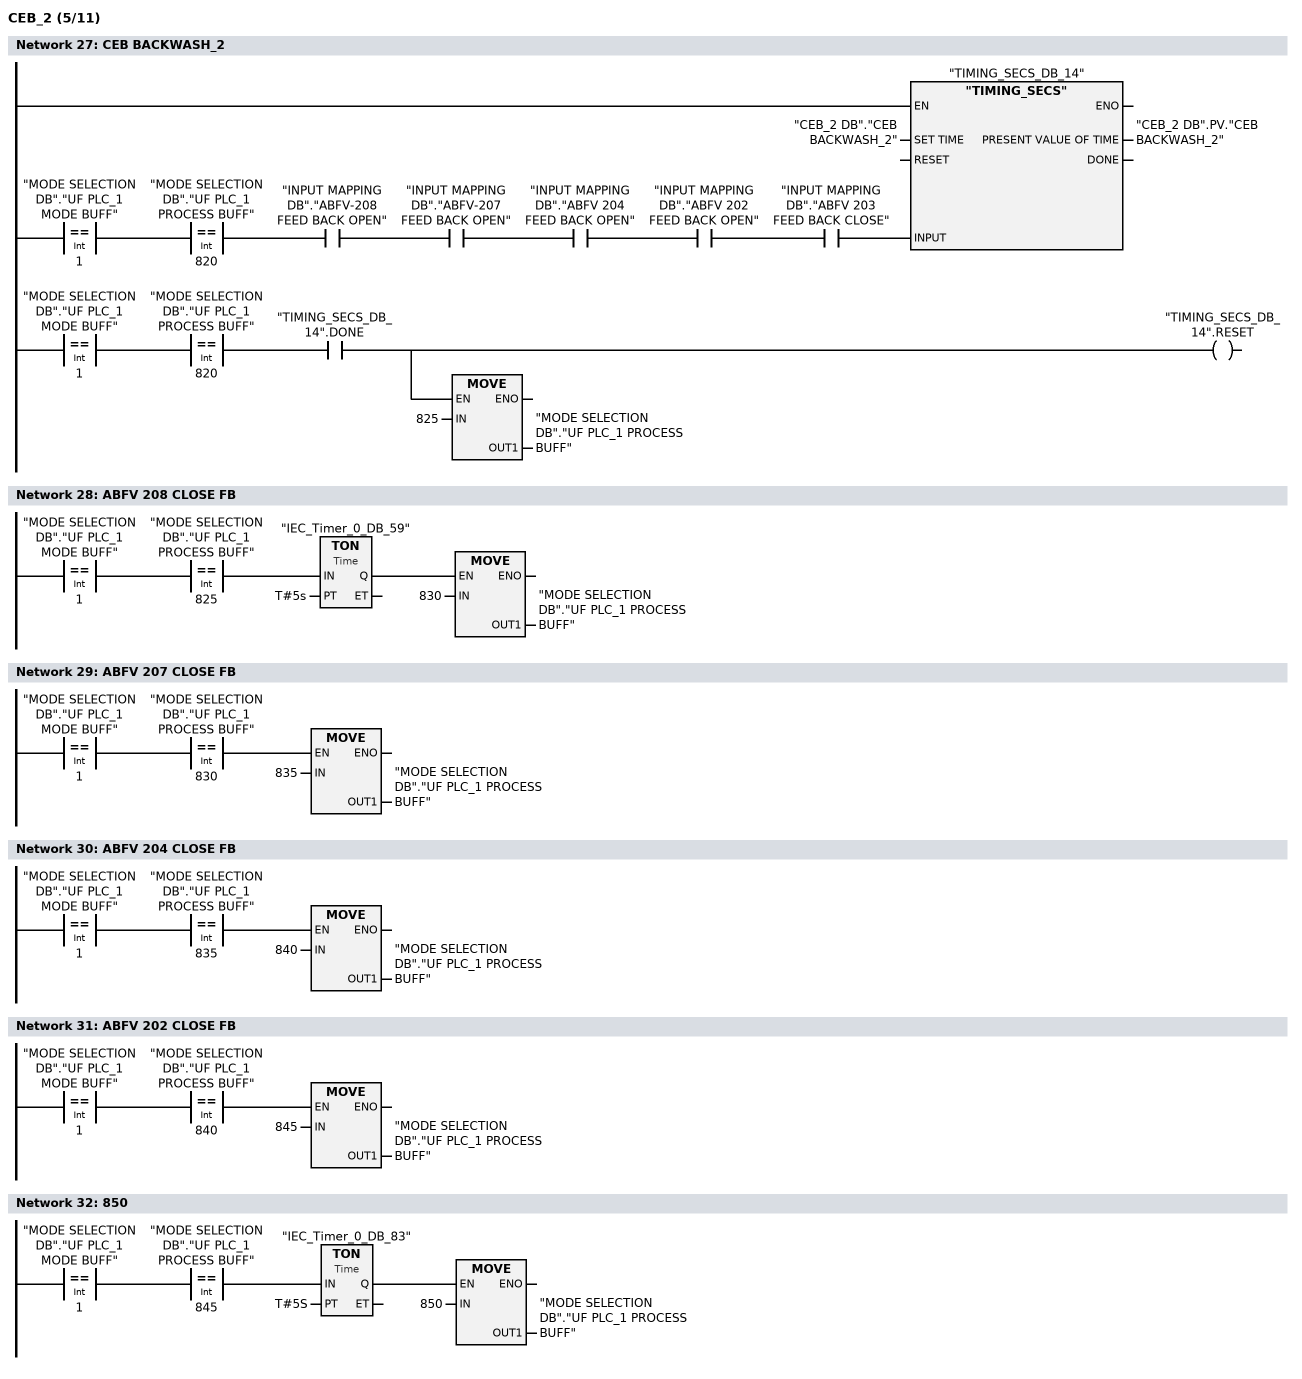
   RUNG wire#powerrail
      "TIMING_SECS_DB_14"(INPUT := wire#w1, "SET TIME" := "CEB_2 DB"."CEB BACKWASH_2", RESET :=, "PRESENT VALUE OF TIME" => "CEB_2 DB".PV."CEB BACKWASH_2", DONE =>)
   END_RUNG
   RUNG wire#powerrail
      { S7_Templates := "SrcType := Int" } EQ_Contact(in1 := "MODE SELECTION DB"."UF PLC_1 MODE BUFF", in2 := 1)
      { S7_Templates := "SrcType := Int" } EQ_Contact(in1 := "MODE SELECTION DB"."UF PLC_1 PROCESS BUFF", in2 := 820)
      Contact( "INPUT MAPPING DB"."ABFV-208 FEED BACK OPEN" )
      Contact( "INPUT MAPPING DB"."ABFV-207 FEED BACK OPEN" )
      Contact( "INPUT MAPPING DB"."ABFV 204 FEED BACK OPEN" )
      Contact( "INPUT MAPPING DB"."ABFV 202 FEED BACK OPEN" )
      Contact( "INPUT MAPPING DB"."ABFV 203 FEED BACK CLOSE" )
   END_RUNG wire#w1
   RUNG wire#powerrail
      { S7_Templates := "SrcType := Int" } EQ_Contact(in1 := "MODE SELECTION DB"."UF PLC_1 MODE BUFF", in2 := 1)
      { S7_Templates := "SrcType := Int" } EQ_Contact(in1 := "MODE SELECTION DB"."UF PLC_1 PROCESS BUFF", in2 := 820)
      Contact( "TIMING_SECS_DB_14".DONE )
      wire#w2
      Coil( "TIMING_SECS_DB_14".RESET )
   END_RUNG
   RUNG wire#w2
      Move(in := 825, out1 => "MODE SELECTION DB"."UF PLC_1 PROCESS BUFF")
   END_RUNG
   // the same network as SCL:
   "TIMING_SECS_DB_14"("SET TIME" := "CEB_2 DB"."CEB BACKWASH_2",   // "TIMING_SECS"
                       INPUT := ("MODE SELECTION DB"."UF PLC_1 MODE BUFF" = 1) AND ("MODE SELECTION DB"."UF PLC_1 PROCESS BUFF" = 820) AND "INPUT MAPPING DB"."ABFV-208 FEED BACK OPEN" AND "INPUT MAPPING DB"."ABFV-207 FEED BACK OPEN" AND "INPUT MAPPING DB"."ABFV 204 FEED BACK OPEN" AND "INPUT MAPPING DB"."ABFV 202 FEED BACK OPEN" AND "INPUT MAPPING DB"."ABFV 203 FEED BACK CLOSE",
                       "PRESENT VALUE OF TIME" => "CEB_2 DB".PV."CEB BACKWASH_2");
   "TIMING_SECS_DB_14".RESET := ("MODE SELECTION DB"."UF PLC_1 MODE BUFF" = 1) AND ("MODE SELECTION DB"."UF PLC_1 PROCESS BUFF" = 820) AND "TIMING_SECS_DB_14".DONE;
   IF "TIMING_SECS_DB_14".RESET THEN "MODE SELECTION DB"."UF PLC_1 PROCESS BUFF" := 825; END_IF;
END_REGION

REGION Network 28: ABFV 208 CLOSE FB
   RUNG wire#powerrail
      { S7_Templates := "SrcType := Int" } EQ_Contact(in1 := "MODE SELECTION DB"."UF PLC_1 MODE BUFF", in2 := 1)
      { S7_Templates := "SrcType := Int" } EQ_Contact(in1 := "MODE SELECTION DB"."UF PLC_1 PROCESS BUFF", in2 := 825)
      { S7_Templates := "time_type := Time" } "IEC_Timer_0_DB_59".TON(pt := T#5s, et =>)
      Move(in := 830, out1 => "MODE SELECTION DB"."UF PLC_1 PROCESS BUFF")
   END_RUNG
   // the same network as SCL:
   "IEC_Timer_0_DB_59".TON(IN := ("MODE SELECTION DB"."UF PLC_1 MODE BUFF" = 1) AND ("MODE SELECTION DB"."UF PLC_1 PROCESS BUFF" = 825),
                           PT := T#5s);
   IF "IEC_Timer_0_DB_59".Q THEN "MODE SELECTION DB"."UF PLC_1 PROCESS BUFF" := 830; END_IF;
END_REGION

REGION Network 29: ABFV 207 CLOSE FB
   RUNG wire#powerrail
      { S7_Templates := "SrcType := Int" } EQ_Contact(in1 := "MODE SELECTION DB"."UF PLC_1 MODE BUFF", in2 := 1)
      { S7_Templates := "SrcType := Int" } EQ_Contact(in1 := "MODE SELECTION DB"."UF PLC_1 PROCESS BUFF", in2 := 830)
      Move(in := 835, out1 => "MODE SELECTION DB"."UF PLC_1 PROCESS BUFF")
   END_RUNG
   // the same network as SCL:
   IF ("MODE SELECTION DB"."UF PLC_1 MODE BUFF" = 1) AND ("MODE SELECTION DB"."UF PLC_1 PROCESS BUFF" = 830) THEN
       "MODE SELECTION DB"."UF PLC_1 PROCESS BUFF" := 835;
   END_IF;
END_REGION

REGION Network 30: ABFV 204 CLOSE FB
   RUNG wire#powerrail
      { S7_Templates := "SrcType := Int" } EQ_Contact(in1 := "MODE SELECTION DB"."UF PLC_1 MODE BUFF", in2 := 1)
      { S7_Templates := "SrcType := Int" } EQ_Contact(in1 := "MODE SELECTION DB"."UF PLC_1 PROCESS BUFF", in2 := 835)
      Move(in := 840, out1 => "MODE SELECTION DB"."UF PLC_1 PROCESS BUFF")
   END_RUNG
   // the same network as SCL:
   IF ("MODE SELECTION DB"."UF PLC_1 MODE BUFF" = 1) AND ("MODE SELECTION DB"."UF PLC_1 PROCESS BUFF" = 835) THEN
       "MODE SELECTION DB"."UF PLC_1 PROCESS BUFF" := 840;
   END_IF;
END_REGION

REGION Network 31: ABFV 202 CLOSE FB
   RUNG wire#powerrail
      { S7_Templates := "SrcType := Int" } EQ_Contact(in1 := "MODE SELECTION DB"."UF PLC_1 MODE BUFF", in2 := 1)
      { S7_Templates := "SrcType := Int" } EQ_Contact(in1 := "MODE SELECTION DB"."UF PLC_1 PROCESS BUFF", in2 := 840)
      Move(in := 845, out1 => "MODE SELECTION DB"."UF PLC_1 PROCESS BUFF")
   END_RUNG
   // the same network as SCL:
   IF ("MODE SELECTION DB"."UF PLC_1 MODE BUFF" = 1) AND ("MODE SELECTION DB"."UF PLC_1 PROCESS BUFF" = 840) THEN
       "MODE SELECTION DB"."UF PLC_1 PROCESS BUFF" := 845;
   END_IF;
END_REGION

REGION Network 32: 850
   RUNG wire#powerrail
      { S7_Templates := "SrcType := Int" } EQ_Contact(in1 := "MODE SELECTION DB"."UF PLC_1 MODE BUFF", in2 := 1)
      { S7_Templates := "SrcType := Int" } EQ_Contact(in1 := "MODE SELECTION DB"."UF PLC_1 PROCESS BUFF", in2 := 845)
      { S7_Templates := "time_type := Time" } "IEC_Timer_0_DB_83".TON(pt := T#5S, et =>)
      Move(in := 850, out1 => "MODE SELECTION DB"."UF PLC_1 PROCESS BUFF")
   END_RUNG
   // the same network as SCL:
   "IEC_Timer_0_DB_83".TON(IN := ("MODE SELECTION DB"."UF PLC_1 MODE BUFF" = 1) AND ("MODE SELECTION DB"."UF PLC_1 PROCESS BUFF" = 845),
                           PT := T#5S);
   IF "IEC_Timer_0_DB_83".Q THEN "MODE SELECTION DB"."UF PLC_1 PROCESS BUFF" := 850; END_IF;
END_REGION

REGION Network 34: SOAK
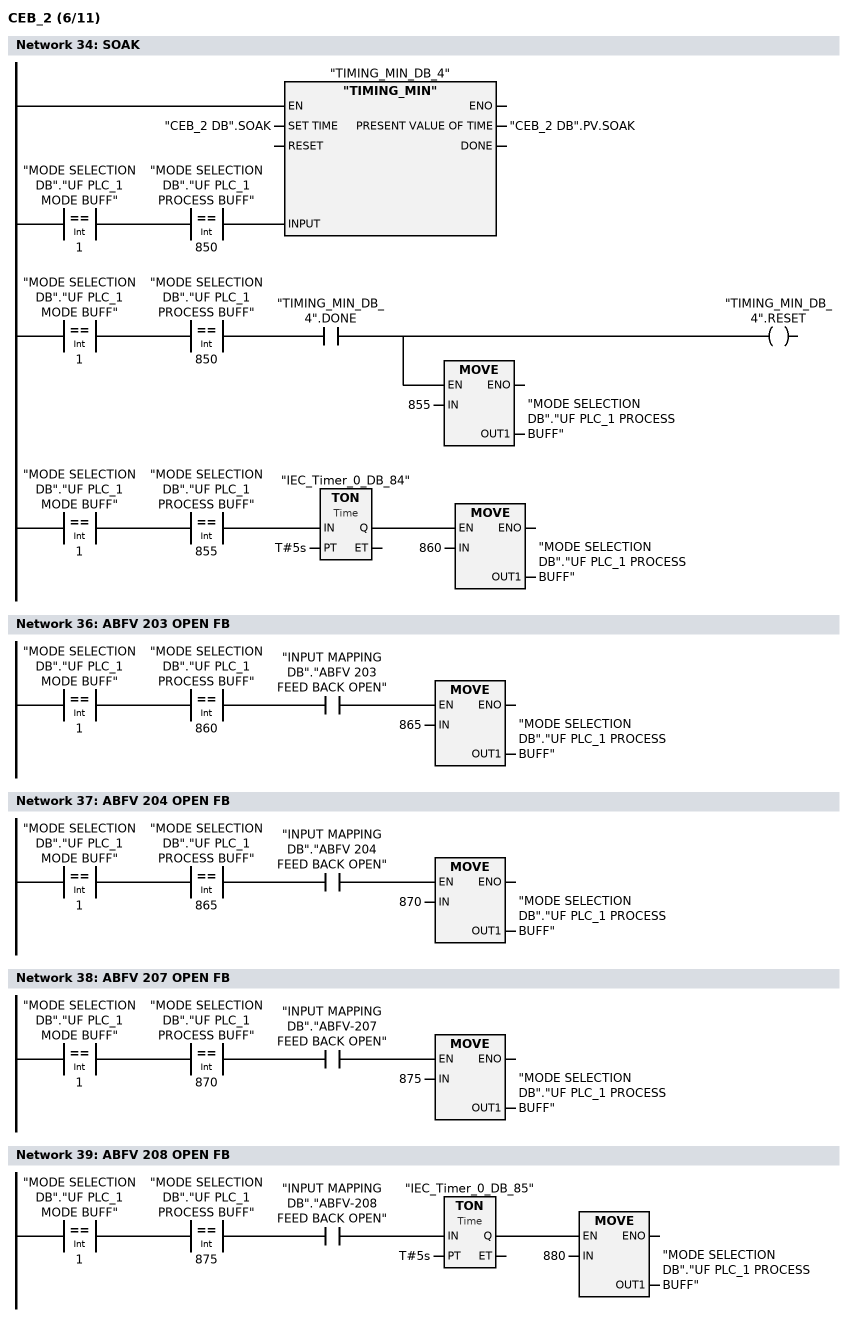
   RUNG wire#powerrail
      "TIMING_MIN_DB_4"(INPUT := wire#w1, "SET TIME" := "CEB_2 DB".SOAK, RESET :=, "PRESENT VALUE OF TIME" => "CEB_2 DB".PV.SOAK, DONE =>)
   END_RUNG
   RUNG wire#powerrail
      { S7_Templates := "SrcType := Int" } EQ_Contact(in1 := "MODE SELECTION DB"."UF PLC_1 MODE BUFF", in2 := 1)
      { S7_Templates := "SrcType := Int" } EQ_Contact(in1 := "MODE SELECTION DB"."UF PLC_1 PROCESS BUFF", in2 := 850)
   END_RUNG wire#w1
   RUNG wire#powerrail
      { S7_Templates := "SrcType := Int" } EQ_Contact(in1 := "MODE SELECTION DB"."UF PLC_1 MODE BUFF", in2 := 1)
      { S7_Templates := "SrcType := Int" } EQ_Contact(in1 := "MODE SELECTION DB"."UF PLC_1 PROCESS BUFF", in2 := 850)
      Contact( "TIMING_MIN_DB_4".DONE )
      wire#w2
      Coil( "TIMING_MIN_DB_4".RESET )
   END_RUNG
   RUNG wire#w2
      Move(in := 855, out1 => "MODE SELECTION DB"."UF PLC_1 PROCESS BUFF")
   END_RUNG
   RUNG wire#powerrail
      { S7_Templates := "SrcType := Int" } EQ_Contact(in1 := "MODE SELECTION DB"."UF PLC_1 MODE BUFF", in2 := 1)
      { S7_Templates := "SrcType := Int" } EQ_Contact(in1 := "MODE SELECTION DB"."UF PLC_1 PROCESS BUFF", in2 := 855)
      { S7_Templates := "time_type := Time" } "IEC_Timer_0_DB_84".TON(pt := T#5s, et =>)
      Move(in := 860, out1 => "MODE SELECTION DB"."UF PLC_1 PROCESS BUFF")
   END_RUNG
   // the same network as SCL:
   "TIMING_MIN_DB_4"("SET TIME" := "CEB_2 DB".SOAK,   // "TIMING_MIN"
                     INPUT := ("MODE SELECTION DB"."UF PLC_1 MODE BUFF" = 1) AND ("MODE SELECTION DB"."UF PLC_1 PROCESS BUFF" = 850),
                     "PRESENT VALUE OF TIME" => "CEB_2 DB".PV.SOAK);
   "TIMING_MIN_DB_4".RESET := ("MODE SELECTION DB"."UF PLC_1 MODE BUFF" = 1) AND ("MODE SELECTION DB"."UF PLC_1 PROCESS BUFF" = 850) AND "TIMING_MIN_DB_4".DONE;
   IF "TIMING_MIN_DB_4".RESET THEN "MODE SELECTION DB"."UF PLC_1 PROCESS BUFF" := 855; END_IF;
   "IEC_Timer_0_DB_84".TON(IN := ("MODE SELECTION DB"."UF PLC_1 MODE BUFF" = 1) AND ("MODE SELECTION DB"."UF PLC_1 PROCESS BUFF" = 855),
                           PT := T#5s);
   IF "IEC_Timer_0_DB_84".Q THEN "MODE SELECTION DB"."UF PLC_1 PROCESS BUFF" := 860; END_IF;
END_REGION

REGION Network 36: ABFV 203 OPEN FB
   RUNG wire#powerrail
      { S7_Templates := "SrcType := Int" } EQ_Contact(in1 := "MODE SELECTION DB"."UF PLC_1 MODE BUFF", in2 := 1)
      { S7_Templates := "SrcType := Int" } EQ_Contact(in1 := "MODE SELECTION DB"."UF PLC_1 PROCESS BUFF", in2 := 860)
      Contact( "INPUT MAPPING DB"."ABFV 203 FEED BACK OPEN" )
      Move(in := 865, out1 => "MODE SELECTION DB"."UF PLC_1 PROCESS BUFF")
   END_RUNG
   // the same network as SCL:
   IF ("MODE SELECTION DB"."UF PLC_1 MODE BUFF" = 1) AND ("MODE SELECTION DB"."UF PLC_1 PROCESS BUFF" = 860) AND "INPUT MAPPING DB"."ABFV 203 FEED BACK OPEN" THEN
       "MODE SELECTION DB"."UF PLC_1 PROCESS BUFF" := 865;
   END_IF;
END_REGION

REGION Network 37: ABFV 204 OPEN FB
   RUNG wire#powerrail
      { S7_Templates := "SrcType := Int" } EQ_Contact(in1 := "MODE SELECTION DB"."UF PLC_1 MODE BUFF", in2 := 1)
      { S7_Templates := "SrcType := Int" } EQ_Contact(in1 := "MODE SELECTION DB"."UF PLC_1 PROCESS BUFF", in2 := 865)
      Contact( "INPUT MAPPING DB"."ABFV 204 FEED BACK OPEN" )
      Move(in := 870, out1 => "MODE SELECTION DB"."UF PLC_1 PROCESS BUFF")
   END_RUNG
   // the same network as SCL:
   IF ("MODE SELECTION DB"."UF PLC_1 MODE BUFF" = 1) AND ("MODE SELECTION DB"."UF PLC_1 PROCESS BUFF" = 865) AND "INPUT MAPPING DB"."ABFV 204 FEED BACK OPEN" THEN
       "MODE SELECTION DB"."UF PLC_1 PROCESS BUFF" := 870;
   END_IF;
END_REGION

